// TIA Portal project "pro_2EV_N" (V16)
// Programa original de la laminadora

(* hardware
DEVICE "S7-1200 station_1"  S7-1200 Station
   slot 0: "Telaio di montaggio_0"  S7-1200 Rack  Rack  V1.0
   slot 1: "PLC"  CPU 1214C DC/DC/DC  6ES7 214-1AG40-0XB0  V4.4
   slot 2: "DQ 8x24VDC _1"  SM 1222 DQ8 x 24VDC  6ES7 222-1BF32-0XB0  V2.0
   slot 3: "AI 4xTC_1"  SM 1231 AI4 x TC  6ES7 231-5QD32-0XB0  V2.0
   slot 3: "DQ 4x24VDC_1"  DQ4 signal board (200 kHz)  6ES7 222-1BD30-0XB0  V1.0
*)

// ===== PLC "PLC"  CPU 1214C DC/DC/DC =====

VAR_GLOBAL   // PLC tag table "Tabla de variables estándar"
   "Emergenza" AT %I0.0 : Bool;
   "P_Reset" AT %I0.1 : Bool;
   "P_Stop_Sirena" AT %I0.2 : Bool;
   "Fc_Coperchio_Chiuso" AT %I0.5 : Bool;
   "Pressostato Aria" AT %I0.6 : Bool;
   "Fedd Back Pompa Vuoto" AT %I0.4 : Bool;
   "Analog Vuoto Sotto" AT %IW64 : Int;
   "Analog Vuoto Sopra" AT %IW66 : Int;
   "Feed Back Ins Resistenze" AT %I0.7 : Bool;
   "Temp 1 Basso" AT %IW128 : Int;
   "Temp 2 Basso" AT %IW130 : Int;
   "Temp 1 Alto" AT %IW132 : Int;
   "iw134" AT %IW134 : Word;
   "i0.3" AT %I0.3 : Bool;
   "Fc Pin Alti" AT %I1.0 : Bool;
   "Fc Pin Bassi" AT %I1.1 : Bool;
   "i1.2" AT %I1.2 : Bool;
   "i1.3" AT %I1.3 : Bool;
   "i1.4" AT %I1.4 : Bool;
   "qq" AT %Q2.6 : Bool;
   "Sirena" AT %Q0.0 : Bool;
   "Lamp_Allarme" AT %Q0.1 : Bool;
   "Lamp_Ciclo" AT %Q0.2 : Bool;
   "Lamp_Blu" AT %Q0.3 : Bool;
   "Comando Pompa vuoto" AT %Q0.4 : Bool;
   "EV Vuoto Sotto" AT %Q0.5 : Bool;
   "EV Aria Sotto" AT %Q0.6 : Bool;
   "Ev Big Vuoto Sopra" AT %Q0.7 : Bool;
   "Ev Big Aria Sopra" AT %Q1.0 : Bool;
   "Ev Small Aria Sopra" AT %Q1.1 : Bool;
   "Ev Small Vuoto Sopra" AT %Q2.0 : Bool;
   "Inserzione Resistenze" AT %Q2.1 : Bool;
   "Com Resistenze Basse" AT %Q2.2 : Bool;
   "Com Resistenze Alte" AT %Q2.3 : Bool;
   "EV H2O Raffredda" AT %Q2.4 : Bool;
   "EV Salita Pin" AT %Q2.5 : Bool;
   "Lamp_Reset" AT %Q2.7 : Bool;
   "System_Byte" AT %MB1 : Byte;
   "FirstScan" AT %M1.0 : Bool;
   "DiagStatusUpdate" AT %M1.1 : Bool;
   "AlwaysTRUE" AT %M1.2 : Bool;
   "AlwaysFALSE" AT %M1.3 : Bool;
   "Clock_Byte" AT %MB0 : Byte;
   "Clock_10Hz" AT %M0.0 : Bool;
   "Clock_5Hz" AT %M0.1 : Bool;
   "Clock_2.5Hz" AT %M0.2 : Bool;
   "Clock_2Hz" AT %M0.3 : Bool;
   "Clock_1.25Hz" AT %M0.4 : Bool;
   "Clock_1Hz" AT %M0.5 : Bool;
   "Clock_0.625Hz" AT %M0.6 : Bool;
   "Clock_0.5Hz" AT %M0.7 : Bool;
   "Start Temp Sotto" AT %M110.0 : Bool;
   "Start Temp Sopra" AT %M110.1 : Bool;
   "Mk Emergenza" AT %M90.0 : Bool;
   "Automatico" AT %M100.0 : Bool;
   "Automatico Start" AT %M100.1 : Bool;
   "Automatico Stop" AT %M100.2 : Bool;
   "Allarme" AT %M900.0 : Bool;
   "Ini Auto" AT %M100.3 : Bool;
   "Manuale" AT %M100.4 : Bool;
   "Com Resistenze Sotto" AT %M120.0 : Bool;
   "Com Resistenze Sopra" AT %M120.2 : Bool;
   "Start Vuoto Sotto" AT %M110.2 : Bool;
   "Start Vuoto Sopra" AT %M110.3 : Bool;
   "A1 Allarme Pompa Vuoto" AT %M1000.0 : Bool;
   "HMI Salta basso" AT %M35.0 : Bool;
   "M_OkNextStep" AT %M35.1 : Bool;
   "HMI Start Ciclo" AT %M50.0 : Bool;
   "Reset_T_Passo" AT %M300.0 : Bool;
   "HMI Stop Ciclo" AT %M50.1 : Bool;
   "Auto_ON" AT %M100.5 : Bool;
   "HMI Reset Ciclo" AT %M50.2 : Bool;
   "HMI Ciclo Terminato" AT %M50.3 : Bool;
   "Temp_Sotto in Range" AT %M111.0 : Bool;
   "Temp_Sopra in Range" AT %M111.1 : Bool;
   "Vuoto_Sotto in Range" AT %M111.2 : Bool;
   "Vuoto_Sopra in Range" AT %M111.3 : Bool;
   "S1 Fc Coperchio NON Chiuso" AT %M1010.0 : Bool;
   "MK_Registra_Temp" AT %M230.0 : Bool;
   "MK_Registra_Vuoto" AT %M230.1 : Bool;
   "Tempo_Passo OK" AT %M112.0 : Bool;
   "HMI Start Set Point Man Up" AT %M35.2 : Bool;
   "HMI Start Set Point Man Dw" AT %M35.3 : Bool;
   "HMI Set Point Man Gen" AT %M35.4 : Bool;
   "HMI Man Start Vuoto UP" AT %M35.5 : Bool;
   "HMI Man Start Vuoto DW" AT %M35.6 : Bool;
   "HMI Forzo Resistenze UP" AT %M35.7 : Bool;
   "HMI Forzo Resistenze DW" AT %M36.0 : Bool;
   "HMI Start Pompa Vuoto" AT %M36.1 : Bool;
   "HMI Com EV Vuoto Sotto" AT %M36.2 : Bool;
   "HMI Com EV Aria Sotto" AT %M36.3 : Bool;
   "HMI Com Ev Big Vuoto Sopra" AT %M36.4 : Bool;
   "HMI Com Ev Big Aria Sopra" AT %M36.5 : Bool;
   "HMI Com Ev Small Vuoto Sopra" AT %M36.6 : Bool;
   "HMI Com Resistenze Basse" AT %M37.0 : Bool;
   "HMI Com Resistenze Alte" AT %M37.1 : Bool;
   "HMI Com Ev Small Aria Sopra" AT %M36.7 : Bool;
   "HMI Stop Set Point Man Up" AT %M37.2 : Bool;
   "HMI Stop Set Point Man Dw" AT %M37.3 : Bool;
   "HMI Man Stop Vuoto UP" AT %M37.4 : Bool;
   "HMI Man Stop Vuoto DW" AT %M37.5 : Bool;
   "MK Man Resistenze UP" AT %M120.3 : Bool;
   "MK Man Resistenze DW" AT %M120.4 : Bool;
   "A2 All Max Temp Coperchio" AT %M1000.1 : Bool;
   "A3 All Max Temp Piastra" AT %M1000.2 : Bool;
   "A4 All Max Delta T" AT %M1000.3 : Bool;
   "Tag_1" AT %M10.0 : Bool;
   "Tag_2" AT %M11.0 : Bool;
   "MK Start Man V UP" AT %M112.1 : Bool;
   "MK Start Man V DW" AT %M112.2 : Bool;
   "MK Start Auto V UP" AT %M112.3 : Bool;
   "MK Start Auto V DW" AT %M112.4 : Bool;
   "MK Start Man Temp UP" AT %M112.5 : Bool;
   "MK Start Man Temp DW" AT %M112.6 : Bool;
   "MK Start Auto Temp UP" AT %M112.7 : Bool;
   "MK Start AutoTemp DW" AT %M113.0 : Bool;
   "A5 TimeOut Movimento PIN" AT %M1000.4 : Bool;
   "HMI Man Com PIN" AT %M37.6 : Bool;
   "MKA Salita PIN" AT %M113.1 : Bool;
   "S2 Chiudere il Coperchio" AT %M1010.1 : Bool;
   "MK Salta Passo" AT %M113.2 : Bool;
   "Tag_4" AT %MD1000 : DWord;
   "A6 EMERGENZA" AT %M1000.5 : Bool;
   "A7 All Max Delta T TC Piastra" AT %M1000.6 : Bool;
   "A8 Mancanza Aria" AT %M1000.7 : Bool;
   "A9 FeedBack KM18.1" AT %M1001.0 : Bool;
   "A10" AT %M1001.1 : Bool;
   "A11" AT %M1001.2 : Bool;
   "A12" AT %M1001.3 : Bool;
   "A13" AT %M1001.4 : Bool;
   "A14" AT %M1001.5 : Bool;
   "A15" AT %M1001.6 : Bool;
   "A16" AT %M1001.7 : Bool;
   "A17" AT %M1002.0 : Bool;
   "A18" AT %M1002.1 : Bool;
   "A19" AT %M1002.2 : Bool;
   "A20" AT %M1002.3 : Bool;
   "A21" AT %M1002.4 : Bool;
   "A22" AT %M1002.5 : Bool;
   "A23" AT %M1002.6 : Bool;
   "A24" AT %M1002.7 : Bool;
   "HMI Rese Allarmi" AT %M50.4 : Bool;
   "Tag_5" AT %MD35 : DWord;
   "Tag_6" AT %MD50 : DWord;
   "Tag_7" AT %MD100 : DWord;
   "Tag_8" AT %MD110 : DWord;
   "Tag_9" AT %MD120 : DWord;
   "Tag_10" AT %MD230 : DWord;
   "Tag_11" AT %MD1010 : DWord;
   "Reset Totale" AT %M910.0 : Bool;
   "HMI Man Com H2O" AT %M38.0 : Bool;
   "Mk EV Vuoto Sotto" AT %M130.0 : Bool;
   "Mk EV Aria Sotto" AT %M130.1 : Bool;
   "MK Ev Vuoto Big Sopra" AT %M130.2 : Bool;
   "MK Ev Small Vuoto Sopra" AT %M130.3 : Bool;
   "MK Ev Big Aria Sopra" AT %M130.4 : Bool;
   "MK Ev Small Aria Sopra" AT %M130.5 : Bool;
   "MK EV H20 Raffredda" AT %M130.6 : Bool;
   "MDPIN" AT %MD600 : DWord;
   "HMI Mem Altitudine" AT %M38.1 : Bool;
   "ARCHIVIO_ON" AT %M240.0 : Bool;
   "PIN_RICETTA" AT %MD60 : DWord;
   "PIN_RICETTA_P" AT %M60.0 : Bool;
   "PIN_RICETTA_P_1" AT %M60.1 : Bool;
   "PIN_RICETTA_P_2" AT %M60.2 : Bool;
   "PIN_RICETTA_P_3" AT %M60.3 : Bool;
   "PIN_RICETTA_P_4" AT %M60.4 : Bool;
   "PIN_RICETTA_P_5" AT %M60.5 : Bool;
   "PIN_RICETTA_P_6" AT %M60.6 : Bool;
   "PIN_RICETTA_P_7" AT %M60.7 : Bool;
   "PIN_RICETTA_P_8" AT %M61.0 : Bool;
   "PIN_RICETTA_P_9" AT %M61.1 : Bool;
   "PIN_RICETTA_P_10" AT %M61.2 : Bool;
   "PIN_RICETTA_P_11" AT %M61.3 : Bool;
   "PIN_RICETTA_P_12" AT %M61.4 : Bool;
   "PIN_RICETTA_P_13" AT %M61.5 : Bool;
   "PIN_RICETTA_P_14" AT %M61.6 : Bool;
   "PIN_RICETTA_P_15" AT %M61.7 : Bool;
   "PIN_RICETTA_P_16" AT %M62.0 : Bool;
   "PIN_RICETTA_P_17" AT %M62.1 : Bool;
   "PIN_RICETTA_P_18" AT %M62.2 : Bool;
   "PIN_RICETTA_P_19" AT %M62.3 : Bool;
   "PIN_RICETTA_P_20" AT %M62.4 : Bool;
   "ALLARMI(1)" AT %MW1000 : Word;
   "ARCHIVIO_OFF" AT %M240.1 : Bool;
   "DATAARCHIVIO_ON" AT %MD1004 : Time_Of_Day;
   "DATAARCHIVIO_OFF" AT %MD1014 : Time_Of_Day;
   "Tag_12" AT %M270.0 : Bool;
   "Tag_13" AT %MW1120 : Int;
   "HMI ImpDataOra" AT %M39.0 : Bool;
   "Tag_14" AT %M400.0 : Bool;
   "Tag_17" AT %M432.0 : Bool;
   "Tag_18" AT %M401.6 : Bool;
   "Tag_3" AT %M290.0 : Bool;
   "Tag_15" AT %M290.1 : Bool;
   "Tag_16" AT %MW1840 : Word;
   "Tag_19" AT %MD1840 : Real;
   "Tag_20" AT %M1578.0 : Bool;
   "Tag_21" AT %M1456.0 : Bool;
   "Tag_22" AT %M1523.5 : Bool;
   "Tag_23" AT %M1634.4 : Bool;
   "Tag_24" AT %M1425.3 : Bool;
   "Tag_25" AT %M1511.3 : Bool;
   "Tag_26" AT %M1423.0 : Bool;
   "Tag_27" AT %M1423.1 : Bool;
   "Tag_28" AT %M1523.3 : Bool;
   "HMI Export Vuoto" AT %M150.0 : Bool;
   "Tag_30" AT %MD1600 : Real;
   "Tag_31" AT %MB1250 : Byte;
   "Tag_32" AT %M1252.0 : Bool;
   "Tag_33" AT %M1245.0 : Bool;
   "Tag_34" AT %M763.5 : Bool;
   "ModeActivate PID Piastra" AT %M170.0 : Bool;
   "ModeActivate PID Coperchio" AT %M170.1 : Bool;
   "Errore PID Piastra" AT %M170.2 : Bool;
   "Errore PID Cover" AT %M170.3 : Bool;
   "Tag_35" AT %M700.0 : Bool;
   "Tag_36" AT %M700.2 : Bool;
   "Tag_37" AT %M701.0 : Bool;
   "Tag_38" AT %M705.0 : Bool;
   "Tag_39" AT %M705.1 : Bool;
   "Tag_40" AT %M723.0 : Bool;
   "Tag_41" AT %M723.1 : Bool;
   "Tag_42" AT %M732.0 : Bool;
   "Tag_43" AT %M732.1 : Bool;
   "USB Registra Vuoto" AT %M150.1 : Bool;
   "HMI Export Temp" AT %M151.0 : Bool;
   "USB Registra Temp" AT %M151.1 : Bool;
   "Tag_29" AT %M789.0 : Bool;
   "HMI Segnale Man Cover" AT %M54.0 : Bool;
   "EV Entrada Refrigerante" AT %Q4.0 : Bool;
   "EV purga" AT %Q4.1 : Bool;
   "Process Refri" AT %M70.0 : Bool;
   "Process Refri Fin" AT %M70.1 : Bool;
   "Proces_Refri_Fin" AT %M70.2 : Bool;
   "Refri_Necesaria" AT %M70.3 : Bool;
   "Ref_ON" AT %M70.4 : Bool;
   "REF_RICETTA" AT %MD80 : DWord;
   "REF_RICETTA_" AT %M80.0 : Bool;
   "REF_RICETTA_1" AT %M84.0 : Bool;
   "REF_RICETTA_2" AT %M84.1 : Bool;
   "REF_RICETTA_3" AT %M84.2 : Bool;
   "REF_RICETTA_4" AT %M84.3 : Bool;
   "REF_RICETTA_5" AT %M84.4 : Bool;
   "REF_RICETTA_6" AT %M84.5 : Bool;
   "REF_RICETTA_7" AT %M84.6 : Bool;
   "REF_RICETTA_8" AT %M84.7 : Bool;
   "REF_RICETTA_9" AT %M85.0 : Bool;
   "REF_RICETTA_10" AT %M85.1 : Bool;
   "REF_RICETTA_11" AT %M85.2 : Bool;
   "REF_RICETTA_12" AT %M85.3 : Bool;
   "REF_RICETTA_13" AT %M85.4 : Bool;
   "REF_RICETTA_14" AT %M85.5 : Bool;
   "REF_RICETTA_15" AT %M85.6 : Bool;
   "REF_RICETTA_16" AT %M85.7 : Bool;
   "REF_RICETTA_17" AT %M86.0 : Bool;
   "REF_RICETTA_18" AT %M86.1 : Bool;
   "REF_RICETTA_19" AT %M86.2 : Bool;
   "REF_RICETTA_20" AT %M86.3 : Bool;
END_VAR

TYPE "Dati_Ricetta"
VERSION : 0.1
   STRUCT
      Nome_Ricetta : String;
      "Passo 1" : Struct
         Tempo : Time;
         Vuoto_Sopra : Real;
         Vuoto_Sotto : Real;
         Temperatura_Sopra : Real;
         Temperatura_Sotto : Real;
         Free1 : Real;
         Free2 : Time;
      END_STRUCT;
      "Passo 2" : Struct
         Tempo : Time;
         Vuoto_Sopra : Real;
         Vuoto_Sotto : Real;
         Temperatura_Sopra : Real;
         Temperatura_Sotto : Real;
         Free1 : Real;
         Free2 : Time;
      END_STRUCT;
      "Passo 3" : Struct
         Tempo : Time;
         Vuoto_Sopra : Real;
         Vuoto_Sotto : Real;
         Temperatura_Sopra : Real;
         Temperatura_Sotto : Real;
         Free1 : Real;
         Free2 : Time;
      END_STRUCT;
      "Passo 4" : Struct
         Tempo : Time;
         Vuoto_Sopra : Real;
         Vuoto_Sotto : Real;
         Temperatura_Sopra : Real;
         Temperatura_Sotto : Real;
         Free1 : Real;
         Free2 : Time;
      END_STRUCT;
      "Passo 5" : Struct
         Tempo : Time;
         Vuoto_Sopra : Real;
         Vuoto_Sotto : Real;
         Temperatura_Sopra : Real;
         Temperatura_Sotto : Real;
         Free1 : Real;
         Free2 : Time;
      END_STRUCT;
      "Passo 6" : Struct
         Tempo : Time;
         Vuoto_Sopra : Real;
         Vuoto_Sotto : Real;
         Temperatura_Sopra : Real;
         Temperatura_Sotto : Real;
         Free1 : Real;
         Free2 : Time;
      END_STRUCT;
      "Passo 7" : Struct
         Tempo : Time;
         Vuoto_Sopra : Real;
         Vuoto_Sotto : Real;
         Temperatura_Sopra : Real;
         Temperatura_Sotto : Real;
         Free1 : Real;
         Free2 : Time;
      END_STRUCT;
      "Passo 8" : Struct
         Tempo : Time;
         Vuoto_Sopra : Real;
         Vuoto_Sotto : Real;
         Temperatura_Sopra : Real;
         Temperatura_Sotto : Real;
         Free1 : Real;
         Free2 : Time;
      END_STRUCT;
      "Passo 9" : Struct
         Tempo : Time;
         Vuoto_Sopra : Real;
         Vuoto_Sotto : Real;
         Temperatura_Sopra : Real;
         Temperatura_Sotto : Real;
         Free1 : Real;
         Free2 : Time;
      END_STRUCT;
      "Passo 10" : Struct
         Tempo : Time;
         Vuoto_Sopra : Real;
         Vuoto_Sotto : Real;
         Temperatura_Sopra : Real;
         Temperatura_Sotto : Real;
         Free1 : Real;
         Free2 : Time;
      END_STRUCT;
      "Passo 11" : Struct
         Tempo : Time;
         Vuoto_Sopra : Real;
         Vuoto_Sotto : Real;
         Temperatura_Sopra : Real;
         Temperatura_Sotto : Real;
         Free1 : Real;
         Free2 : Time;
      END_STRUCT;
      "Passo 12" : Struct
         Tempo : Time;
         Vuoto_Sopra : Real;
         Vuoto_Sotto : Real;
         Temperatura_Sopra : Real;
         Temperatura_Sotto : Real;
         Free1 : Real;
         Free2 : Time;
      END_STRUCT;
      "Passo 13" : Struct
         Tempo : Time;
         Vuoto_Sopra : Real;
         Vuoto_Sotto : Real;
         Temperatura_Sopra : Real;
         Temperatura_Sotto : Real;
         Free1 : Real;
         Free2 : Time;
      END_STRUCT;
      "Passo 14" : Struct
         Tempo : Time;
         Vuoto_Sopra : Real;
         Vuoto_Sotto : Real;
         Temperatura_Sopra : Real;
         Temperatura_Sotto : Real;
         Free1 : Real;
         Free2 : Time;
      END_STRUCT;
      "Passo 15" : Struct
         Tempo : Time;
         Vuoto_Sopra : Real;
         Vuoto_Sotto : Real;
         Temperatura_Sopra : Real;
         Temperatura_Sotto : Real;
         Free1 : Real;
         Free2 : Time;
      END_STRUCT;
      "Passo 16" : Struct
         Tempo : Time;
         Vuoto_Sopra : Real;
         Vuoto_Sotto : Real;
         Temperatura_Sopra : Real;
         Temperatura_Sotto : Real;
         Free1 : Real;
         Free2 : Time;
      END_STRUCT;
      "Passo 17" : Struct
         Tempo : Time;
         Vuoto_Sopra : Real;
         Vuoto_Sotto : Real;
         Temperatura_Sopra : Real;
         Temperatura_Sotto : Real;
         Free1 : Real;
         Free2 : Time;
      END_STRUCT;
      "Passo 18" : Struct
         Tempo : Time;
         Vuoto_Sopra : Real;
         Vuoto_Sotto : Real;
         Temperatura_Sopra : Real;
         Temperatura_Sotto : Real;
         Free1 : Real;
         Free2 : Time;
      END_STRUCT;
      "Passo 19" : Struct
         Tempo : Time;
         Vuoto_Sopra : Real;
         Vuoto_Sotto : Real;
         Temperatura_Sopra : Real;
         Temperatura_Sotto : Real;
         Free1 : Real;
         Free2 : Time;
      END_STRUCT;
      "Passo 20" : Struct
         Tempo : Time;
         Vuoto_Sopra : Real;
         Vuoto_Sotto : Real;
         Temperatura_Sopra : Real;
         Temperatura_Sotto : Real;
         Free1 : Real;
         Free2 : Time;
      END_STRUCT;
   END_STRUCT;
END_TYPE

DATA_BLOCK "Ricette"   // DB1
{ S7_Optimized_Access := 'FALSE' }
VERSION : 0.1
   VAR
      Ricetta : String := 'PRUEBA_CALENTAR$00$00$00$00$00';
      Numero : Int := 0;
      PIN_HMI : DWord := 16#0000_0000;
      PIN_Passo : Array[0..31] of Bool;
      "Passo 1" : Struct
         Tempo1 : Time := T#0MS;
         tempo2 : Time := T#0MS;
         "Temperatura UP" : Real := 0.0;
         "Temperatura DW" : Real := 0.0;
         "vuoto sopra" : Real := 0.0;
         "vuoto sotto" : Real := 0.0;
         libero2 : Real := 0.0;
         PIN : Bool := FALSE;
         REF_bit : Bool;
      END_STRUCT;
      "Passo 2" : Struct
         Tempo1 : Time := T#5MS;
         tempo2 : Time := T#0MS;
         "Temperatura UP" : Real := 50.0;
         "Temperatura DW" : Real := 120.0;
         "vuoto sopra" : Real := 0.0;
         "vuoto sotto" : Real := 0.0;
         libero2 : Real := 0.0;
         PIN : Bool := FALSE;
         REF_bit : Bool;
      END_STRUCT;
      "Passo 3" : Struct
         Tempo1 : Time := T#60MS;
         tempo2 : Time := T#0MS;
         "Temperatura UP" : Real := 50.0;
         "Temperatura DW" : Real := 120.0;
         "vuoto sopra" : Real := 1000.0;
         "vuoto sotto" : Real := 1000.0;
         libero2 : Real := 0.0;
         PIN : Bool := FALSE;
         REF_bit : Bool;
      END_STRUCT;
      "Passo 4" : Struct
         Tempo1 : Time := T#10MS;
         tempo2 : Time := T#0MS;
         "Temperatura UP" : Real := 50.0;
         "Temperatura DW" : Real := 120.0;
         "vuoto sopra" : Real := 0.0;
         "vuoto sotto" : Real := 1000.0;
         libero2 : Real := 0.0;
         PIN : Bool := FALSE;
         REF_bit : Bool;
      END_STRUCT;
      "Passo 5" : Struct
         Tempo1 : Time := T#10MS;
         tempo2 : Time := T#0MS;
         "Temperatura UP" : Real := 30.0;
         "Temperatura DW" : Real := 50.0;
         "vuoto sopra" : Real := 0.0;
         "vuoto sotto" : Real := 1000.0;
         libero2 : Real := 0.0;
         PIN : Bool := FALSE;
         REF_bit : Bool;
      END_STRUCT;
      "Passo 6" : Struct
         Tempo1 : Time := T#0MS;
         tempo2 : Time := T#0MS;
         "Temperatura UP" : Real := 0.0;
         "Temperatura DW" : Real := 0.0;
         "vuoto sopra" : Real := 0.0;
         "vuoto sotto" : Real := 0.0;
         libero2 : Real := 0.0;
         PIN : Bool := FALSE;
         REF_bit : Bool;
      END_STRUCT;
      "Passo 7" : Struct
         Tempo1 : Time := T#0MS;
         tempo2 : Time := T#0MS;
         "Temperatura UP" : Real := 0.0;
         "Temperatura DW" : Real := 0.0;
         "vuoto sopra" : Real := 0.0;
         "vuoto sotto" : Real := 0.0;
         libero2 : Real := 0.0;
         PIN : Bool := FALSE;
         REF_bit : Bool;
      END_STRUCT;
      "Passo 8" : Struct
         Tempo1 : Time := T#0MS;
         tempo2 : Time := T#0MS;
         "Temperatura UP" : Real := 0.0;
         "Temperatura DW" : Real := 0.0;
         "vuoto sopra" : Real := 0.0;
         "vuoto sotto" : Real := 0.0;
         libero2 : Real := 0.0;
         PIN : Bool := FALSE;
         REF_bit : Bool;
      END_STRUCT;
      "Passo 9" : Struct
         Tempo1 : Time := T#0MS;
         tempo2 : Time := T#0MS;
         "Temperatura UP" : Real := 0.0;
         "Temperatura DW" : Real := 0.0;
         "vuoto sopra" : Real := 0.0;
         "vuoto sotto" : Real := 0.0;
         libero2 : Real := 0.0;
         PIN : Bool := FALSE;
         REF_bit : Bool;
      END_STRUCT;
      "Passo 10" : Struct
         Tempo1 : Time := T#0MS;
         tempo2 : Time := T#0MS;
         "Temperatura UP" : Real := 0.0;
         "Temperatura DW" : Real := 0.0;
         "vuoto sopra" : Real := 0.0;
         "vuoto sotto" : Real := 0.0;
         libero2 : Real := 0.0;
         PIN : Bool := FALSE;
         REF_bit : Bool;
      END_STRUCT;
      "Passo 11" : Struct
         Tempo1 : Time := T#0MS;
         tempo2 : Time := T#0MS;
         "Temperatura UP" : Real := 0.0;
         "Temperatura DW" : Real := 0.0;
         "vuoto sopra" : Real := 0.0;
         "vuoto sotto" : Real := 0.0;
         libero2 : Real := 0.0;
         PIN : Bool := FALSE;
         REF_bit : Bool;
      END_STRUCT;
      "Passo 12" : Struct
         Tempo1 : Time := T#0MS;
         tempo2 : Time := T#0MS;
         "Temperatura UP" : Real := 0.0;
         "Temperatura DW" : Real := 0.0;
         "vuoto sopra" : Real := 0.0;
         "vuoto sotto" : Real := 0.0;
         libero2 : Real := 0.0;
         PIN : Bool := FALSE;
         REF_bit : Bool;
      END_STRUCT;
      "Passo 13" : Struct
         Tempo1 : Time := T#0MS;
         tempo2 : Time := T#0MS;
         "Temperatura UP" : Real := 0.0;
         "Temperatura DW" : Real := 0.0;
         "vuoto sopra" : Real := 0.0;
         "vuoto sotto" : Real := 0.0;
         libero2 : Real := 0.0;
         PIN : Bool := FALSE;
         REF_bit : Bool;
      END_STRUCT;
      "Passo 14" : Struct
         Tempo1 : Time := T#0MS;
         tempo2 : Time := T#0MS;
         "Temperatura UP" : Real := 0.0;
         "Temperatura DW" : Real := 0.0;
         "vuoto sopra" : Real := 0.0;
         "vuoto sotto" : Real := 0.0;
         libero2 : Real := 0.0;
         PIN : Bool := FALSE;
         REF_bit : Bool;
      END_STRUCT;
      "Passo 15" : Struct
         Tempo1 : Time := T#0MS;
         tempo2 : Time := T#0MS;
         "Temperatura UP" : Real := 0.0;
         "Temperatura DW" : Real := 0.0;
         "vuoto sopra" : Real := 0.0;
         "vuoto sotto" : Real := 0.0;
         libero2 : Real := 0.0;
         PIN : Bool := FALSE;
         REF_bit : Bool;
      END_STRUCT;
      "Passo 16" : Struct
         Tempo1 : Time := T#0MS;
         tempo2 : Time := T#0MS;
         "Temperatura UP" : Real := 0.0;
         "Temperatura DW" : Real := 0.0;
         "vuoto sopra" : Real := 0.0;
         "vuoto sotto" : Real := 0.0;
         libero2 : Real := 0.0;
         PIN : Bool := FALSE;
         REF_bit : Bool;
      END_STRUCT;
      "Passo 17" : Struct
         Tempo1 : Time := T#0MS;
         tempo2 : Time := T#0MS;
         "Temperatura UP" : Real := 0.0;
         "Temperatura DW" : Real := 0.0;
         "vuoto sopra" : Real := 0.0;
         "vuoto sotto" : Real := 0.0;
         libero2 : Real := 0.0;
         PIN : Bool := FALSE;
         REF_bit : Bool;
      END_STRUCT;
      "Passo 18" : Struct
         Tempo1 : Time := T#0MS;
         tempo2 : Time := T#0MS;
         "Temperatura UP" : Real := 0.0;
         "Temperatura DW" : Real := 0.0;
         "vuoto sopra" : Real := 0.0;
         "vuoto sotto" : Real := 0.0;
         libero2 : Real := 0.0;
         PIN : Bool := FALSE;
         REF_bit : Bool;
      END_STRUCT;
      "Passo 19" : Struct
         Tempo1 : Time := T#0MS;
         tempo2 : Time := T#0MS;
         "Temperatura UP" : Real := 0.0;
         "Temperatura DW" : Real := 0.0;
         "vuoto sopra" : Real := 0.0;
         "vuoto sotto" : Real := 0.0;
         libero2 : Real := 0.0;
         PIN : Bool := FALSE;
         REF_bit : Bool;
      END_STRUCT;
      "Passo 20" : Struct
         Tempo1 : Time := T#0MS;
         tempo2 : Time := T#0MS;
         "Temperatura UP" : Real := 0.0;
         "Temperatura DW" : Real := 0.0;
         "vuoto sopra" : Real := 0.0;
         "vuoto sotto" : Real := 0.0;
         libero2 : Real := 0.0;
         PIN : Bool := FALSE;
         REF_bit : Bool;
      END_STRUCT;
      REF_bit_Passo : Array[0..31] of Bool;
   END_VAR
BEGIN
   PIN_Passo[0] := FALSE;
   PIN_Passo[1] := FALSE;
   PIN_Passo[2] := FALSE;
   PIN_Passo[3] := FALSE;
   PIN_Passo[4] := FALSE;
   PIN_Passo[5] := FALSE;
   PIN_Passo[6] := FALSE;
   PIN_Passo[7] := FALSE;
   PIN_Passo[8] := FALSE;
   PIN_Passo[9] := FALSE;
   PIN_Passo[10] := FALSE;
   PIN_Passo[11] := FALSE;
   PIN_Passo[12] := FALSE;
   PIN_Passo[13] := FALSE;
   PIN_Passo[14] := FALSE;
   PIN_Passo[15] := FALSE;
   PIN_Passo[16] := FALSE;
   PIN_Passo[17] := FALSE;
   PIN_Passo[18] := FALSE;
   PIN_Passo[19] := FALSE;
   PIN_Passo[20] := FALSE;
   PIN_Passo[21] := FALSE;
   PIN_Passo[22] := FALSE;
   PIN_Passo[23] := FALSE;
   PIN_Passo[24] := FALSE;
   PIN_Passo[25] := FALSE;
   PIN_Passo[26] := FALSE;
   PIN_Passo[27] := FALSE;
   PIN_Passo[28] := FALSE;
   PIN_Passo[29] := FALSE;
   PIN_Passo[30] := FALSE;
   PIN_Passo[31] := FALSE;
END_DATA_BLOCK

DATA_BLOCK "Temperature"   // DB2
{ S7_Optimized_Access := 'FALSE' }
VERSION : 0.1
   VAR
      Temperatura_Auto : Real := 0.0;
      "Termocoppia Piastra 1" : Real := 1100.0;
      "Divisore TC1 Piastra" : Real := 10.0;
      "Correzione TC1 Piastra" : Real := 0.0;
      "Appo TC1" : Real := 110.0;
      "Max Temperatura Piastra" : Real := 200.0;
      "Termocoppia Piastra 2" : Real := 1102.0;
      "Divisore TC2 Piastra" : Real := 10.0;
      "Correzione TC2 Piastra" : Real := 0.0;
      "Appo TC2" : Real := 110.2;
      "Max_Delta T  Cop/Piastra" : Real := 150.0;
      "Max Delta T Termocoppie DW" : Real := 20.0;
      "Delta TT Istantaneo" : Real := -0.1999969;
      "Delta Appoggio" : Real := -20.0;
      "Termocoppia coperchio" : Real := 301.0;
      "Divisore TC Coperchio" : Real := 10.0;
      "Correzione TC Coperchio" : Real := 0.0;
      "Appo TC Cop" : Real := 30.1;
      "Max Temperatura Coperchio" : Real := 72.0;
      "Temperatura Piastra" : Real := 110.1;
      "Temperatura coperchio" : Real := 30.1;
      "Set_point Piastra" : Real := 110.0;
      "Set Point Coperchio" : Real := 48.0;
      "Set Point Generale" : Real := 0.0;
      "Set Point Man Sopra" : Real := 89.0;
      "Set Point Man Sotto" : Real := 110.0;
      "Set Point Man Generale" : Real := 0.0;
      HMI_Toll_Temp_Passo_UP : Real := 6.0;
      HMI_Toll_Temp_Passo_DW : Real := 3.5;
      "SogliaPasso_T_UP+" : Real := 54.0;
      "SogliaPasso_T_UP-" : Real := 42.0;
      "SogliaPasso_T_DW+" : Real := 2.0;
      "SogliaPasso_T_DW-" : Real := -2.0;
      "Tolleranza -1 Piastra" : Real := 3.0;
      "Tolleranza -2 Piastra" : Real := 5.0;
      "Tolleranza -3 Piastra" : Real := 10.0;
      "Tolleranza -4 Piastra" : Real := 20.0;
      "Tolleranza +1 Piastra" : Real := 0.1;
      "DeltaTemp x H2O Piastra" : Real := 1.8;
      "Soglia -1 Piastra" : Real := -3.0;
      "Soglia -2 Piastra" : Real := -5.0;
      "Soglia -3 Piastra" : Real := -10.0;
      "Soglia -4 Piastra" : Real := -20.0;
      "Soglia +1 Piastra" : Real := 0.1;
      "Soglia C° X H2O Piastra" : Real := 1.8;
      free : Real := 0.0;
      "Tolleranza -1 Coperchio" : Real := 1.0;
      "Tolleranza -2 Coperchio" : Real := 2.5;
      "Tolleranza -3 Coperchio" : Real := 5.0;
      "Tolleranza -4 Coperchio" : Real := 10.0;
      "Tolleranza +1 Coperchio" : Real := 0.5;
      "DeltaTemp x H2O Coperchio" : Real := 7.0;
      "Soglia -1 Coperchio" : Real := 47.0;
      "Soglia -2 Coperchio" : Real := 45.5;
      "Soglia -3 Coperchio" : Real := 43.0;
      "Soglia -4 Coperchio" : Real := 38.0;
      "Soglia +1 Coperchio" : Real := 48.5;
      "Soglia C° X H2O Coperchio" : Real := 0.0;
      free2 : Real := 0.0;
      "T_ON 1 Piastra" : Time := T#1S;
      "T_OFF 1 Piastra" : Time := T#1S_500MS;
      "T_ON 2 Piastra" : Time := T#1S;
      "T_OFF 2 Piastra" : Time := T#1S;
      "T_ON 3 Piastra" : Time := T#5S;
      "T_OFF 3 Piastra" : Time := T#1S;
      "T_ON 4 Piastra" : Time := T#10S;
      "T_OFF 4 Piastra" : Time := T#1S;
      "T_ON 5 Piastra" : Time := T#250MS;
      "T_OFF 5 Piastra" : Time := T#3S;
      "T_ON 1 Coperchio" : Time := T#3S;
      "T_OFF 1 Coperchio" : Time := T#700MS;
      "T_ON 2 Coperchio" : Time := T#5S;
      "T_OFF 2 Coperchio" : Time := T#500MS;
      "T_ON 3 Coperchio" : Time := T#10S;
      "T_OFF 3 Coperchio" : Time := T#1S;
      "T_ON 4 Coperchio" : Time := T#20S;
      "T_OFF 4 Coperchio" : Time := T#1S;
      "T_ON 5 Coperchio" : Time := T#750MS;
      "T_OFF 5 Coperchio" : Time := T#1S;
      "Min Valore temp UP" : Int;
      "Max Valore temp UP" : Int := 72;
      "Min Valore temp DW" : Int;
      "Max Valore temp DW" : Int := 200;
   END_VAR
BEGIN
END_DATA_BLOCK

DATA_BLOCK "Vuoto"   // DB3
{ S7_Optimized_Access := 'FALSE' }
VERSION : 0.1
   VAR
      "TFM Motore Pompa Vuoto" : Time := T#3M;
      "Valore Vuoto Sotto" : Real := 793.5913;
      "K x4mA_VuotoSotto" : Real := 5450.0;
      "Divisore Vuoto Sotto" : Real := 22.02;
      "K Correggi Vuoto Sotto" : Real := -994.0;
      "SetPoint Vuoto Sotto" : Real := 800.0;
      "SetPoint Man Vuoto Sotto" : Real := 800.0;
      "Tolleranza a 1000 Sotto" : Real := 50.0;
      "Soglia Max Sotto" : Real := 950.0;
      "Tolleranza +1 Sotto_Vuoto" : Real := 10.0;
      "Tolleranza -1 Sotto_Aria" : Real := 10.0;
      "Soglia +1 Sotto Vuoto" : Real := 790.0;
      "Soglia -1 Sotto Aria" : Real := 810.0;
      "Tolleranza Sotto Automatico" : Real := 30.0;
      "Soglia Sotto + Auto" : Real := 830.0;
      "Soglia Sotto - Auto" : Real := 770.0;
      "Valore Vuoto Sopra" : Real := 172.5046;
      "Divisore Vuoto Sopra" : Real := 22.034;
      "K x4mA_VuotoSopra" : Real := 5440.0;
      "K Correggi Vuoto Sopra" : Real := -999.0;
      "SetPoint Vuoto Sopra" : Real := 0.0;
      "SetPoint Man Vuoto Sopra" : Real := 0.0;
      "Tolleranza a 1000 Sopra" : Real := 50.0;
      "Soglia Max Sopra" : Real := 950.0;
      "Tolleranza +1Fine Sopra" : Real := 0.0;
      "Tolleranza +2Grossa Sopra" : Real := 25.0;
      "Tolleranza -1Fine Sopra" : Real := 10.0;
      "Tolleranza -2 Grossa Sopra" : Real := 100.0;
      "Tolleranza Passo Coperchio" : Real := 1.0;
      "Tolleranza Passo Piastra" : Real := 1.0;
      "Tolleranza Zero" : Real := 10.0;
      "Soglia +1 Fine Sopra" : Real := 0.0;
      "Soglia -1 Fine Sopra" : Real := -10.0;
      "Soglia +2 Grossa Sopra" : Real := 25.0;
      "Soglia -2 Grossa Sopra" : Real := -100.0;
      "Tolleranza Sopra Automatico" : Real := 30.0;
      "Soglia Sopra + Auto" : Real := 30.0;
      "Soglia Sopra - Auto" : Real := -30.0;
      testint : Int := 0;
      K_Altitudine_V_UP : Real := 0.0;
      K_Altitudine_V_DW : Real := 0.0;
   END_VAR
BEGIN
END_DATA_BLOCK

DATA_BLOCK "Dati Ciclo"   // DB4
{ S7_Optimized_Access := 'FALSE' }
VERSION : 0.1
   VAR
      "Stato Macchina" : Int;
      Ab_Auto_Passo : Int;
      CicloAutPasso : Int;
      A_PassoRicetta : Int;
      "Passo in Corso" : Struct
         Tempo1 : Time;
         tempo2 : Time;
         "Temperatura UP" : Real;
         "Temperatura DW" : Real;
         "vuoto sopra" : Real;
         "vuoto sotto" : Real;
         libero2 : Real;
         PIN : Bool;
         REF_bit : Bool;
      END_STRUCT;
      Tempo1_sec : Time;
      Tempo2_sec : Time;
      HMI_DurataPasso : Int;
      App_T_Passo : Real;
      Tempo_Passo : Time;
      T_Resto_Passo : Time;
      Temperatura_Passo : Real;
      Vuoto_Sopra_Passo : Real;
      Vuoto_Sotto_Passo : Real;
      pin1 : Real;
      pin2 : DInt;
      pin3 : DWord;
      TemperaturaSottoDINT : DInt;
      Tempo_X_MiniSet : Time;
      t1xminiset : Time;
      Miniset_DINT : DInt;
      Miniset_DINT_1 : DInt;
      Miniset_DINT_2 : DInt;
      MiniSet_P : Real;
      MiniSet_P_1 : Real;
      MiniSet_P_2 : Real;
      SP_PassoPrec : Real;
      SP_PassoAttu : Real;
      Delta_T_Passo : Real;
   END_VAR
BEGIN
END_DATA_BLOCK

DATA_BLOCK "Parametri Macchina"   // DB5
{ S7_Optimized_Access := 'FALSE' }
VERSION : 0.1
   VAR
      Modello : Array[0..20] of Word;
      "Temp Provvisoria" : Real;
   END_VAR
BEGIN
END_DATA_BLOCK

DATA_BLOCK "Trend"   // DB6
{ S7_Optimized_Access := 'FALSE' }
VERSION : 0.1
   VAR
      Trend_Temperature : Array[0..3] of Real;
      Tred_Pressioni : Array[0..3] of Real;
      "Time Trend Temp" : Time := T#10s;
      "Time Trend Pression" : Time := T#10s;
      Trend_Temperature_HS : Array[0..3] of Real;
      Tred_Pressioni_HS : Array[0..3] of Real;
   END_VAR
BEGIN
END_DATA_BLOCK

DATA_BLOCK "Blocco_dati_1"   // DB7
{ S7_Optimized_Access := 'FALSE' }
VERSION : 0.1
   VAR
      "HMI Num Pagina" : Int;
      "HMI NumPasso" : Int;
      f : Int;
      RTM_imposta_Conta : DInt;
      RTM_ReturnValue : Int;
      RTM_Status : Bool;
      RTM_CurrentValue : DInt;
      RTM_ComandMode : Byte := 16#1;
      RPIN : DWord;
   END_VAR
BEGIN
END_DATA_BLOCK

DATA_BLOCK "Data_ora"   // DB8
{ S7_Optimized_Access := 'FALSE' }
VERSION : 0.1
   VAR
      dataora : DTL := DTL#2022-06-01-13:15:53.231817;
      "return" : Int := 0;
      anno : Int := 2022;
      mese : Int := 6;
      giorno : Int := 1;
      giornosettimanale : Int := 4;
      ora : Int := 13;
      minuti : Int := 15;
      secondi : Int := 53;
      w8 : Int := 0;
      w9 : Int := 0;
      inputdataora : DTL := DTL#2022-06-01-12:03:00;
      returninputDTL : Int := 0;
      dataArchivioON : DTL := DTL#2022-06-01-11:26:19.989299;
      "add time" : Time := T#10s;
      "local time" : Time_Of_Day;
   END_VAR
BEGIN
END_DATA_BLOCK

DATA_BLOCK "Ricetta In Uso"   // DB10
{ S7_Optimized_Access := 'FALSE' }
VERSION : 0.1
   VAR
      Ricetta : Array[0..20] of Word;
      Numero : Int;
      PIN_HMI : DWord;
      PIN_Passo : Array[0..31] of Bool;
      "Passo 1" : Struct
         Tempo1 : Time;
         tempo2 : Time;
         "Temperatura UP" : Real;
         "Temperatura DW" : Real;
         "vuoto sopra" : Real;
         "vuoto sotto" : Real;
         libero2 : Real;
         PIN : Bool;
         REF_bit : Bool;
      END_STRUCT;
      "Passo 2" : Struct
         Tempo1 : Time;
         tempo2 : Time;
         "Temperatura UP" : Real;
         "Temperatura DW" : Real;
         "vuoto sopra" : Real;
         "vuoto sotto" : Real;
         libero2 : Real;
         PIN : Bool;
         REF_bit : Bool;
      END_STRUCT;
      "Passo 3" : Struct
         Tempo1 : Time;
         tempo2 : Time;
         "Temperatura UP" : Real;
         "Temperatura DW" : Real;
         "vuoto sopra" : Real;
         "vuoto sotto" : Real;
         libero2 : Real;
         PIN : Bool;
         REF_bit : Bool;
      END_STRUCT;
      "Passo 4" : Struct
         Tempo1 : Time;
         tempo2 : Time;
         "Temperatura UP" : Real;
         "Temperatura DW" : Real;
         "vuoto sopra" : Real;
         "vuoto sotto" : Real;
         libero2 : Real;
         PIN : Bool;
         REF_bit : Bool;
      END_STRUCT;
      "Passo 5" : Struct
         Tempo1 : Time;
         tempo2 : Time;
         "Temperatura UP" : Real;
         "Temperatura DW" : Real;
         "vuoto sopra" : Real;
         "vuoto sotto" : Real;
         libero2 : Real;
         PIN : Bool;
         REF_bit : Bool;
      END_STRUCT;
      "Passo 6" : Struct
         Tempo1 : Time;
         tempo2 : Time;
         "Temperatura UP" : Real;
         "Temperatura DW" : Real;
         "vuoto sopra" : Real;
         "vuoto sotto" : Real;
         libero2 : Real;
         PIN : Bool;
         REF_bit : Bool;
      END_STRUCT;
      "Passo 7" : Struct
         Tempo1 : Time;
         tempo2 : Time;
         "Temperatura UP" : Real;
         "Temperatura DW" : Real;
         "vuoto sopra" : Real;
         "vuoto sotto" : Real;
         libero2 : Real;
         PIN : Bool;
         REF_bit : Bool;
      END_STRUCT;
      "Passo 8" : Struct
         Tempo1 : Time;
         tempo2 : Time;
         "Temperatura UP" : Real;
         "Temperatura DW" : Real;
         "vuoto sopra" : Real;
         "vuoto sotto" : Real;
         libero2 : Real;
         PIN : Bool;
         REF_bit : Bool;
      END_STRUCT;
      "Passo 9" : Struct
         Tempo1 : Time;
         tempo2 : Time;
         "Temperatura UP" : Real;
         "Temperatura DW" : Real;
         "vuoto sopra" : Real;
         "vuoto sotto" : Real;
         libero2 : Real;
         PIN : Bool;
         REF_bit : Bool;
      END_STRUCT;
      "Passo 10" : Struct
         Tempo1 : Time;
         tempo2 : Time;
         "Temperatura UP" : Real;
         "Temperatura DW" : Real;
         "vuoto sopra" : Real;
         "vuoto sotto" : Real;
         libero2 : Real;
         PIN : Bool;
         REF_bit : Bool;
      END_STRUCT;
      "Passo 11" : Struct
         Tempo1 : Time;
         tempo2 : Time;
         "Temperatura UP" : Real;
         "Temperatura DW" : Real;
         "vuoto sopra" : Real;
         "vuoto sotto" : Real;
         libero2 : Real;
         PIN : Bool;
         REF_bit : Bool;
      END_STRUCT;
      "Passo 12" : Struct
         Tempo1 : Time;
         tempo2 : Time;
         "Temperatura UP" : Real;
         "Temperatura DW" : Real;
         "vuoto sopra" : Real;
         "vuoto sotto" : Real;
         libero2 : Real;
         PIN : Bool;
         REF_bit : Bool;
      END_STRUCT;
      "Passo 13" : Struct
         Tempo1 : Time;
         tempo2 : Time;
         "Temperatura UP" : Real;
         "Temperatura DW" : Real;
         "vuoto sopra" : Real;
         "vuoto sotto" : Real;
         libero2 : Real;
         PIN : Bool;
         REF_bit : Bool;
      END_STRUCT;
      "Passo 14" : Struct
         Tempo1 : Time;
         tempo2 : Time;
         "Temperatura UP" : Real;
         "Temperatura DW" : Real;
         "vuoto sopra" : Real;
         "vuoto sotto" : Real;
         libero2 : Real;
         PIN : Bool;
         REF_bit : Bool;
      END_STRUCT;
      "Passo 15" : Struct
         Tempo1 : Time;
         tempo2 : Time;
         "Temperatura UP" : Real;
         "Temperatura DW" : Real;
         "vuoto sopra" : Real;
         "vuoto sotto" : Real;
         libero2 : Real;
         PIN : Bool;
         REF_bit : Bool;
      END_STRUCT;
      "Passo 16" : Struct
         Tempo1 : Time;
         tempo2 : Time;
         "Temperatura UP" : Real;
         "Temperatura DW" : Real;
         "vuoto sopra" : Real;
         "vuoto sotto" : Real;
         libero2 : Real;
         PIN : Bool;
         REF_bit : Bool;
      END_STRUCT;
      "Passo 17" : Struct
         Tempo1 : Time;
         tempo2 : Time;
         "Temperatura UP" : Real;
         "Temperatura DW" : Real;
         "vuoto sopra" : Real;
         "vuoto sotto" : Real;
         libero2 : Real;
         PIN : Bool;
         REF_bit : Bool;
      END_STRUCT;
      "Passo 18" : Struct
         Tempo1 : Time;
         tempo2 : Time;
         "Temperatura UP" : Real;
         "Temperatura DW" : Real;
         "vuoto sopra" : Real;
         "vuoto sotto" : Real;
         libero2 : Real;
         PIN : Bool;
         REF_bit : Bool;
      END_STRUCT;
      "Passo 19" : Struct
         Tempo1 : Time;
         tempo2 : Time;
         "Temperatura UP" : Real;
         "Temperatura DW" : Real;
         "vuoto sopra" : Real;
         "vuoto sotto" : Real;
         libero2 : Real;
         PIN : Bool;
         REF_bit : Bool;
      END_STRUCT;
      "Passo 20" : Struct
         Tempo1 : Time;
         tempo2 : Time;
         "Temperatura UP" : Real;
         "Temperatura DW" : Real;
         "vuoto sopra" : Real;
         "vuoto sotto" : Real;
         libero2 : Real;
         PIN : Bool;
         REF_bit : Bool;
      END_STRUCT;
      Test_bit : Bool;
      REF_bit_Passo : Array[0..31] of Bool;
   END_VAR
BEGIN
END_DATA_BLOCK

DATA_BLOCK "DDD"   // DB11
{ S7_Optimized_Access := 'FALSE' }
VERSION : 0.1
   VAR
      anno : Int := 2022;
      mese : Int := 6;
      giorno : Int := 1;
      giornosettimanale : Int := 4;
      ora : Int := 13;
      minuti : Int := 15;
      secondi : Int := 53;
      w8 : Int := 0;
      w9 : Int := 0;
   END_VAR
BEGIN
END_DATA_BLOCK

DATA_BLOCK "Dati PID"   // DB12
{ S7_Optimized_Access := 'FALSE' }
VERSION : 0.1
   VAR
      "Modo PID Piastra" : Int := 3;
      "Modo PID Coperchio" : Int := 3;
      "Errore PID Piastra" : Int;
      "Errore PID Cover" : Int;
      "State PID Piastra" : Int;
      "State PID Cover" : Int;
      "Gain PID Piastra" : Real := 50.0;
      "Ti PID Piastra" : Real := 100.0;
      "Td PID Piastra" : Real := 5.0;
      "Gain PID Cover" : Real := 200.0;
      "Ti PID Cover" : Real := 1.0;
      "Td PID Cover" : Real;
   END_VAR
BEGIN
END_DATA_BLOCK

DATA_BLOCK "TITOLORICETTA"   // DB13
{ S7_Optimized_Access := 'TRUE' }
VERSION : 0.1
   VAR
      TITOLO : String;
   END_VAR
BEGIN
END_DATA_BLOCK

// folder: System blocks/Program resources

DATA_BLOCK "IEC_Timer_0_DB_6"   // DB14
{ S7_Optimized_Access := 'TRUE' }
AUTHOR : Simatic
FAMILY : IEC
NAME : IEC_TMR
VERSION : 1.0
// stored: InstanceOfName IEC_TIMER
"IEC_TIMER"
BEGIN
END_DATA_BLOCK

DATA_BLOCK "IEC_Timer_0_DB_7"   // DB15
{ S7_Optimized_Access := 'TRUE' }
AUTHOR : Simatic
FAMILY : IEC
NAME : IEC_TMR
VERSION : 1.0
// stored: InstanceOfName IEC_TIMER
"IEC_TIMER"
BEGIN
END_DATA_BLOCK

DATA_BLOCK "IEC_Timer_0_DB_10"   // DB18
{ S7_Optimized_Access := 'TRUE' }
AUTHOR : Simatic
FAMILY : IEC
NAME : IEC_TMR
VERSION : 1.0
// stored: InstanceOfName IEC_TIMER
"IEC_TIMER"
BEGIN
END_DATA_BLOCK

DATA_BLOCK "IEC_Timer_0_DB_3"   // DB122
{ S7_Optimized_Access := 'TRUE' }
AUTHOR : Simatic
FAMILY : IEC
NAME : IEC_TMR
VERSION : 1.0
// stored: InstanceOfName IEC_TIMER
"IEC_TIMER"
BEGIN
END_DATA_BLOCK

DATA_BLOCK "IEC_Timer_0_DB_12"   // DB123
{ S7_Optimized_Access := 'TRUE' }
AUTHOR : Simatic
FAMILY : IEC
NAME : IEC_TMR
VERSION : 1.0
// stored: InstanceOfName IEC_TIMER
"IEC_TIMER"
BEGIN
END_DATA_BLOCK

DATA_BLOCK "IEC_Timer_0_DB_14"   // DB124
{ S7_Optimized_Access := 'TRUE' }
AUTHOR : Simatic
FAMILY : IEC
NAME : IEC_TMR
VERSION : 1.0
// stored: InstanceOfName IEC_TIMER
"IEC_TIMER"
BEGIN
END_DATA_BLOCK

DATA_BLOCK "IEC_Timer_0_DB_15"   // DB125
{ S7_Optimized_Access := 'TRUE' }
AUTHOR : Simatic
FAMILY : IEC
NAME : IEC_TMR
VERSION : 1.0
// stored: InstanceOfName IEC_TIMER
"IEC_TIMER"
BEGIN
END_DATA_BLOCK

DATA_BLOCK "IEC_Timer_0_DB_16"   // DB126
{ S7_Optimized_Access := 'TRUE' }
AUTHOR : Simatic
FAMILY : IEC
NAME : IEC_TMR
VERSION : 1.0
// stored: InstanceOfName IEC_TIMER
"IEC_TIMER"
BEGIN
END_DATA_BLOCK

DATA_BLOCK "IEC_Timer_0_DB_13"   // DB130
{ S7_Optimized_Access := 'TRUE' }
AUTHOR : Simatic
FAMILY : IEC
NAME : IEC_TMR
VERSION : 1.0
// stored: InstanceOfName IEC_TIMER
"IEC_TIMER"
BEGIN
END_DATA_BLOCK

DATA_BLOCK "IEC_Timer_0_DB_4"   // DB131
{ S7_Optimized_Access := 'TRUE' }
AUTHOR : Simatic
FAMILY : IEC
NAME : IEC_TMR
VERSION : 1.0
// stored: InstanceOfName IEC_TIMER
"IEC_TIMER"
BEGIN
END_DATA_BLOCK

DATA_BLOCK "IEC_Timer_0_DB_41"   // DB132
{ S7_Optimized_Access := 'TRUE' }
AUTHOR : Simatic
FAMILY : IEC
NAME : IEC_TMR
VERSION : 1.0
// stored: InstanceOfName IEC_TIMER
"IEC_TIMER"
BEGIN
END_DATA_BLOCK

DATA_BLOCK "IEC_Timer_0_DB_26"   // DB133
{ S7_Optimized_Access := 'TRUE' }
AUTHOR : Simatic
FAMILY : IEC
NAME : IEC_TMR
VERSION : 1.0
// stored: InstanceOfName IEC_TIMER
"IEC_TIMER"
BEGIN
END_DATA_BLOCK

DATA_BLOCK "IEC_Timer_0_DB_18"   // DB134
{ S7_Optimized_Access := 'TRUE' }
AUTHOR : Simatic
FAMILY : IEC
NAME : IEC_TMR
VERSION : 1.0
// stored: InstanceOfName IEC_TIMER
"IEC_TIMER"
BEGIN
END_DATA_BLOCK

DATA_BLOCK "IEC_Timer_0_DB_17"   // DB135
{ S7_Optimized_Access := 'TRUE' }
AUTHOR : Simatic
FAMILY : IEC
NAME : IEC_TMR
VERSION : 1.0
// stored: InstanceOfName IEC_TIMER
"IEC_TIMER"
BEGIN
END_DATA_BLOCK

DATA_BLOCK "IEC_Timer_0_DB_27"   // DB136
{ S7_Optimized_Access := 'TRUE' }
AUTHOR : Simatic
FAMILY : IEC
NAME : IEC_TMR
VERSION : 1.0
// stored: InstanceOfName IEC_TIMER
"IEC_TIMER"
BEGIN
END_DATA_BLOCK

DATA_BLOCK "IEC_Timer_0_DB_2"   // DB140
{ S7_Optimized_Access := 'TRUE' }
AUTHOR : Simatic
FAMILY : IEC
NAME : IEC_TMR
VERSION : 1.0
// stored: InstanceOfName IEC_TIMER
"IEC_TIMER"
BEGIN
END_DATA_BLOCK

DATA_BLOCK "IEC_Timer_0_DB_28"   // DB141
{ S7_Optimized_Access := 'TRUE' }
AUTHOR : Simatic
FAMILY : IEC
NAME : IEC_TMR
VERSION : 1.0
// stored: InstanceOfName IEC_TIMER
"IEC_TIMER"
BEGIN
END_DATA_BLOCK

DATA_BLOCK "IEC_Timer_0_DB_29"   // DB142
{ S7_Optimized_Access := 'TRUE' }
AUTHOR : Simatic
FAMILY : IEC
NAME : IEC_TMR
VERSION : 1.0
// stored: InstanceOfName IEC_TIMER
"IEC_TIMER"
BEGIN
END_DATA_BLOCK

DATA_BLOCK "IEC_Timer_0_DB"   // DB143
{ S7_Optimized_Access := 'TRUE' }
AUTHOR : Simatic
FAMILY : IEC
NAME : IEC_TMR
VERSION : 1.0
// stored: InstanceOfName IEC_TIMER
"IEC_TIMER"
BEGIN
END_DATA_BLOCK

DATA_BLOCK "IEC_Timer_0_DB_1"   // DB144
{ S7_Optimized_Access := 'TRUE' }
AUTHOR : Simatic
FAMILY : IEC
NAME : IEC_TMR
VERSION : 1.0
// stored: InstanceOfName IEC_TIMER
"IEC_TIMER"
BEGIN
END_DATA_BLOCK

DATA_BLOCK "IEC_Timer_0_DB_31"   // DB145
{ S7_Optimized_Access := 'TRUE' }
AUTHOR : Simatic
FAMILY : IEC
NAME : IEC_TMR
VERSION : 1.0
// stored: InstanceOfName IEC_TIMER
"IEC_TIMER"
BEGIN
END_DATA_BLOCK

DATA_BLOCK "IEC_Timer_0_DB_33"   // DB148
{ S7_Optimized_Access := 'TRUE' }
AUTHOR : Simatic
FAMILY : IEC
NAME : IEC_TMR
VERSION : 1.0
// stored: InstanceOfName IEC_TIMER
"IEC_TIMER"
BEGIN
END_DATA_BLOCK

DATA_BLOCK "IEC_Timer_0_DB_34"   // DB150
{ S7_Optimized_Access := 'TRUE' }
AUTHOR : Simatic
FAMILY : IEC
NAME : IEC_TMR
VERSION : 1.0
// stored: InstanceOfName IEC_TIMER
"IEC_TIMER"
BEGIN
END_DATA_BLOCK

DATA_BLOCK "IEC_Timer_0_DB_35"   // DB151
{ S7_Optimized_Access := 'TRUE' }
AUTHOR : Simatic
FAMILY : IEC
NAME : IEC_TMR
VERSION : 1.0
// stored: InstanceOfName IEC_TIMER
"IEC_TIMER"
BEGIN
END_DATA_BLOCK

DATA_BLOCK "IEC_Timer_0_DB_40"   // DB152
{ S7_Optimized_Access := 'TRUE' }
AUTHOR : Simatic
FAMILY : IEC
NAME : IEC_TMR
VERSION : 1.0
// stored: InstanceOfName IEC_TIMER
"IEC_TIMER"
BEGIN
END_DATA_BLOCK

DATA_BLOCK "IEC_Timer_0_DB_37"   // DB153
{ S7_Optimized_Access := 'TRUE' }
AUTHOR : Simatic
FAMILY : IEC
NAME : IEC_TMR
VERSION : 1.0
// stored: InstanceOfName IEC_TIMER
"IEC_TIMER"
BEGIN
END_DATA_BLOCK

DATA_BLOCK "IEC_Timer_0_DB_39"   // DB154
{ S7_Optimized_Access := 'TRUE' }
AUTHOR : Simatic
FAMILY : IEC
NAME : IEC_TMR
VERSION : 1.0
// stored: InstanceOfName IEC_TIMER
"IEC_TIMER"
BEGIN
END_DATA_BLOCK

DATA_BLOCK "IEC_Timer_0_DB_36"   // DB160
{ S7_Optimized_Access := 'TRUE' }
AUTHOR : Simatic
FAMILY : IEC
NAME : IEC_TMR
VERSION : 1.0
// stored: InstanceOfName IEC_TIMER
"IEC_TIMER"
BEGIN
END_DATA_BLOCK

DATA_BLOCK "IEC_Timer_0_DB_38"   // DB161
{ S7_Optimized_Access := 'TRUE' }
AUTHOR : Simatic
FAMILY : IEC
NAME : IEC_TMR
VERSION : 1.0
// stored: InstanceOfName IEC_TIMER
"IEC_TIMER"
BEGIN
END_DATA_BLOCK

DATA_BLOCK "IEC_Timer_0_DB_32"   // DB180
{ S7_Optimized_Access := 'TRUE' }
AUTHOR : Simatic
FAMILY : IEC
NAME : IEC_TMR
VERSION : 1.0
// stored: InstanceOfName IEC_TIMER
"IEC_TIMER"
BEGIN
END_DATA_BLOCK

DATA_BLOCK "IEC_Timer_0_DB_42"   // DB187
{ S7_Optimized_Access := 'TRUE' }
AUTHOR : Simatic
FAMILY : IEC
NAME : IEC_TMR
VERSION : 1.0
// stored: InstanceOfName IEC_TIMER
"IEC_TIMER"
BEGIN
END_DATA_BLOCK

// folder: (top level)

FUNCTION "PIN" : Void   // FC1, LAD
{ S7_Optimized_Access := 'TRUE' }
VERSION : 0.1
BEGIN

REGION Network 1: Q2.5 EV SALITA PIN
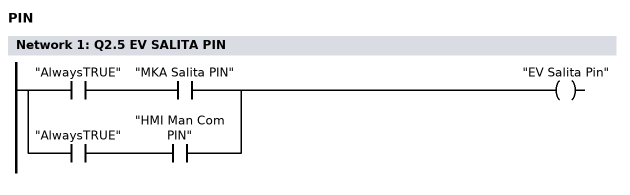
   RUNG wire#powerrail
      Contact( "AlwaysTRUE" )
      Contact( "MKA Salita PIN" )
      wire#w1
      Coil( "EV Salita Pin" )
   END_RUNG
   RUNG wire#powerrail
      Contact( "AlwaysTRUE" )
      Contact( "HMI Man Com PIN" )
   END_RUNG wire#w1
   // the same network as SCL:
   "EV Salita Pin" := ("AlwaysTRUE" AND "MKA Salita PIN") OR ("AlwaysTRUE" AND "HMI Man Com PIN");
END_REGION
END_FUNCTION

FUNCTION "Ciclo_Aut" : Void   // FC2, LAD
{ S7_Optimized_Access := 'TRUE' }
VERSION : 0.1
   VAR_TEMP   // added for the SCL form of the ladder/FBD networks
      _w1 : Bool;
      _w2 : Bool;
   END_VAR
BEGIN

REGION Network 1
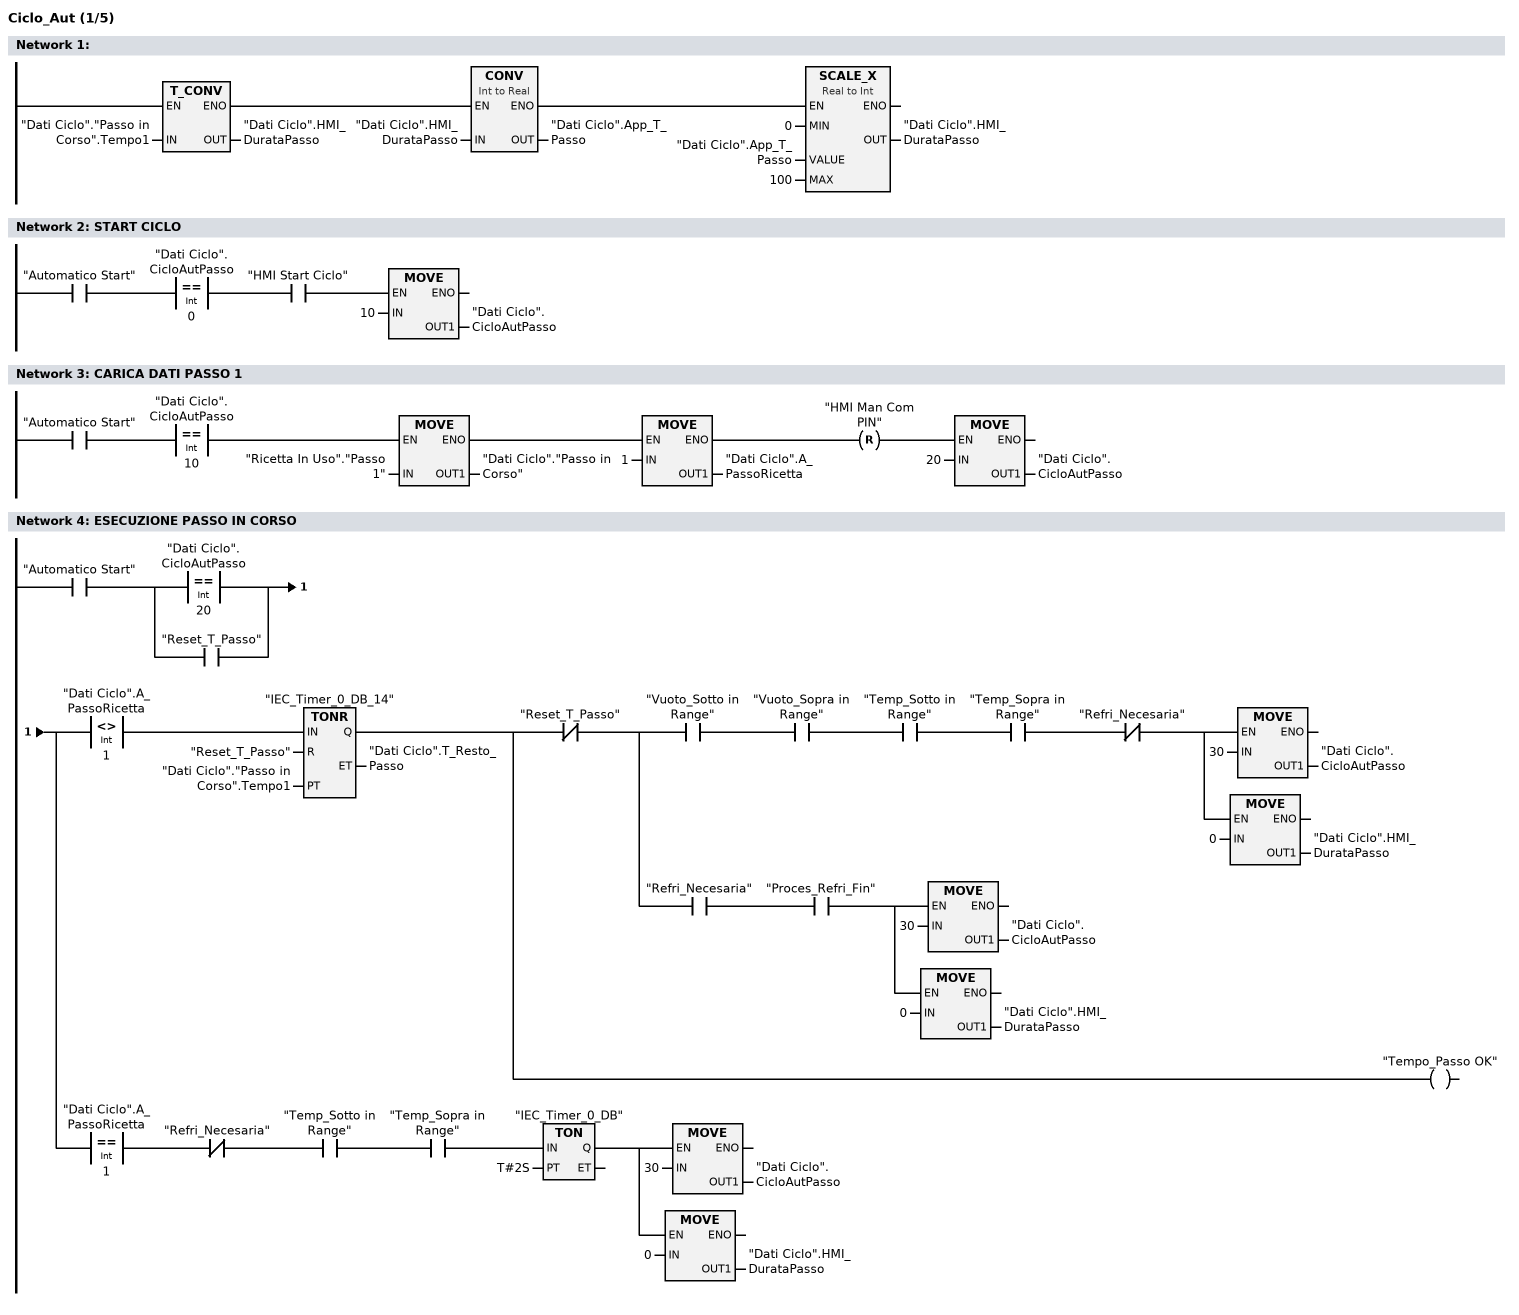
   // ENO of a box is taken as its EN; it also drops when the box reports an error
   "Dati Ciclo".HMI_DurataPasso := T_CONV(IN := "Dati Ciclo"."Passo in Corso".Tempo1);
   "Dati Ciclo".App_T_Passo := INT_TO_REAL("Dati Ciclo".HMI_DurataPasso);
   "Dati Ciclo".HMI_DurataPasso := SCALE_X(MIN := 0, VALUE := "Dati Ciclo".App_T_Passo, MAX := 100);
END_REGION

REGION Network 2: START CICLO
   RUNG wire#powerrail
      Contact( "Automatico Start" )
      { S7_Templates := "SrcType := Int" } EQ_Contact(in1 := "Dati Ciclo".CicloAutPasso, in2 := 0)
      Contact( "HMI Start Ciclo" )
      Move(in := 10, out1 => "Dati Ciclo".CicloAutPasso)
   END_RUNG
   // the same network as SCL:
   IF "Automatico Start" AND ("Dati Ciclo".CicloAutPasso = 0) AND "HMI Start Ciclo" THEN
       "Dati Ciclo".CicloAutPasso := 10;
   END_IF;
END_REGION

REGION Network 3: CARICA DATI PASSO 1
   RUNG wire#powerrail
      Contact( "Automatico Start" )
      { S7_Templates := "SrcType := Int" } EQ_Contact(in1 := "Dati Ciclo".CicloAutPasso, in2 := 10)
      Move(in := "Ricetta In Uso"."Passo 1", out1 => "Dati Ciclo"."Passo in Corso")
      Move(in := 1, out1 => "Dati Ciclo".A_PassoRicetta)
      R_Coil( "HMI Man Com PIN" )
      Move(in := 20, out1 => "Dati Ciclo".CicloAutPasso)
   END_RUNG
   // the same network as SCL:
   IF "Automatico Start" AND ("Dati Ciclo".CicloAutPasso = 10) THEN
       "Dati Ciclo"."Passo in Corso" := "Ricetta In Uso"."Passo 1";
       "Dati Ciclo".A_PassoRicetta := 1;
       "HMI Man Com PIN" := FALSE;
       "Dati Ciclo".CicloAutPasso := 20;
   END_IF;
END_REGION

REGION Network 4: ESECUZIONE PASSO IN CORSO
   #_w1 := "Automatico Start" AND (("Dati Ciclo".CicloAutPasso = 20) OR "Reset_T_Passo");
   "IEC_Timer_0_DB_14".TONR(IN := #_w1 AND ("Dati Ciclo".A_PassoRicetta <> 1),
                           R := "Reset_T_Passo",
                           PT := "Dati Ciclo"."Passo in Corso".Tempo1,
                           ET => "Dati Ciclo".T_Resto_Passo);
   #_w2 := "IEC_Timer_0_DB_14".Q AND NOT "Reset_T_Passo";
   IF #_w2 AND "Vuoto_Sotto in Range" AND "Vuoto_Sopra in Range" AND "Temp_Sotto in Range" AND "Temp_Sopra in Range" AND NOT "Refri_Necesaria" THEN
       "Dati Ciclo".CicloAutPasso := 30;
       "Dati Ciclo".HMI_DurataPasso := 0;
   END_IF;
   IF #_w2 AND "Refri_Necesaria" AND "Proces_Refri_Fin" THEN
       "Dati Ciclo".CicloAutPasso := 30;
       "Dati Ciclo".HMI_DurataPasso := 0;
   END_IF;
   "Tempo_Passo OK" := "IEC_Timer_0_DB_14".Q;
   "IEC_Timer_0_DB".TON(IN := #_w1 AND ("Dati Ciclo".A_PassoRicetta = 1) AND NOT "Refri_Necesaria" AND "Temp_Sotto in Range" AND "Temp_Sopra in Range",
                        PT := T#2S);
   IF "IEC_Timer_0_DB".Q THEN
       "Dati Ciclo".CicloAutPasso := 30;
       "Dati Ciclo".HMI_DurataPasso := 0;
   END_IF;
END_REGION

REGION Network 5: PIN IN AUTOMATICO + SALTA PASSO
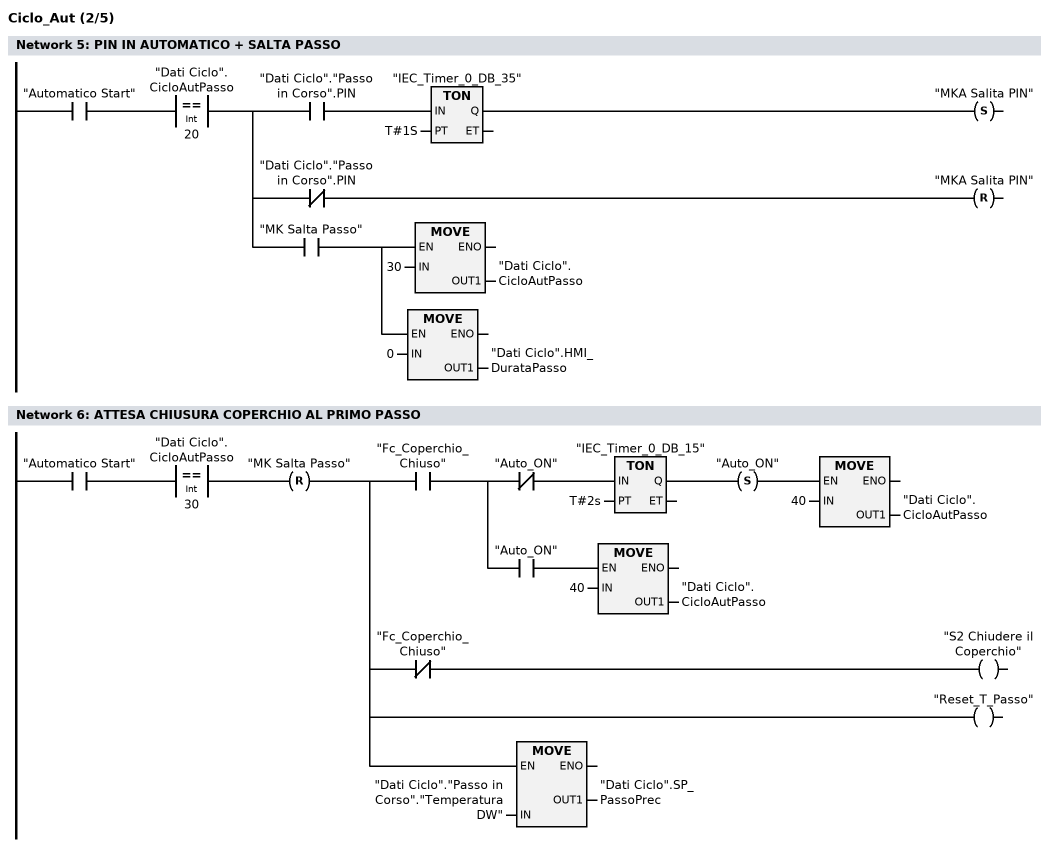
   #_w1 := "Automatico Start" AND ("Dati Ciclo".CicloAutPasso = 20);
   "IEC_Timer_0_DB_35".TON(IN := #_w1 AND "Dati Ciclo"."Passo in Corso".PIN, PT := T#1S);
   IF "IEC_Timer_0_DB_35".Q THEN "MKA Salita PIN" := TRUE; END_IF;
   IF #_w1 AND NOT "Dati Ciclo"."Passo in Corso".PIN THEN "MKA Salita PIN" := FALSE; END_IF;
   IF #_w1 AND "MK Salta Passo" THEN
       "Dati Ciclo".CicloAutPasso := 30;
       "Dati Ciclo".HMI_DurataPasso := 0;
   END_IF;
END_REGION

REGION Network 6: ATTESA CHIUSURA COPERCHIO AL PRIMO PASSO
   #_w1 := "Automatico Start" AND ("Dati Ciclo".CicloAutPasso = 30);
   IF #_w1 THEN "MK Salta Passo" := FALSE; END_IF;
   #_w2 := #_w1 AND "Fc_Coperchio_Chiuso";
   "IEC_Timer_0_DB_15".TON(IN := #_w2 AND NOT "Auto_ON", PT := T#2s);
   IF "IEC_Timer_0_DB_15".Q THEN
       "Auto_ON" := TRUE;
       "Dati Ciclo".CicloAutPasso := 40;
   END_IF;
   IF #_w2 AND "Auto_ON" THEN "Dati Ciclo".CicloAutPasso := 40; END_IF;
   "S2 Chiudere il Coperchio" := #_w1 AND NOT "Fc_Coperchio_Chiuso";
   "Reset_T_Passo" := #_w1;
   IF #_w1 THEN "Dati Ciclo".SP_PassoPrec := "Dati Ciclo"."Passo in Corso"."Temperatura DW"; END_IF;
END_REGION

REGION Network 7: CARICA DATI PASSO SUCCESSIVO
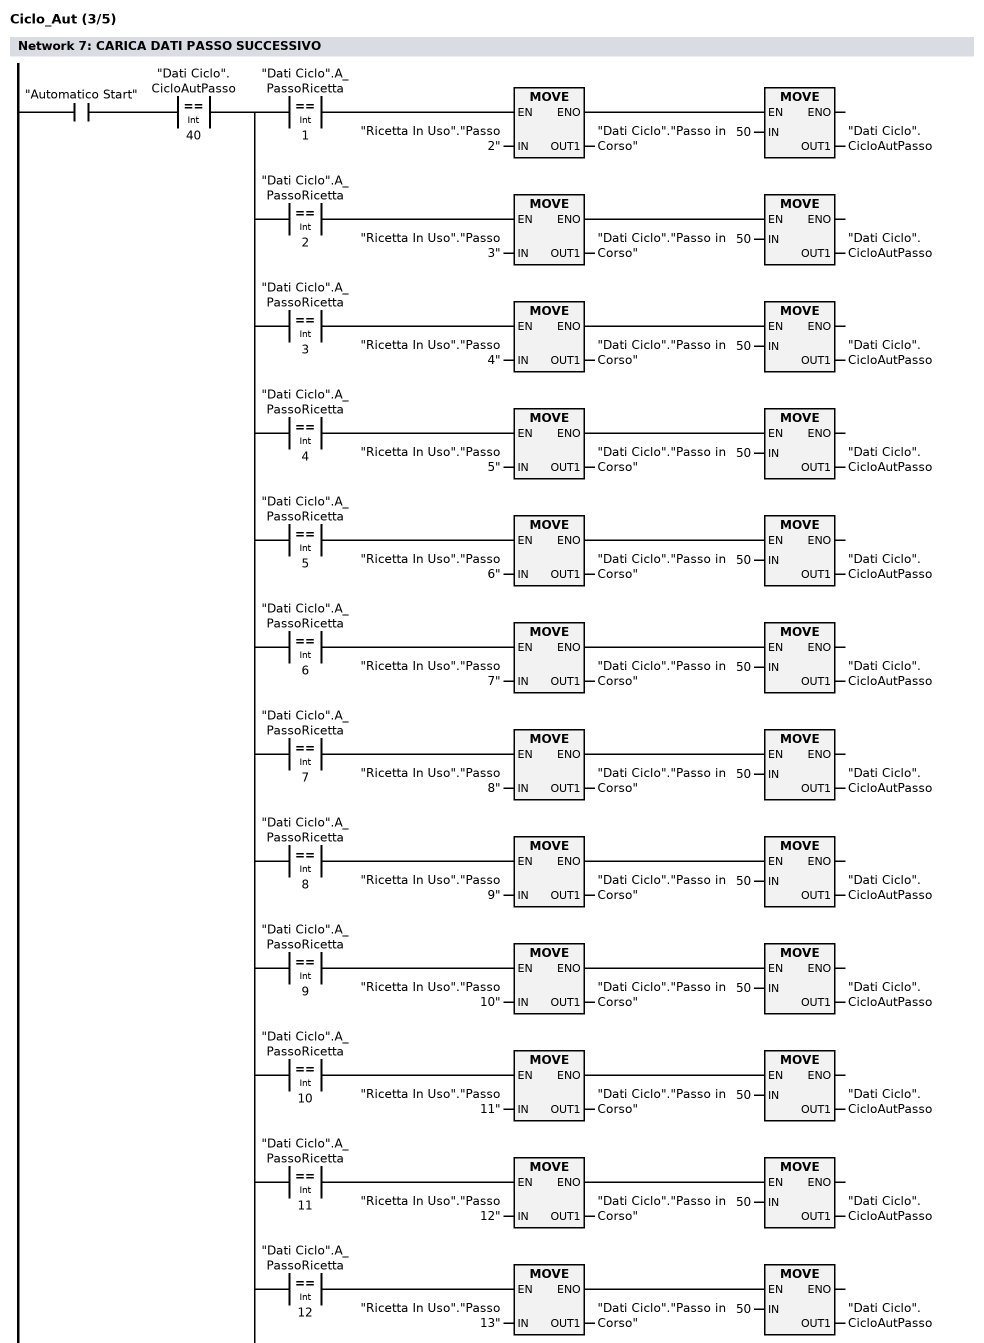
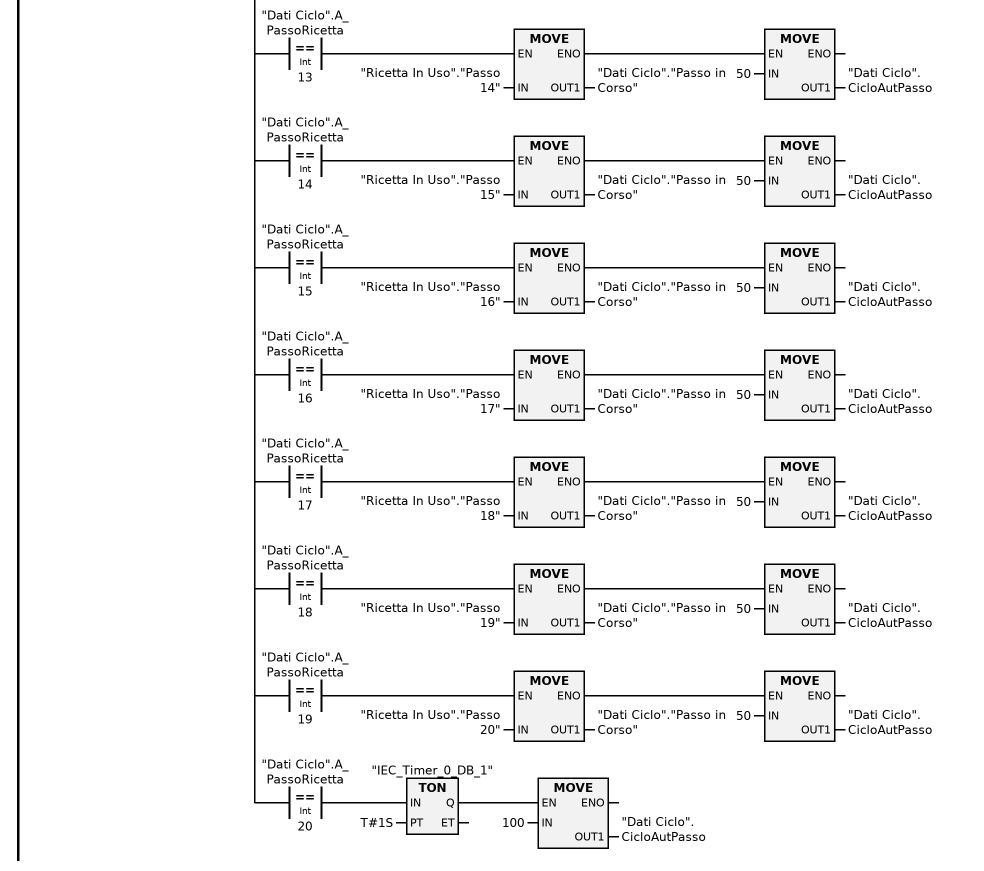
   #_w1 := "Automatico Start" AND ("Dati Ciclo".CicloAutPasso = 40);
   IF #_w1 AND ("Dati Ciclo".A_PassoRicetta = 1) THEN
       "Dati Ciclo"."Passo in Corso" := "Ricetta In Uso"."Passo 2";
       "Dati Ciclo".CicloAutPasso := 50;
   END_IF;
   IF #_w1 AND ("Dati Ciclo".A_PassoRicetta = 2) THEN
       "Dati Ciclo"."Passo in Corso" := "Ricetta In Uso"."Passo 3";
       "Dati Ciclo".CicloAutPasso := 50;
   END_IF;
   IF #_w1 AND ("Dati Ciclo".A_PassoRicetta = 3) THEN
       "Dati Ciclo"."Passo in Corso" := "Ricetta In Uso"."Passo 4";
       "Dati Ciclo".CicloAutPasso := 50;
   END_IF;
   IF #_w1 AND ("Dati Ciclo".A_PassoRicetta = 4) THEN
       "Dati Ciclo"."Passo in Corso" := "Ricetta In Uso"."Passo 5";
       "Dati Ciclo".CicloAutPasso := 50;
   END_IF;
   IF #_w1 AND ("Dati Ciclo".A_PassoRicetta = 5) THEN
       "Dati Ciclo"."Passo in Corso" := "Ricetta In Uso"."Passo 6";
       "Dati Ciclo".CicloAutPasso := 50;
   END_IF;
   IF #_w1 AND ("Dati Ciclo".A_PassoRicetta = 6) THEN
       "Dati Ciclo"."Passo in Corso" := "Ricetta In Uso"."Passo 7";
       "Dati Ciclo".CicloAutPasso := 50;
   END_IF;
   IF #_w1 AND ("Dati Ciclo".A_PassoRicetta = 7) THEN
       "Dati Ciclo"."Passo in Corso" := "Ricetta In Uso"."Passo 8";
       "Dati Ciclo".CicloAutPasso := 50;
   END_IF;
   IF #_w1 AND ("Dati Ciclo".A_PassoRicetta = 8) THEN
       "Dati Ciclo"."Passo in Corso" := "Ricetta In Uso"."Passo 9";
       "Dati Ciclo".CicloAutPasso := 50;
   END_IF;
   IF #_w1 AND ("Dati Ciclo".A_PassoRicetta = 9) THEN
       "Dati Ciclo"."Passo in Corso" := "Ricetta In Uso"."Passo 10";
       "Dati Ciclo".CicloAutPasso := 50;
   END_IF;
   IF #_w1 AND ("Dati Ciclo".A_PassoRicetta = 10) THEN
       "Dati Ciclo"."Passo in Corso" := "Ricetta In Uso"."Passo 11";
       "Dati Ciclo".CicloAutPasso := 50;
   END_IF;
   IF #_w1 AND ("Dati Ciclo".A_PassoRicetta = 11) THEN
       "Dati Ciclo"."Passo in Corso" := "Ricetta In Uso"."Passo 12";
       "Dati Ciclo".CicloAutPasso := 50;
   END_IF;
   IF #_w1 AND ("Dati Ciclo".A_PassoRicetta = 12) THEN
       "Dati Ciclo"."Passo in Corso" := "Ricetta In Uso"."Passo 13";
       "Dati Ciclo".CicloAutPasso := 50;
   END_IF;
   IF #_w1 AND ("Dati Ciclo".A_PassoRicetta = 13) THEN
       "Dati Ciclo"."Passo in Corso" := "Ricetta In Uso"."Passo 14";
       "Dati Ciclo".CicloAutPasso := 50;
   END_IF;
   IF #_w1 AND ("Dati Ciclo".A_PassoRicetta = 14) THEN
       "Dati Ciclo"."Passo in Corso" := "Ricetta In Uso"."Passo 15";
       "Dati Ciclo".CicloAutPasso := 50;
   END_IF;
   IF #_w1 AND ("Dati Ciclo".A_PassoRicetta = 15) THEN
       "Dati Ciclo"."Passo in Corso" := "Ricetta In Uso"."Passo 16";
       "Dati Ciclo".CicloAutPasso := 50;
   END_IF;
   IF #_w1 AND ("Dati Ciclo".A_PassoRicetta = 16) THEN
       "Dati Ciclo"."Passo in Corso" := "Ricetta In Uso"."Passo 17";
       "Dati Ciclo".CicloAutPasso := 50;
   END_IF;
   IF #_w1 AND ("Dati Ciclo".A_PassoRicetta = 17) THEN
       "Dati Ciclo"."Passo in Corso" := "Ricetta In Uso"."Passo 18";
       "Dati Ciclo".CicloAutPasso := 50;
   END_IF;
   IF #_w1 AND ("Dati Ciclo".A_PassoRicetta = 18) THEN
       "Dati Ciclo"."Passo in Corso" := "Ricetta In Uso"."Passo 19";
       "Dati Ciclo".CicloAutPasso := 50;
   END_IF;
   IF #_w1 AND ("Dati Ciclo".A_PassoRicetta = 19) THEN
       "Dati Ciclo"."Passo in Corso" := "Ricetta In Uso"."Passo 20";
       "Dati Ciclo".CicloAutPasso := 50;
   END_IF;
   "IEC_Timer_0_DB_1".TON(IN := #_w1 AND ("Dati Ciclo".A_PassoRicetta = 20), PT := T#1S);
   IF "IEC_Timer_0_DB_1".Q THEN "Dati Ciclo".CicloAutPasso := 100; END_IF;
END_REGION

REGION Network 8: SOMMA POSSO RICETTA
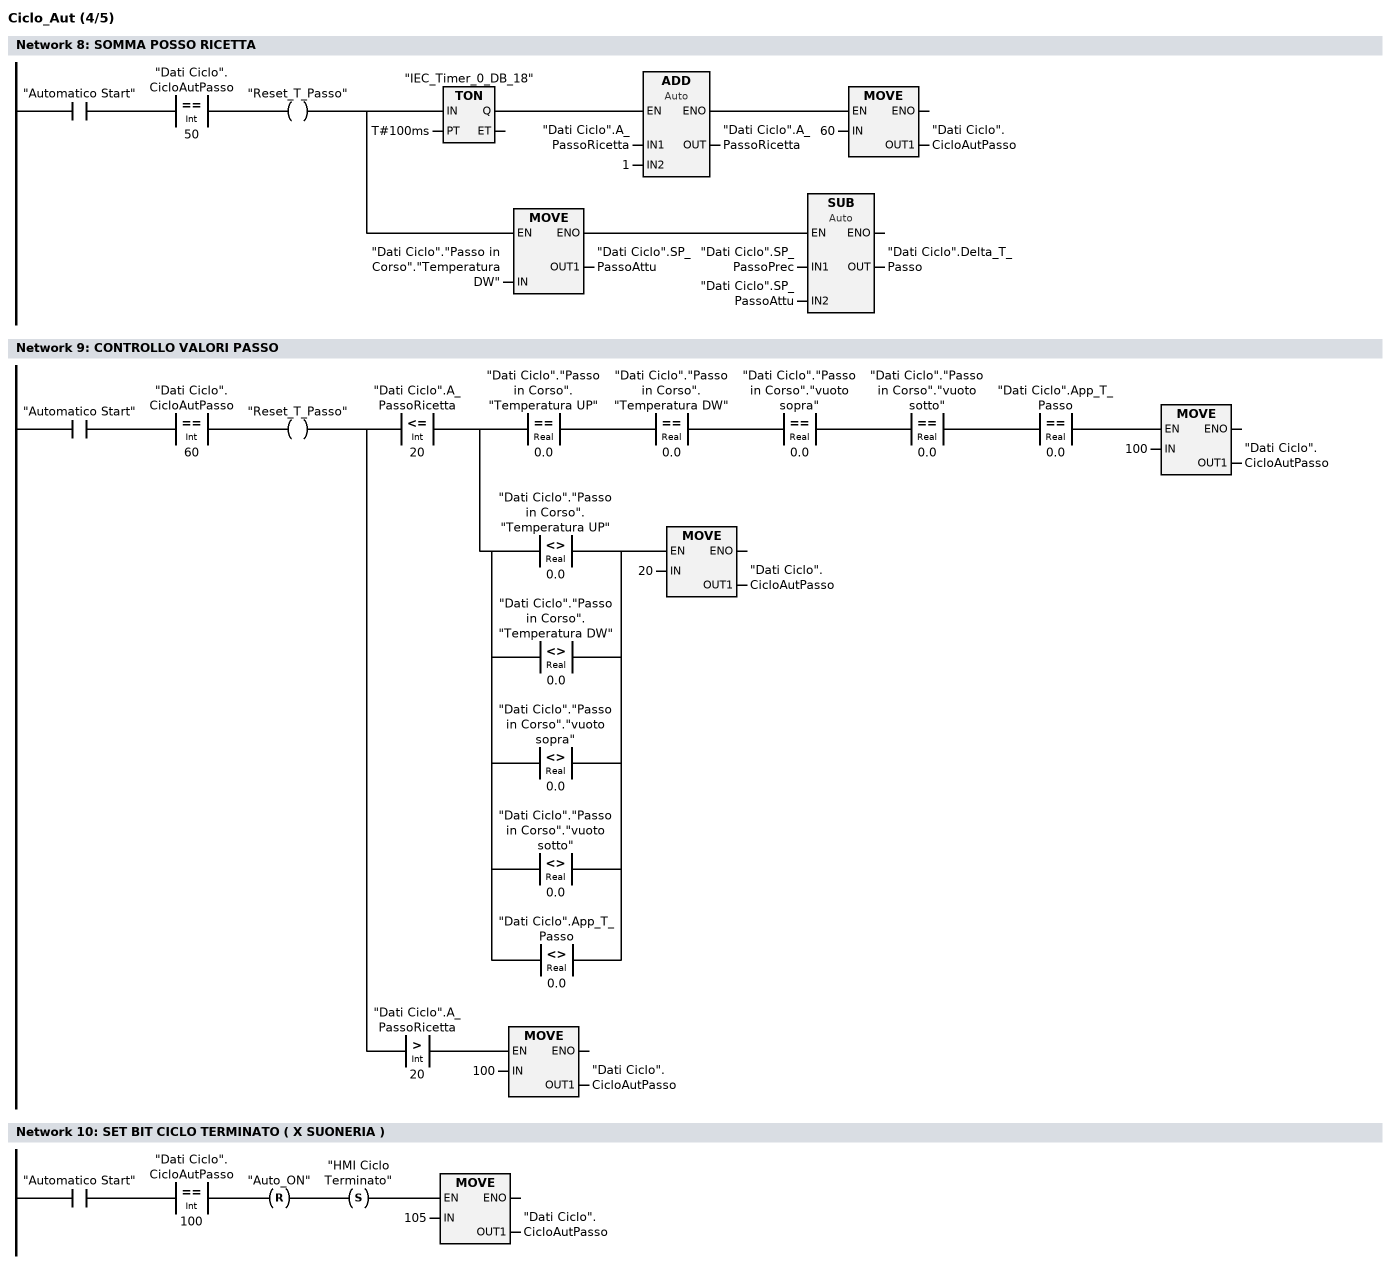
   "Reset_T_Passo" := "Automatico Start" AND ("Dati Ciclo".CicloAutPasso = 50);
   "IEC_Timer_0_DB_18".TON(IN := "Reset_T_Passo", PT := T#100ms);
   IF "IEC_Timer_0_DB_18".Q THEN
       "Dati Ciclo".A_PassoRicetta := "Dati Ciclo".A_PassoRicetta + 1;
       "Dati Ciclo".CicloAutPasso := 60;
   END_IF;
   IF "Reset_T_Passo" THEN
       "Dati Ciclo".SP_PassoAttu := "Dati Ciclo"."Passo in Corso"."Temperatura DW";
       "Dati Ciclo".Delta_T_Passo := "Dati Ciclo".SP_PassoPrec - "Dati Ciclo".SP_PassoAttu;
   END_IF;
END_REGION

REGION Network 9: CONTROLLO VALORI PASSO
   RUNG wire#powerrail
      Contact( "Automatico Start" )
      { S7_Templates := "SrcType := Int" } EQ_Contact(in1 := "Dati Ciclo".CicloAutPasso, in2 := 60)
      Coil( "Reset_T_Passo" )
      wire#w1
      { S7_Templates := "SrcType := Int" } LE_Contact(in1 := "Dati Ciclo".A_PassoRicetta, in2 := 20)
      wire#w2
      { S7_Templates := "SrcType := Real" } EQ_Contact(in1 := "Dati Ciclo"."Passo in Corso"."Temperatura UP", in2 := 0.0)
      { S7_Templates := "SrcType := Real" } EQ_Contact(in1 := "Dati Ciclo"."Passo in Corso"."Temperatura DW", in2 := 0.0)
      { S7_Templates := "SrcType := Real" } EQ_Contact(in1 := "Dati Ciclo"."Passo in Corso"."vuoto sopra", in2 := 0.0)
      { S7_Templates := "SrcType := Real" } EQ_Contact(in1 := "Dati Ciclo"."Passo in Corso"."vuoto sotto", in2 := 0.0)
      { S7_Templates := "SrcType := Real" } EQ_Contact(in1 := "Dati Ciclo".App_T_Passo, in2 := 0.0)
      Move(in := 100, out1 => "Dati Ciclo".CicloAutPasso)
   END_RUNG
   RUNG wire#w2
      { S7_Templates := "SrcType := Real" } NE_Contact(in1 := "Dati Ciclo"."Passo in Corso"."Temperatura UP", in2 := 0.0)
      wire#w3
      Move(in := 20, out1 => "Dati Ciclo".CicloAutPasso)
   END_RUNG
   RUNG wire#w2
      { S7_Templates := "SrcType := Real" } NE_Contact(in1 := "Dati Ciclo"."Passo in Corso"."Temperatura DW", in2 := 0.0)
   END_RUNG wire#w3
   RUNG wire#w2
      { S7_Templates := "SrcType := Real" } NE_Contact(in1 := "Dati Ciclo"."Passo in Corso"."vuoto sopra", in2 := 0.0)
   END_RUNG wire#w3
   RUNG wire#w2
      { S7_Templates := "SrcType := Real" } NE_Contact(in1 := "Dati Ciclo"."Passo in Corso"."vuoto sotto", in2 := 0.0)
   END_RUNG wire#w3
   RUNG wire#w2
      { S7_Templates := "SrcType := Real" } NE_Contact(in1 := "Dati Ciclo".App_T_Passo, in2 := 0.0)
   END_RUNG wire#w3
   RUNG wire#w1
      { S7_Templates := "SrcType := Int" } GT_Contact(in1 := "Dati Ciclo".A_PassoRicetta, in2 := 20)
      Move(in := 100, out1 => "Dati Ciclo".CicloAutPasso)
   END_RUNG
   // the same network as SCL:
   "Reset_T_Passo" := "Automatico Start" AND ("Dati Ciclo".CicloAutPasso = 60);
   #_w1 := "Reset_T_Passo" AND ("Dati Ciclo".A_PassoRicetta <= 20);
   IF #_w1 AND ("Dati Ciclo"."Passo in Corso"."Temperatura UP" = 0.0) AND ("Dati Ciclo"."Passo in Corso"."Temperatura DW" = 0.0) AND ("Dati Ciclo"."Passo in Corso"."vuoto sopra" = 0.0) AND ("Dati Ciclo"."Passo in Corso"."vuoto sotto" = 0.0) AND ("Dati Ciclo".App_T_Passo = 0.0) THEN
       "Dati Ciclo".CicloAutPasso := 100;
   END_IF;
   IF #_w1 AND (("Dati Ciclo"."Passo in Corso"."Temperatura UP" <> 0.0) OR ("Dati Ciclo"."Passo in Corso"."Temperatura DW" <> 0.0) OR ("Dati Ciclo"."Passo in Corso"."vuoto sopra" <> 0.0) OR ("Dati Ciclo"."Passo in Corso"."vuoto sotto" <> 0.0) OR ("Dati Ciclo".App_T_Passo <> 0.0)) THEN
       "Dati Ciclo".CicloAutPasso := 20;
   END_IF;
   IF "Reset_T_Passo" AND ("Dati Ciclo".A_PassoRicetta > 20) THEN "Dati Ciclo".CicloAutPasso := 100; END_IF;
END_REGION

REGION Network 10: SET BIT CICLO TERMINATO ( X SUONERIA )
   RUNG wire#powerrail
      Contact( "Automatico Start" )
      { S7_Templates := "SrcType := Int" } EQ_Contact(in1 := "Dati Ciclo".CicloAutPasso, in2 := 100)
      R_Coil( "Auto_ON" )
      S_Coil( "HMI Ciclo Terminato" )
      Move(in := 105, out1 => "Dati Ciclo".CicloAutPasso)
   END_RUNG
   // the same network as SCL:
   IF "Automatico Start" AND ("Dati Ciclo".CicloAutPasso = 100) THEN
       "Auto_ON" := FALSE;
       "HMI Ciclo Terminato" := TRUE;
       "Dati Ciclo".CicloAutPasso := 105;
   END_IF;
END_REGION

REGION Network 11
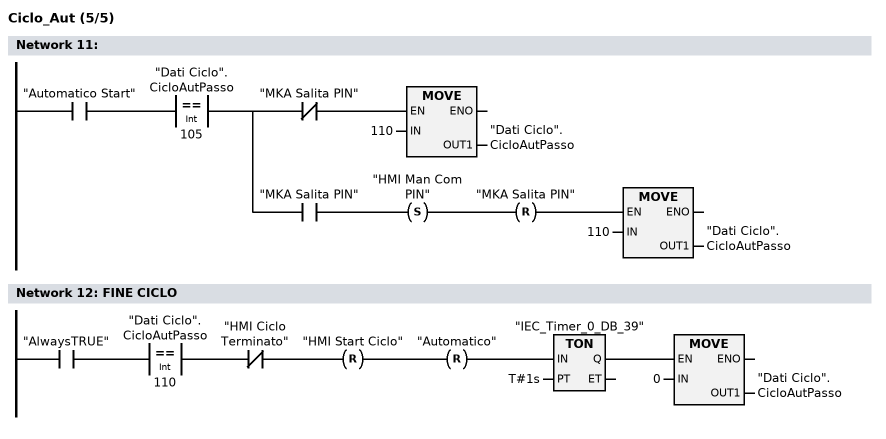
   RUNG wire#powerrail
      Contact( "Automatico Start" )
      { S7_Templates := "SrcType := Int" } EQ_Contact(in1 := "Dati Ciclo".CicloAutPasso, in2 := 105)
      wire#w1
      I_Contact( "MKA Salita PIN" )
      Move(in := 110, out1 => "Dati Ciclo".CicloAutPasso)
   END_RUNG
   RUNG wire#w1
      Contact( "MKA Salita PIN" )
      S_Coil( "HMI Man Com PIN" )
      R_Coil( "MKA Salita PIN" )
      Move(in := 110, out1 => "Dati Ciclo".CicloAutPasso)
   END_RUNG
   // the same network as SCL:
   #_w1 := "Automatico Start" AND ("Dati Ciclo".CicloAutPasso = 105);
   IF #_w1 AND NOT "MKA Salita PIN" THEN "Dati Ciclo".CicloAutPasso := 110; END_IF;
   IF #_w1 AND "MKA Salita PIN" THEN "HMI Man Com PIN" := TRUE; END_IF;
   #_w2 := #_w1 AND "MKA Salita PIN";
   IF #_w2 THEN
       "MKA Salita PIN" := FALSE;
       "Dati Ciclo".CicloAutPasso := 110;
   END_IF;
END_REGION

REGION Network 12: FINE CICLO
   #_w1 := "AlwaysTRUE" AND ("Dati Ciclo".CicloAutPasso = 110) AND NOT "HMI Ciclo Terminato";
   IF #_w1 THEN
       "HMI Start Ciclo" := FALSE;
       "Automatico" := FALSE;
   END_IF;
   "IEC_Timer_0_DB_39".TON(IN := #_w1, PT := T#1s);
   IF "IEC_Timer_0_DB_39".Q THEN "Dati Ciclo".CicloAutPasso := 0; END_IF;
END_REGION
END_FUNCTION

FUNCTION "Generale" : Void   // FC3, LAD
{ S7_Optimized_Access := 'TRUE' }
VERSION : 0.1
   VAR_TEMP   // added for the SCL form of the ladder/FBD networks
      _w1 : Bool;
   END_VAR
BEGIN

REGION Network 1: CONDICIONE DI MANUALE
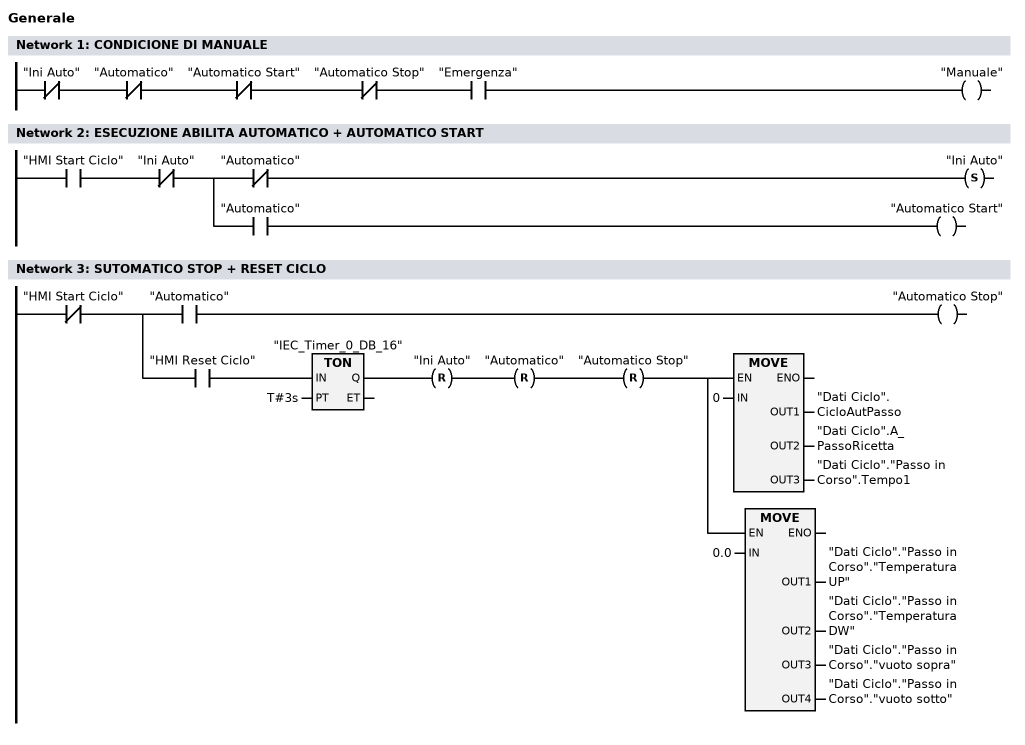
   RUNG wire#powerrail
      I_Contact( "Ini Auto" )
      I_Contact( "Automatico" )
      I_Contact( "Automatico Start" )
      I_Contact( "Automatico Stop" )
      Contact( "Emergenza" )
      Coil( "Manuale" )
   END_RUNG
   // the same network as SCL:
   "Manuale" := NOT "Ini Auto" AND NOT "Automatico" AND NOT "Automatico Start" AND NOT "Automatico Stop" AND "Emergenza";
END_REGION

REGION Network 2: ESECUZIONE ABILITA AUTOMATICO + AUTOMATICO START
   RUNG wire#powerrail
      Contact( "HMI Start Ciclo" )
      I_Contact( "Ini Auto" )
      wire#w1
      I_Contact( "Automatico" )
      S_Coil( "Ini Auto" )
   END_RUNG
   RUNG wire#w1
      Contact( "Automatico" )
      Coil( "Automatico Start" )
   END_RUNG
   // the same network as SCL:
   #_w1 := "HMI Start Ciclo" AND NOT "Ini Auto";
   IF #_w1 AND NOT "Automatico" THEN "Ini Auto" := TRUE; END_IF;
   "Automatico Start" := #_w1 AND "Automatico";
END_REGION

REGION Network 3: SUTOMATICO STOP + RESET CICLO
   "Automatico Stop" := NOT "HMI Start Ciclo" AND "Automatico";
   "IEC_Timer_0_DB_16".TON(IN := NOT "HMI Start Ciclo" AND "HMI Reset Ciclo", PT := T#3s);
   IF "IEC_Timer_0_DB_16".Q THEN
       "Ini Auto" := FALSE;
       "Automatico" := FALSE;
       "Automatico Stop" := FALSE;
       "Dati Ciclo".CicloAutPasso := 0;
       "Dati Ciclo".A_PassoRicetta := 0;
       "Dati Ciclo"."Passo in Corso".Tempo1 := 0;
       "Dati Ciclo"."Passo in Corso"."Temperatura UP" := 0.0;
       "Dati Ciclo"."Passo in Corso"."Temperatura DW" := 0.0;
       "Dati Ciclo"."Passo in Corso"."vuoto sopra" := 0.0;
       "Dati Ciclo"."Passo in Corso"."vuoto sotto" := 0.0;
   END_IF;
END_REGION
END_FUNCTION

FUNCTION "Ab Auto" : Void   // FC4, LAD
{ S7_Optimized_Access := 'TRUE' }
VERSION : 0.1
BEGIN

REGION Network 1: START ABILITA AUTO CON RESET MANUALI
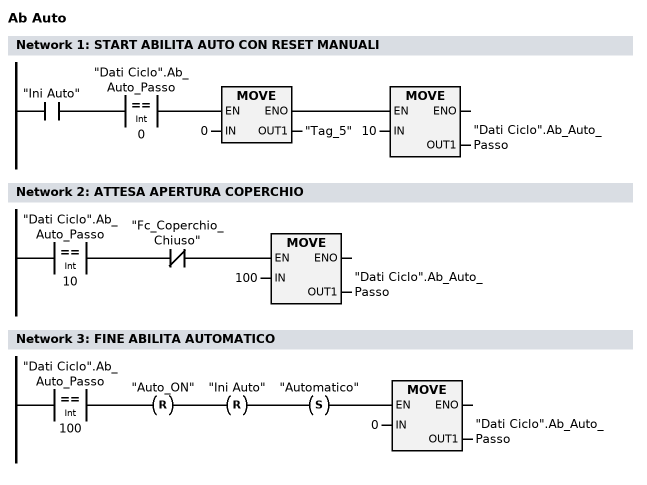
   RUNG wire#powerrail
      Contact( "Ini Auto" )
      { S7_Templates := "SrcType := Int" } EQ_Contact(in1 := "Dati Ciclo".Ab_Auto_Passo, in2 := 0)
      Move(in := 0, out1 => "Tag_5")
      Move(in := 10, out1 => "Dati Ciclo".Ab_Auto_Passo)
   END_RUNG
   // the same network as SCL:
   IF "Ini Auto" AND ("Dati Ciclo".Ab_Auto_Passo = 0) THEN
       "Tag_5" := 0;
       "Dati Ciclo".Ab_Auto_Passo := 10;
   END_IF;
END_REGION

REGION Network 2: ATTESA APERTURA COPERCHIO
   RUNG wire#powerrail
      { S7_Templates := "SrcType := Int" } EQ_Contact(in1 := "Dati Ciclo".Ab_Auto_Passo, in2 := 10)
      I_Contact( "Fc_Coperchio_Chiuso" )
      Move(in := 100, out1 => "Dati Ciclo".Ab_Auto_Passo)
   END_RUNG
   // the same network as SCL:
   IF ("Dati Ciclo".Ab_Auto_Passo = 10) AND NOT "Fc_Coperchio_Chiuso" THEN
       "Dati Ciclo".Ab_Auto_Passo := 100;
   END_IF;
END_REGION

REGION Network 3: FINE ABILITA AUTOMATICO
   RUNG wire#powerrail
      { S7_Templates := "SrcType := Int" } EQ_Contact(in1 := "Dati Ciclo".Ab_Auto_Passo, in2 := 100)
      R_Coil( "Auto_ON" )
      R_Coil( "Ini Auto" )
      S_Coil( "Automatico" )
      Move(in := 0, out1 => "Dati Ciclo".Ab_Auto_Passo)
   END_RUNG
   // the same network as SCL:
   IF "Dati Ciclo".Ab_Auto_Passo = 100 THEN
       "Auto_ON" := FALSE;
       "Ini Auto" := FALSE;
       "Automatico" := TRUE;
       "Dati Ciclo".Ab_Auto_Passo := 0;
   END_IF;
END_REGION
END_FUNCTION

FUNCTION "Ausiliari" : Void   // FC5, LAD
{ S7_Optimized_Access := 'TRUE' }
VERSION : 0.1
   VAR_TEMP   // added for the SCL form of the ladder/FBD networks
      _w1 : Bool;
      _w2 : Bool;
      _w3 : Bool;
      _w4 : Bool;
      _w5 : Bool;
      _w6 : Bool;
      _w7 : Bool;
      _w8 : Bool;
      _w9 : Bool;
      _w10 : Bool;
      _w11 : Bool;
      _w12 : Bool;
      _w13 : Bool;
      _w14 : Bool;
      _w15 : Bool;
      _w16 : Bool;
      _w17 : Bool;
      _w18 : Bool;
      _w19 : Bool;
      _w20 : Bool;
      _w21 : Bool;
   END_VAR
BEGIN

REGION Network 1: VARIABILE STATO MACCHINA
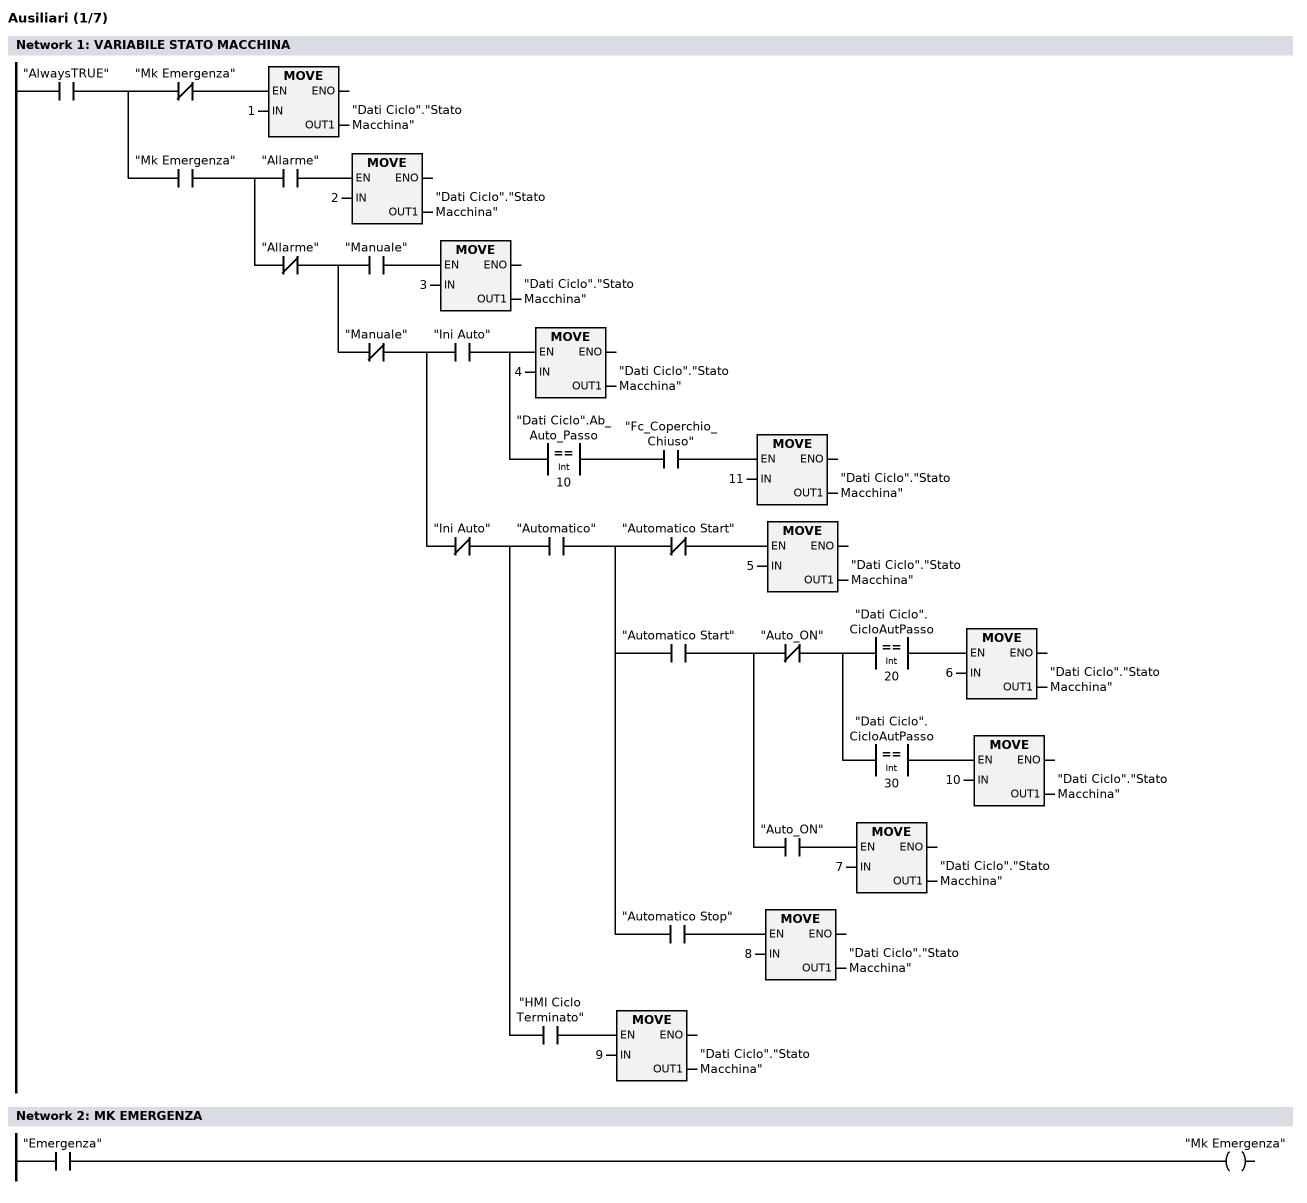
   RUNG wire#powerrail
      Contact( "AlwaysTRUE" )
      wire#w1
      I_Contact( "Mk Emergenza" )
      Move(in := 1, out1 => "Dati Ciclo"."Stato Macchina")
   END_RUNG
   RUNG wire#w1
      Contact( "Mk Emergenza" )
      wire#w2
      Contact( "Allarme" )
      Move(in := 2, out1 => "Dati Ciclo"."Stato Macchina")
   END_RUNG
   RUNG wire#w2
      I_Contact( "Allarme" )
      wire#w3
      Contact( "Manuale" )
      Move(in := 3, out1 => "Dati Ciclo"."Stato Macchina")
   END_RUNG
   RUNG wire#w3
      I_Contact( "Manuale" )
      wire#w4
      Contact( "Ini Auto" )
      wire#w5
      Move(in := 4, out1 => "Dati Ciclo"."Stato Macchina")
   END_RUNG
   RUNG wire#w5
      { S7_Templates := "SrcType := Int" } EQ_Contact(in1 := "Dati Ciclo".Ab_Auto_Passo, in2 := 10)
      Contact( "Fc_Coperchio_Chiuso" )
      Move(in := 11, out1 => "Dati Ciclo"."Stato Macchina")
   END_RUNG
   RUNG wire#w4
      I_Contact( "Ini Auto" )
      wire#w6
      Contact( "Automatico" )
      wire#w7
      I_Contact( "Automatico Start" )
      Move(in := 5, out1 => "Dati Ciclo"."Stato Macchina")
   END_RUNG
   RUNG wire#w7
      Contact( "Automatico Start" )
      wire#w8
      I_Contact( "Auto_ON" )
      wire#w9
      { S7_Templates := "SrcType := Int" } EQ_Contact(in1 := "Dati Ciclo".CicloAutPasso, in2 := 20)
      Move(in := 6, out1 => "Dati Ciclo"."Stato Macchina")
   END_RUNG
   RUNG wire#w9
      { S7_Templates := "SrcType := Int" } EQ_Contact(in1 := "Dati Ciclo".CicloAutPasso, in2 := 30)
      Move(in := 10, out1 => "Dati Ciclo"."Stato Macchina")
   END_RUNG
   RUNG wire#w8
      Contact( "Auto_ON" )
      Move(in := 7, out1 => "Dati Ciclo"."Stato Macchina")
   END_RUNG
   RUNG wire#w7
      Contact( "Automatico Stop" )
      Move(in := 8, out1 => "Dati Ciclo"."Stato Macchina")
   END_RUNG
   RUNG wire#w6
      Contact( "HMI Ciclo Terminato" )
      Move(in := 9, out1 => "Dati Ciclo"."Stato Macchina")
   END_RUNG
   // the same network as SCL:
   IF "AlwaysTRUE" AND NOT "Mk Emergenza" THEN "Dati Ciclo"."Stato Macchina" := 1; END_IF;
   #_w1 := "AlwaysTRUE" AND "Mk Emergenza";
   IF #_w1 AND "Allarme" THEN "Dati Ciclo"."Stato Macchina" := 2; END_IF;
   #_w2 := #_w1 AND NOT "Allarme";
   IF #_w2 AND "Manuale" THEN "Dati Ciclo"."Stato Macchina" := 3; END_IF;
   #_w3 := #_w2 AND NOT "Manuale";
   #_w4 := #_w3 AND "Ini Auto";
   IF #_w4 THEN "Dati Ciclo"."Stato Macchina" := 4; END_IF;
   IF #_w4 AND ("Dati Ciclo".Ab_Auto_Passo = 10) AND "Fc_Coperchio_Chiuso" THEN
       "Dati Ciclo"."Stato Macchina" := 11;
   END_IF;
   #_w5 := #_w3 AND NOT "Ini Auto";
   #_w6 := #_w5 AND "Automatico";
   IF #_w6 AND NOT "Automatico Start" THEN "Dati Ciclo"."Stato Macchina" := 5; END_IF;
   #_w7 := #_w6 AND "Automatico Start";
   #_w8 := #_w7 AND NOT "Auto_ON";
   IF #_w8 AND ("Dati Ciclo".CicloAutPasso = 20) THEN "Dati Ciclo"."Stato Macchina" := 6; END_IF;
   IF #_w8 AND ("Dati Ciclo".CicloAutPasso = 30) THEN "Dati Ciclo"."Stato Macchina" := 10; END_IF;
   IF #_w7 AND "Auto_ON" THEN "Dati Ciclo"."Stato Macchina" := 7; END_IF;
   IF #_w6 AND "Automatico Stop" THEN "Dati Ciclo"."Stato Macchina" := 8; END_IF;
   IF #_w5 AND "HMI Ciclo Terminato" THEN "Dati Ciclo"."Stato Macchina" := 9; END_IF;
END_REGION

REGION Network 2: MK EMERGENZA
   RUNG wire#powerrail
      Contact( "Emergenza" )
      Coil( "Mk Emergenza" )
   END_RUNG
   // the same network as SCL:
   "Mk Emergenza" := "Emergenza";
END_REGION

REGION Network 3: REGISTRAZIONI TEMPERATURE
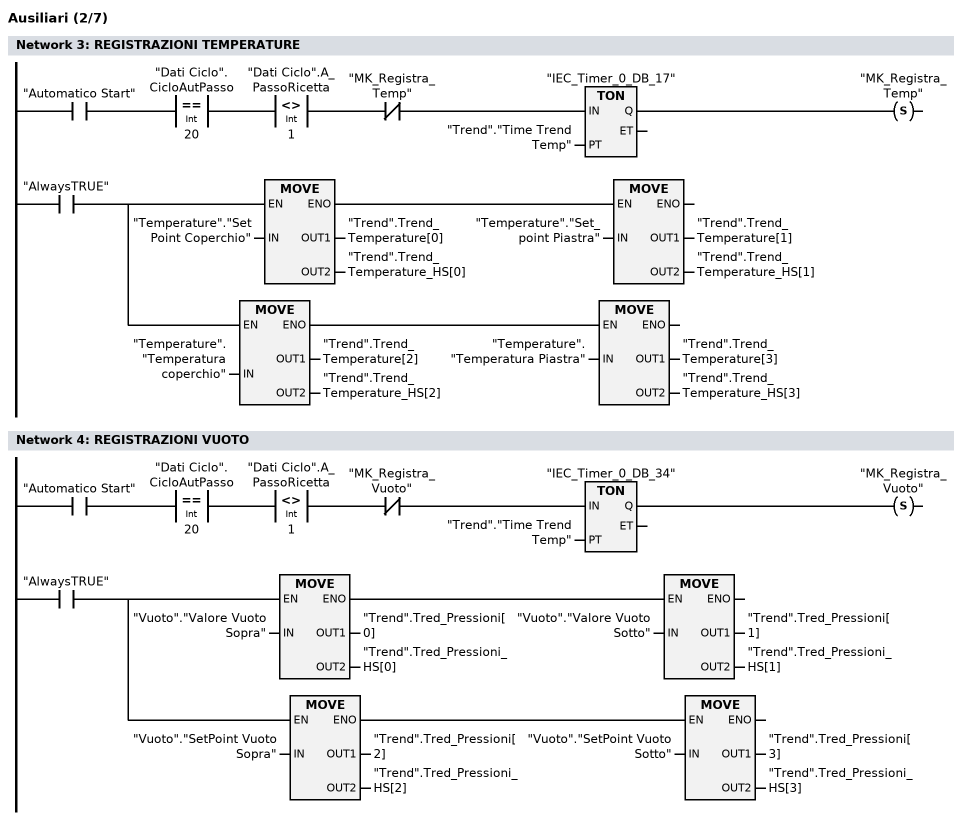
   "IEC_Timer_0_DB_17".TON(IN := "Automatico Start" AND ("Dati Ciclo".CicloAutPasso = 20) AND ("Dati Ciclo".A_PassoRicetta <> 1) AND NOT "MK_Registra_Temp",
                           PT := "Trend"."Time Trend Temp");
   IF "IEC_Timer_0_DB_17".Q THEN "MK_Registra_Temp" := TRUE; END_IF;
   IF "AlwaysTRUE" THEN
       "Trend".Trend_Temperature[0] := "Temperature"."Set Point Coperchio";
       "Trend".Trend_Temperature_HS[0] := "Temperature"."Set Point Coperchio";
       "Trend".Trend_Temperature[1] := "Temperature"."Set_point Piastra";
       "Trend".Trend_Temperature_HS[1] := "Temperature"."Set_point Piastra";
       "Trend".Trend_Temperature[2] := "Temperature"."Temperatura coperchio";
       "Trend".Trend_Temperature_HS[2] := "Temperature"."Temperatura coperchio";
       "Trend".Trend_Temperature[3] := "Temperature"."Temperatura Piastra";
       "Trend".Trend_Temperature_HS[3] := "Temperature"."Temperatura Piastra";
   END_IF;
END_REGION

REGION Network 4: REGISTRAZIONI VUOTO
   "IEC_Timer_0_DB_34".TON(IN := "Automatico Start" AND ("Dati Ciclo".CicloAutPasso = 20) AND ("Dati Ciclo".A_PassoRicetta <> 1) AND NOT "MK_Registra_Vuoto",
                           PT := "Trend"."Time Trend Temp");
   IF "IEC_Timer_0_DB_34".Q THEN "MK_Registra_Vuoto" := TRUE; END_IF;
   IF "AlwaysTRUE" THEN
       "Trend".Tred_Pressioni[0] := "Vuoto"."Valore Vuoto Sopra";
       "Trend".Tred_Pressioni_HS[0] := "Vuoto"."Valore Vuoto Sopra";
       "Trend".Tred_Pressioni[1] := "Vuoto"."Valore Vuoto Sotto";
       "Trend".Tred_Pressioni_HS[1] := "Vuoto"."Valore Vuoto Sotto";
       "Trend".Tred_Pressioni[2] := "Vuoto"."SetPoint Vuoto Sopra";
       "Trend".Tred_Pressioni_HS[2] := "Vuoto"."SetPoint Vuoto Sopra";
       "Trend".Tred_Pressioni[3] := "Vuoto"."SetPoint Vuoto Sotto";
       "Trend".Tred_Pressioni_HS[3] := "Vuoto"."SetPoint Vuoto Sotto";
   END_IF;
END_REGION

REGION Network 5: COPIA RICETTA
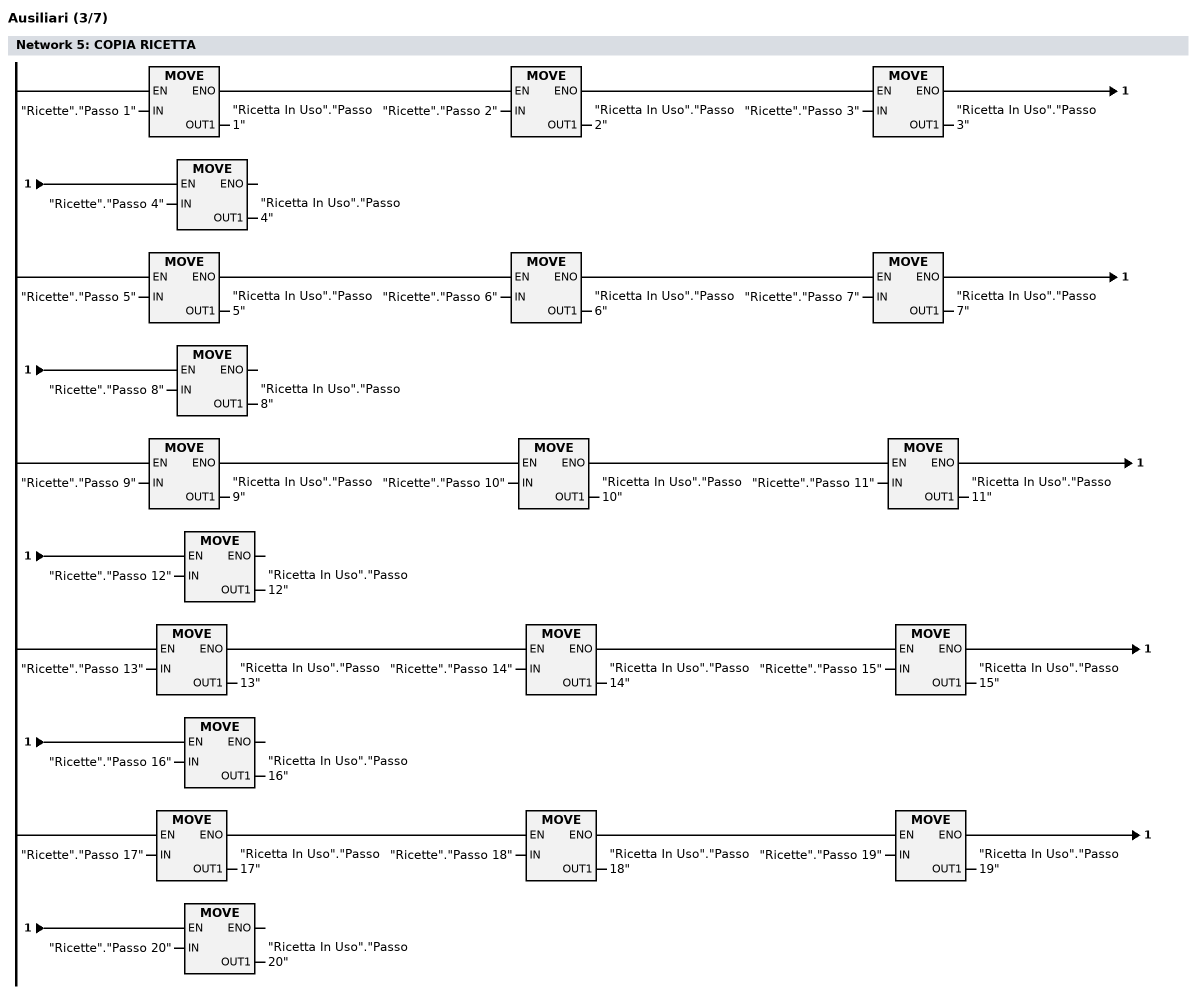
   RUNG wire#powerrail
      Move(in := "Ricette"."Passo 1", out1 => "Ricetta In Uso"."Passo 1")
      Move(in := "Ricette"."Passo 2", out1 => "Ricetta In Uso"."Passo 2")
      Move(in := "Ricette"."Passo 3", out1 => "Ricetta In Uso"."Passo 3")
      Move(in := "Ricette"."Passo 4", out1 => "Ricetta In Uso"."Passo 4")
   END_RUNG
   RUNG wire#powerrail
      Move(in := "Ricette"."Passo 5", out1 => "Ricetta In Uso"."Passo 5")
      Move(in := "Ricette"."Passo 6", out1 => "Ricetta In Uso"."Passo 6")
      Move(in := "Ricette"."Passo 7", out1 => "Ricetta In Uso"."Passo 7")
      Move(in := "Ricette"."Passo 8", out1 => "Ricetta In Uso"."Passo 8")
   END_RUNG
   RUNG wire#powerrail
      Move(in := "Ricette"."Passo 9", out1 => "Ricetta In Uso"."Passo 9")
      Move(in := "Ricette"."Passo 10", out1 => "Ricetta In Uso"."Passo 10")
      Move(in := "Ricette"."Passo 11", out1 => "Ricetta In Uso"."Passo 11")
      Move(in := "Ricette"."Passo 12", out1 => "Ricetta In Uso"."Passo 12")
   END_RUNG
   RUNG wire#powerrail
      Move(in := "Ricette"."Passo 13", out1 => "Ricetta In Uso"."Passo 13")
      Move(in := "Ricette"."Passo 14", out1 => "Ricetta In Uso"."Passo 14")
      Move(in := "Ricette"."Passo 15", out1 => "Ricetta In Uso"."Passo 15")
      Move(in := "Ricette"."Passo 16", out1 => "Ricetta In Uso"."Passo 16")
   END_RUNG
   RUNG wire#powerrail
      Move(in := "Ricette"."Passo 17", out1 => "Ricetta In Uso"."Passo 17")
      Move(in := "Ricette"."Passo 18", out1 => "Ricetta In Uso"."Passo 18")
      Move(in := "Ricette"."Passo 19", out1 => "Ricetta In Uso"."Passo 19")
      Move(in := "Ricette"."Passo 20", out1 => "Ricetta In Uso"."Passo 20")
   END_RUNG
   // the same network as SCL:
   "Ricetta In Uso"."Passo 1" := "Ricette"."Passo 1";
   "Ricetta In Uso"."Passo 2" := "Ricette"."Passo 2";
   "Ricetta In Uso"."Passo 3" := "Ricette"."Passo 3";
   "Ricetta In Uso"."Passo 4" := "Ricette"."Passo 4";
   "Ricetta In Uso"."Passo 5" := "Ricette"."Passo 5";
   "Ricetta In Uso"."Passo 6" := "Ricette"."Passo 6";
   "Ricetta In Uso"."Passo 7" := "Ricette"."Passo 7";
   "Ricetta In Uso"."Passo 8" := "Ricette"."Passo 8";
   "Ricetta In Uso"."Passo 9" := "Ricette"."Passo 9";
   "Ricetta In Uso"."Passo 10" := "Ricette"."Passo 10";
   "Ricetta In Uso"."Passo 11" := "Ricette"."Passo 11";
   "Ricetta In Uso"."Passo 12" := "Ricette"."Passo 12";
   "Ricetta In Uso"."Passo 13" := "Ricette"."Passo 13";
   "Ricetta In Uso"."Passo 14" := "Ricette"."Passo 14";
   "Ricetta In Uso"."Passo 15" := "Ricette"."Passo 15";
   "Ricetta In Uso"."Passo 16" := "Ricette"."Passo 16";
   "Ricetta In Uso"."Passo 17" := "Ricette"."Passo 17";
   "Ricetta In Uso"."Passo 18" := "Ricette"."Passo 18";
   "Ricetta In Uso"."Passo 19" := "Ricette"."Passo 19";
   "Ricetta In Uso"."Passo 20" := "Ricette"."Passo 20";
END_REGION

REGION Network 6: COSTRUZIONE BIT PIN
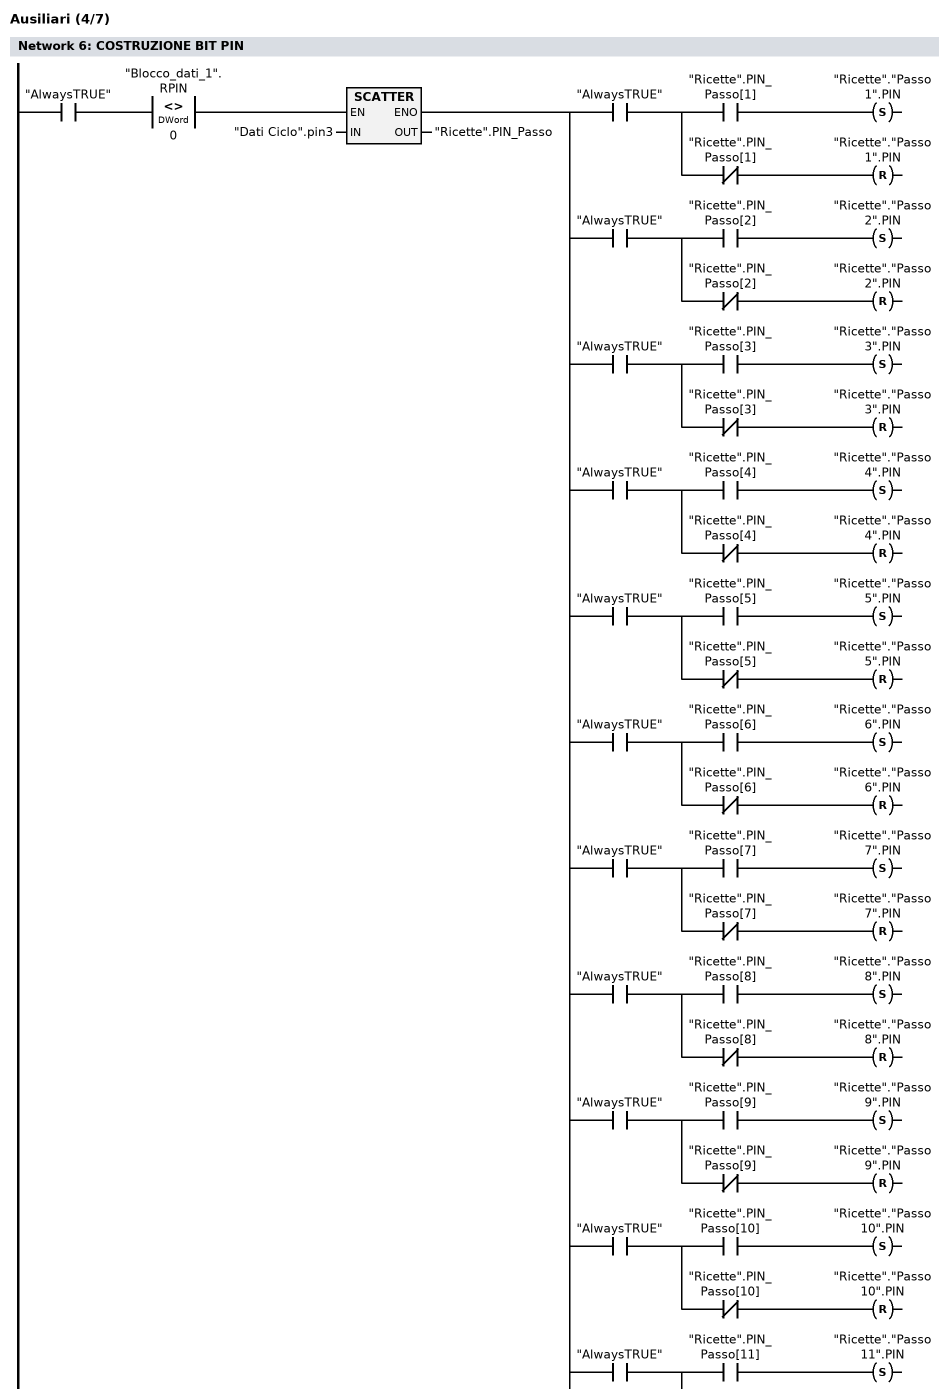
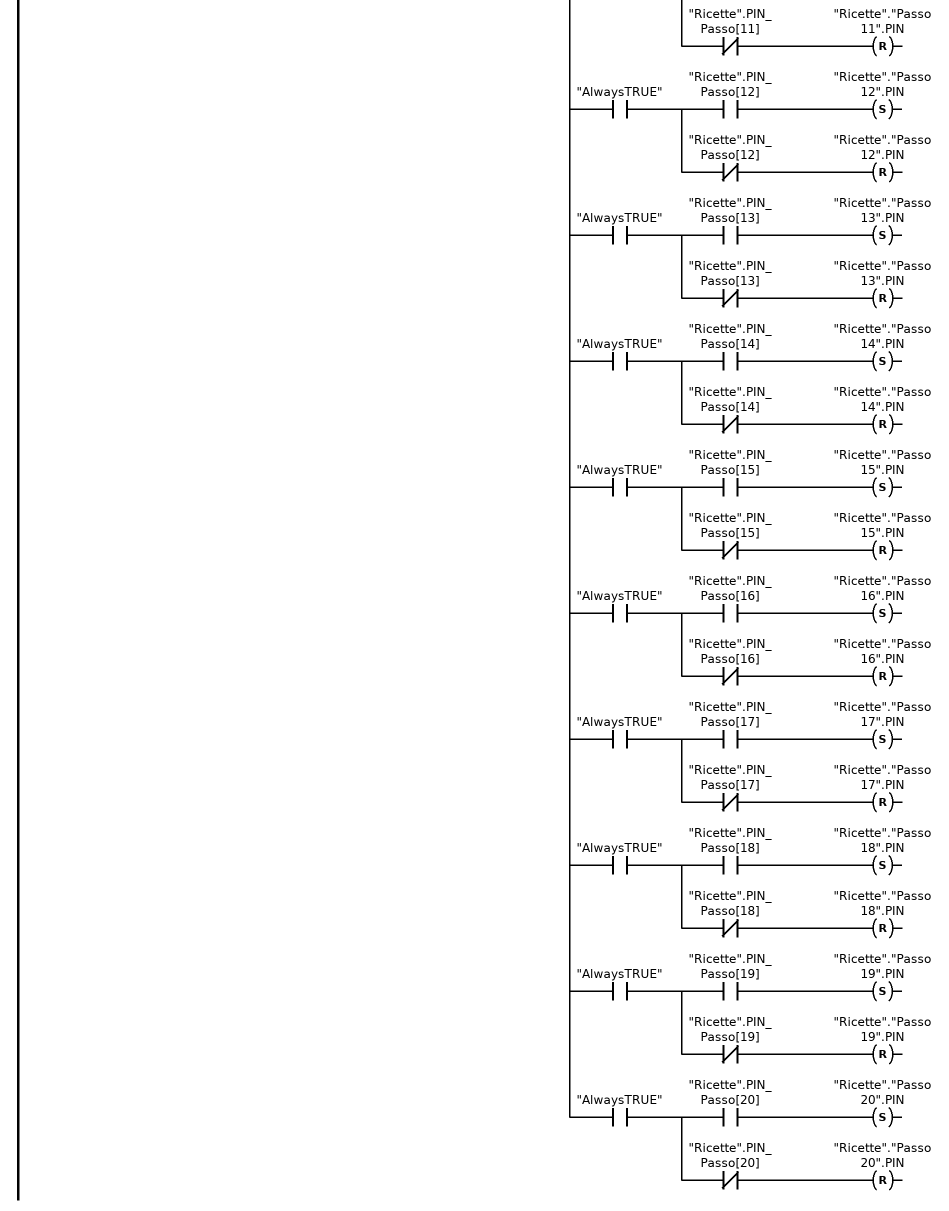
   #_w1 := "AlwaysTRUE" AND ("Blocco_dati_1".RPIN <> 0);
   IF #_w1 THEN SCATTER(IN := "Dati Ciclo".pin3, OUT => "Ricette".PIN_Passo); END_IF;
   #_w2 := #_w1 AND "AlwaysTRUE";
   IF #_w2 AND "Ricette".PIN_Passo[1] THEN "Ricette"."Passo 1".PIN := TRUE; END_IF;
   IF #_w2 AND NOT "Ricette".PIN_Passo[1] THEN "Ricette"."Passo 1".PIN := FALSE; END_IF;
   #_w3 := #_w1 AND "AlwaysTRUE";
   IF #_w3 AND "Ricette".PIN_Passo[2] THEN "Ricette"."Passo 2".PIN := TRUE; END_IF;
   IF #_w3 AND NOT "Ricette".PIN_Passo[2] THEN "Ricette"."Passo 2".PIN := FALSE; END_IF;
   #_w4 := #_w1 AND "AlwaysTRUE";
   IF #_w4 AND "Ricette".PIN_Passo[3] THEN "Ricette"."Passo 3".PIN := TRUE; END_IF;
   IF #_w4 AND NOT "Ricette".PIN_Passo[3] THEN "Ricette"."Passo 3".PIN := FALSE; END_IF;
   #_w5 := #_w1 AND "AlwaysTRUE";
   IF #_w5 AND "Ricette".PIN_Passo[4] THEN "Ricette"."Passo 4".PIN := TRUE; END_IF;
   IF #_w5 AND NOT "Ricette".PIN_Passo[4] THEN "Ricette"."Passo 4".PIN := FALSE; END_IF;
   #_w6 := #_w1 AND "AlwaysTRUE";
   IF #_w6 AND "Ricette".PIN_Passo[5] THEN "Ricette"."Passo 5".PIN := TRUE; END_IF;
   IF #_w6 AND NOT "Ricette".PIN_Passo[5] THEN "Ricette"."Passo 5".PIN := FALSE; END_IF;
   #_w7 := #_w1 AND "AlwaysTRUE";
   IF #_w7 AND "Ricette".PIN_Passo[6] THEN "Ricette"."Passo 6".PIN := TRUE; END_IF;
   IF #_w7 AND NOT "Ricette".PIN_Passo[6] THEN "Ricette"."Passo 6".PIN := FALSE; END_IF;
   #_w8 := #_w1 AND "AlwaysTRUE";
   IF #_w8 AND "Ricette".PIN_Passo[7] THEN "Ricette"."Passo 7".PIN := TRUE; END_IF;
   IF #_w8 AND NOT "Ricette".PIN_Passo[7] THEN "Ricette"."Passo 7".PIN := FALSE; END_IF;
   #_w9 := #_w1 AND "AlwaysTRUE";
   IF #_w9 AND "Ricette".PIN_Passo[8] THEN "Ricette"."Passo 8".PIN := TRUE; END_IF;
   IF #_w9 AND NOT "Ricette".PIN_Passo[8] THEN "Ricette"."Passo 8".PIN := FALSE; END_IF;
   #_w10 := #_w1 AND "AlwaysTRUE";
   IF #_w10 AND "Ricette".PIN_Passo[9] THEN "Ricette"."Passo 9".PIN := TRUE; END_IF;
   IF #_w10 AND NOT "Ricette".PIN_Passo[9] THEN "Ricette"."Passo 9".PIN := FALSE; END_IF;
   #_w11 := #_w1 AND "AlwaysTRUE";
   IF #_w11 AND "Ricette".PIN_Passo[10] THEN "Ricette"."Passo 10".PIN := TRUE; END_IF;
   IF #_w11 AND NOT "Ricette".PIN_Passo[10] THEN "Ricette"."Passo 10".PIN := FALSE; END_IF;
   #_w12 := #_w1 AND "AlwaysTRUE";
   IF #_w12 AND "Ricette".PIN_Passo[11] THEN "Ricette"."Passo 11".PIN := TRUE; END_IF;
   IF #_w12 AND NOT "Ricette".PIN_Passo[11] THEN "Ricette"."Passo 11".PIN := FALSE; END_IF;
   #_w13 := #_w1 AND "AlwaysTRUE";
   IF #_w13 AND "Ricette".PIN_Passo[12] THEN "Ricette"."Passo 12".PIN := TRUE; END_IF;
   IF #_w13 AND NOT "Ricette".PIN_Passo[12] THEN "Ricette"."Passo 12".PIN := FALSE; END_IF;
   #_w14 := #_w1 AND "AlwaysTRUE";
   IF #_w14 AND "Ricette".PIN_Passo[13] THEN "Ricette"."Passo 13".PIN := TRUE; END_IF;
   IF #_w14 AND NOT "Ricette".PIN_Passo[13] THEN "Ricette"."Passo 13".PIN := FALSE; END_IF;
   #_w15 := #_w1 AND "AlwaysTRUE";
   IF #_w15 AND "Ricette".PIN_Passo[14] THEN "Ricette"."Passo 14".PIN := TRUE; END_IF;
   IF #_w15 AND NOT "Ricette".PIN_Passo[14] THEN "Ricette"."Passo 14".PIN := FALSE; END_IF;
   #_w16 := #_w1 AND "AlwaysTRUE";
   IF #_w16 AND "Ricette".PIN_Passo[15] THEN "Ricette"."Passo 15".PIN := TRUE; END_IF;
   IF #_w16 AND NOT "Ricette".PIN_Passo[15] THEN "Ricette"."Passo 15".PIN := FALSE; END_IF;
   #_w17 := #_w1 AND "AlwaysTRUE";
   IF #_w17 AND "Ricette".PIN_Passo[16] THEN "Ricette"."Passo 16".PIN := TRUE; END_IF;
   IF #_w17 AND NOT "Ricette".PIN_Passo[16] THEN "Ricette"."Passo 16".PIN := FALSE; END_IF;
   #_w18 := #_w1 AND "AlwaysTRUE";
   IF #_w18 AND "Ricette".PIN_Passo[17] THEN "Ricette"."Passo 17".PIN := TRUE; END_IF;
   IF #_w18 AND NOT "Ricette".PIN_Passo[17] THEN "Ricette"."Passo 17".PIN := FALSE; END_IF;
   #_w19 := #_w1 AND "AlwaysTRUE";
   IF #_w19 AND "Ricette".PIN_Passo[18] THEN "Ricette"."Passo 18".PIN := TRUE; END_IF;
   IF #_w19 AND NOT "Ricette".PIN_Passo[18] THEN "Ricette"."Passo 18".PIN := FALSE; END_IF;
   #_w20 := #_w1 AND "AlwaysTRUE";
   IF #_w20 AND "Ricette".PIN_Passo[19] THEN "Ricette"."Passo 19".PIN := TRUE; END_IF;
   IF #_w20 AND NOT "Ricette".PIN_Passo[19] THEN "Ricette"."Passo 19".PIN := FALSE; END_IF;
   #_w21 := #_w1 AND "AlwaysTRUE";
   IF #_w21 AND "Ricette".PIN_Passo[20] THEN "Ricette"."Passo 20".PIN := TRUE; END_IF;
   IF #_w21 AND NOT "Ricette".PIN_Passo[20] THEN "Ricette"."Passo 20".PIN := FALSE; END_IF;
END_REGION

REGION Network 7
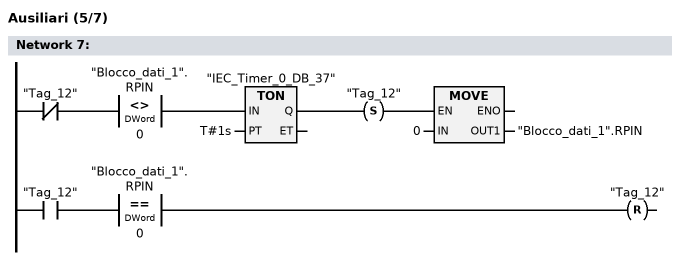
   "IEC_Timer_0_DB_37".TON(IN := NOT "Tag_12" AND ("Blocco_dati_1".RPIN <> 0), PT := T#1s);
   IF "IEC_Timer_0_DB_37".Q THEN
       "Tag_12" := TRUE;
       "Blocco_dati_1".RPIN := 0;
   END_IF;
   IF "Tag_12" AND ("Blocco_dati_1".RPIN = 0) THEN "Tag_12" := FALSE; END_IF;
END_REGION

REGION Network 8: MOLTIPLICA PER MILLE I VALORI TEMPO DELLA RICETTA
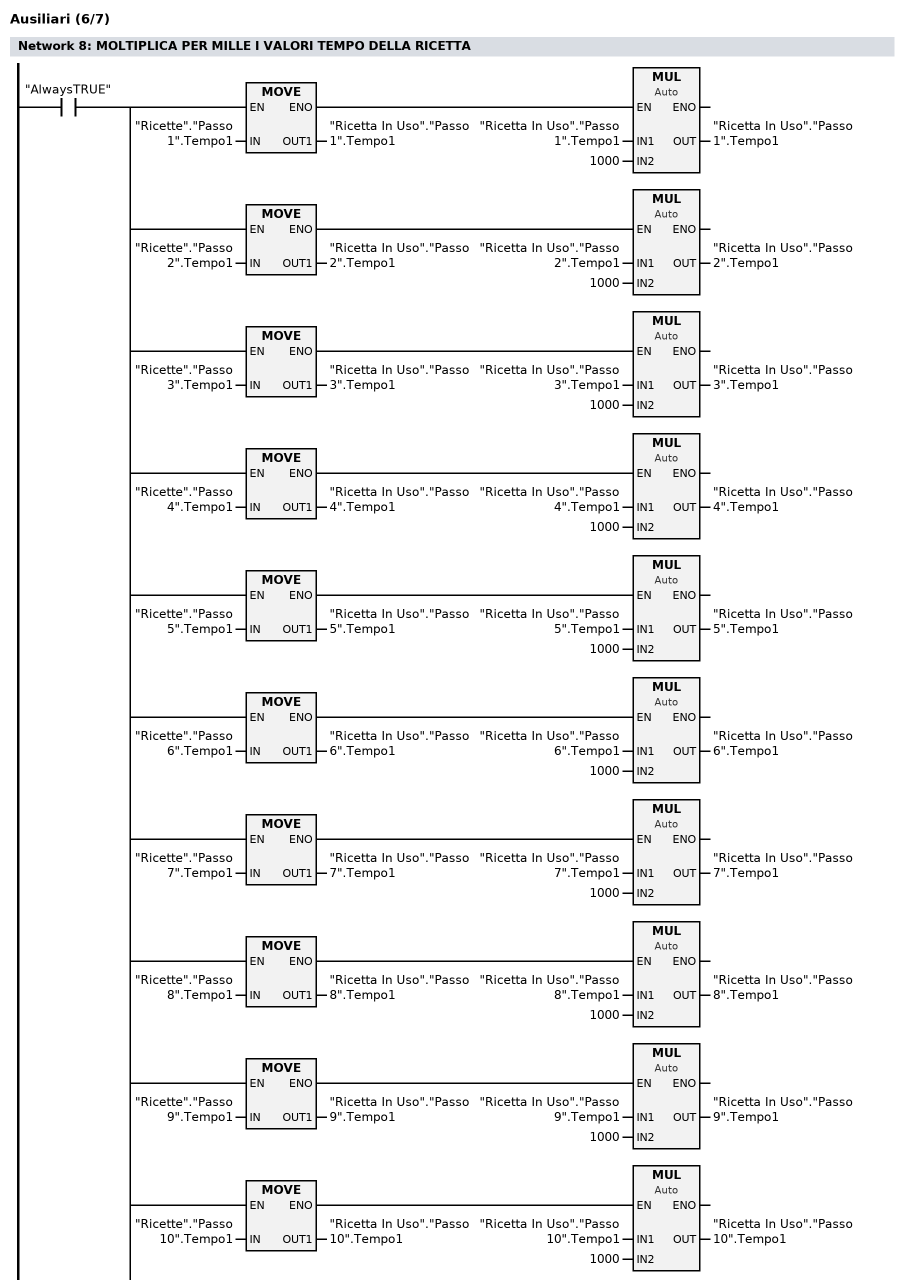
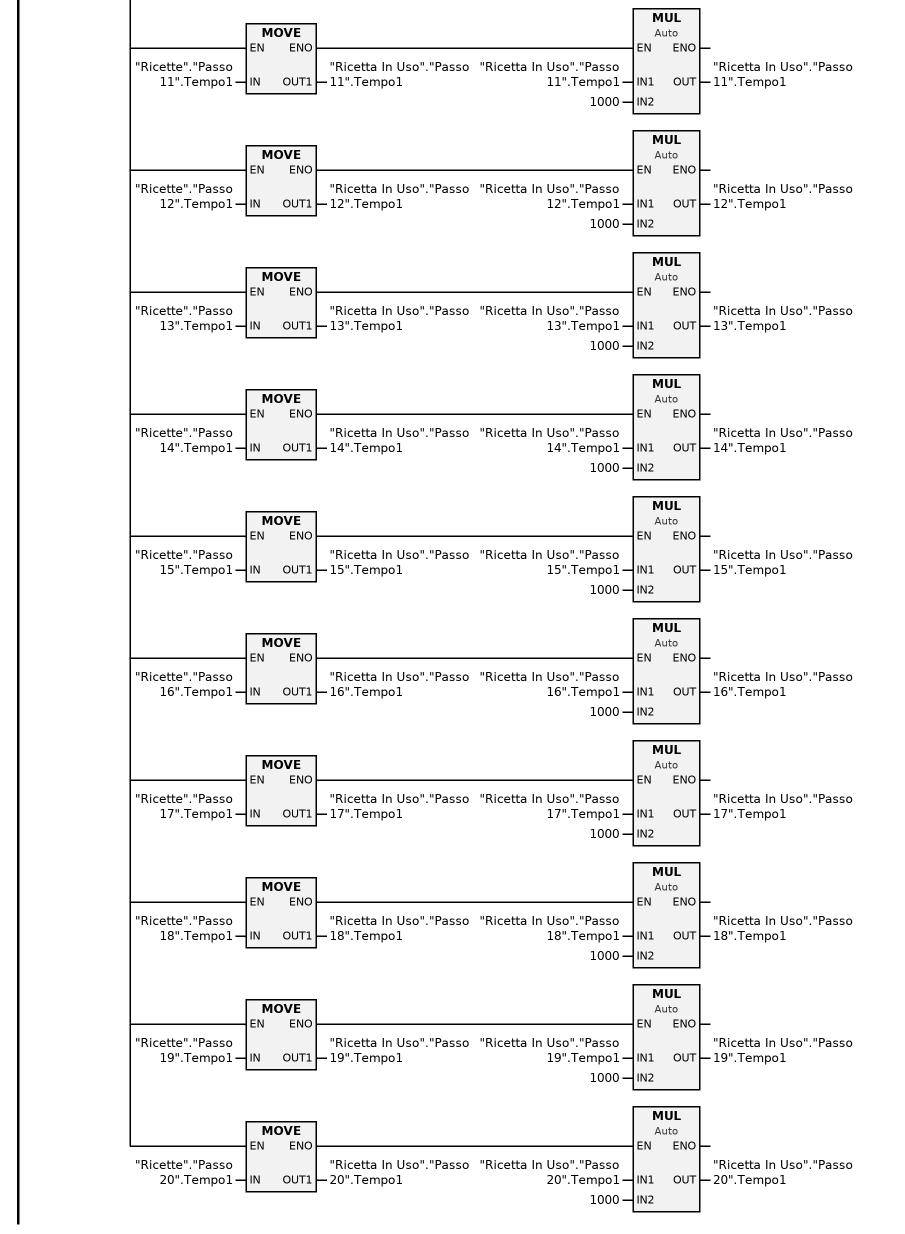
   RUNG wire#powerrail
      Contact( "AlwaysTRUE" )
      wire#w1
      Move(in := "Ricette"."Passo 1".Tempo1, out1 => "Ricetta In Uso"."Passo 1".Tempo1)
      Mul(in1 := "Ricetta In Uso"."Passo 1".Tempo1, in2 := 1000, out => "Ricetta In Uso"."Passo 1".Tempo1)
   END_RUNG
   RUNG wire#w1
      Move(in := "Ricette"."Passo 2".Tempo1, out1 => "Ricetta In Uso"."Passo 2".Tempo1)
      Mul(in1 := "Ricetta In Uso"."Passo 2".Tempo1, in2 := 1000, out => "Ricetta In Uso"."Passo 2".Tempo1)
   END_RUNG
   RUNG wire#w1
      Move(in := "Ricette"."Passo 3".Tempo1, out1 => "Ricetta In Uso"."Passo 3".Tempo1)
      Mul(in1 := "Ricetta In Uso"."Passo 3".Tempo1, in2 := 1000, out => "Ricetta In Uso"."Passo 3".Tempo1)
   END_RUNG
   RUNG wire#w1
      Move(in := "Ricette"."Passo 4".Tempo1, out1 => "Ricetta In Uso"."Passo 4".Tempo1)
      Mul(in1 := "Ricetta In Uso"."Passo 4".Tempo1, in2 := 1000, out => "Ricetta In Uso"."Passo 4".Tempo1)
   END_RUNG
   RUNG wire#w1
      Move(in := "Ricette"."Passo 5".Tempo1, out1 => "Ricetta In Uso"."Passo 5".Tempo1)
      Mul(in1 := "Ricetta In Uso"."Passo 5".Tempo1, in2 := 1000, out => "Ricetta In Uso"."Passo 5".Tempo1)
   END_RUNG
   RUNG wire#w1
      Move(in := "Ricette"."Passo 6".Tempo1, out1 => "Ricetta In Uso"."Passo 6".Tempo1)
      Mul(in1 := "Ricetta In Uso"."Passo 6".Tempo1, in2 := 1000, out => "Ricetta In Uso"."Passo 6".Tempo1)
   END_RUNG
   RUNG wire#w1
      Move(in := "Ricette"."Passo 7".Tempo1, out1 => "Ricetta In Uso"."Passo 7".Tempo1)
      Mul(in1 := "Ricetta In Uso"."Passo 7".Tempo1, in2 := 1000, out => "Ricetta In Uso"."Passo 7".Tempo1)
   END_RUNG
   RUNG wire#w1
      Move(in := "Ricette"."Passo 8".Tempo1, out1 => "Ricetta In Uso"."Passo 8".Tempo1)
      Mul(in1 := "Ricetta In Uso"."Passo 8".Tempo1, in2 := 1000, out => "Ricetta In Uso"."Passo 8".Tempo1)
   END_RUNG
   RUNG wire#w1
      Move(in := "Ricette"."Passo 9".Tempo1, out1 => "Ricetta In Uso"."Passo 9".Tempo1)
      Mul(in1 := "Ricetta In Uso"."Passo 9".Tempo1, in2 := 1000, out => "Ricetta In Uso"."Passo 9".Tempo1)
   END_RUNG
   RUNG wire#w1
      Move(in := "Ricette"."Passo 10".Tempo1, out1 => "Ricetta In Uso"."Passo 10".Tempo1)
      Mul(in1 := "Ricetta In Uso"."Passo 10".Tempo1, in2 := 1000, out => "Ricetta In Uso"."Passo 10".Tempo1)
   END_RUNG
   RUNG wire#w1
      Move(in := "Ricette"."Passo 11".Tempo1, out1 => "Ricetta In Uso"."Passo 11".Tempo1)
      Mul(in1 := "Ricetta In Uso"."Passo 11".Tempo1, in2 := 1000, out => "Ricetta In Uso"."Passo 11".Tempo1)
   END_RUNG
   RUNG wire#w1
      Move(in := "Ricette"."Passo 12".Tempo1, out1 => "Ricetta In Uso"."Passo 12".Tempo1)
      Mul(in1 := "Ricetta In Uso"."Passo 12".Tempo1, in2 := 1000, out => "Ricetta In Uso"."Passo 12".Tempo1)
   END_RUNG
   RUNG wire#w1
      Move(in := "Ricette"."Passo 13".Tempo1, out1 => "Ricetta In Uso"."Passo 13".Tempo1)
      Mul(in1 := "Ricetta In Uso"."Passo 13".Tempo1, in2 := 1000, out => "Ricetta In Uso"."Passo 13".Tempo1)
   END_RUNG
   RUNG wire#w1
      Move(in := "Ricette"."Passo 14".Tempo1, out1 => "Ricetta In Uso"."Passo 14".Tempo1)
      Mul(in1 := "Ricetta In Uso"."Passo 14".Tempo1, in2 := 1000, out => "Ricetta In Uso"."Passo 14".Tempo1)
   END_RUNG
   RUNG wire#w1
      Move(in := "Ricette"."Passo 15".Tempo1, out1 => "Ricetta In Uso"."Passo 15".Tempo1)
      Mul(in1 := "Ricetta In Uso"."Passo 15".Tempo1, in2 := 1000, out => "Ricetta In Uso"."Passo 15".Tempo1)
   END_RUNG
   RUNG wire#w1
      Move(in := "Ricette"."Passo 16".Tempo1, out1 => "Ricetta In Uso"."Passo 16".Tempo1)
      Mul(in1 := "Ricetta In Uso"."Passo 16".Tempo1, in2 := 1000, out => "Ricetta In Uso"."Passo 16".Tempo1)
   END_RUNG
   RUNG wire#w1
      Move(in := "Ricette"."Passo 17".Tempo1, out1 => "Ricetta In Uso"."Passo 17".Tempo1)
      Mul(in1 := "Ricetta In Uso"."Passo 17".Tempo1, in2 := 1000, out => "Ricetta In Uso"."Passo 17".Tempo1)
   END_RUNG
   RUNG wire#w1
      Move(in := "Ricette"."Passo 18".Tempo1, out1 => "Ricetta In Uso"."Passo 18".Tempo1)
      Mul(in1 := "Ricetta In Uso"."Passo 18".Tempo1, in2 := 1000, out => "Ricetta In Uso"."Passo 18".Tempo1)
   END_RUNG
   RUNG wire#w1
      Move(in := "Ricette"."Passo 19".Tempo1, out1 => "Ricetta In Uso"."Passo 19".Tempo1)
      Mul(in1 := "Ricetta In Uso"."Passo 19".Tempo1, in2 := 1000, out => "Ricetta In Uso"."Passo 19".Tempo1)
   END_RUNG
   RUNG wire#w1
      Move(in := "Ricette"."Passo 20".Tempo1, out1 => "Ricetta In Uso"."Passo 20".Tempo1)
      Mul(in1 := "Ricetta In Uso"."Passo 20".Tempo1, in2 := 1000, out => "Ricetta In Uso"."Passo 20".Tempo1)
   END_RUNG
   // the same network as SCL:
   IF "AlwaysTRUE" THEN
       "Ricetta In Uso"."Passo 1".Tempo1 := "Ricette"."Passo 1".Tempo1;
       "Ricetta In Uso"."Passo 1".Tempo1 := "Ricetta In Uso"."Passo 1".Tempo1 * 1000;
       "Ricetta In Uso"."Passo 2".Tempo1 := "Ricette"."Passo 2".Tempo1;
       "Ricetta In Uso"."Passo 2".Tempo1 := "Ricetta In Uso"."Passo 2".Tempo1 * 1000;
       "Ricetta In Uso"."Passo 3".Tempo1 := "Ricette"."Passo 3".Tempo1;
       "Ricetta In Uso"."Passo 3".Tempo1 := "Ricetta In Uso"."Passo 3".Tempo1 * 1000;
       "Ricetta In Uso"."Passo 4".Tempo1 := "Ricette"."Passo 4".Tempo1;
       "Ricetta In Uso"."Passo 4".Tempo1 := "Ricetta In Uso"."Passo 4".Tempo1 * 1000;
       "Ricetta In Uso"."Passo 5".Tempo1 := "Ricette"."Passo 5".Tempo1;
       "Ricetta In Uso"."Passo 5".Tempo1 := "Ricetta In Uso"."Passo 5".Tempo1 * 1000;
       "Ricetta In Uso"."Passo 6".Tempo1 := "Ricette"."Passo 6".Tempo1;
       "Ricetta In Uso"."Passo 6".Tempo1 := "Ricetta In Uso"."Passo 6".Tempo1 * 1000;
       "Ricetta In Uso"."Passo 7".Tempo1 := "Ricette"."Passo 7".Tempo1;
       "Ricetta In Uso"."Passo 7".Tempo1 := "Ricetta In Uso"."Passo 7".Tempo1 * 1000;
       "Ricetta In Uso"."Passo 8".Tempo1 := "Ricette"."Passo 8".Tempo1;
       "Ricetta In Uso"."Passo 8".Tempo1 := "Ricetta In Uso"."Passo 8".Tempo1 * 1000;
       "Ricetta In Uso"."Passo 9".Tempo1 := "Ricette"."Passo 9".Tempo1;
       "Ricetta In Uso"."Passo 9".Tempo1 := "Ricetta In Uso"."Passo 9".Tempo1 * 1000;
       "Ricetta In Uso"."Passo 10".Tempo1 := "Ricette"."Passo 10".Tempo1;
       "Ricetta In Uso"."Passo 10".Tempo1 := "Ricetta In Uso"."Passo 10".Tempo1 * 1000;
       "Ricetta In Uso"."Passo 11".Tempo1 := "Ricette"."Passo 11".Tempo1;
       "Ricetta In Uso"."Passo 11".Tempo1 := "Ricetta In Uso"."Passo 11".Tempo1 * 1000;
       "Ricetta In Uso"."Passo 12".Tempo1 := "Ricette"."Passo 12".Tempo1;
       "Ricetta In Uso"."Passo 12".Tempo1 := "Ricetta In Uso"."Passo 12".Tempo1 * 1000;
       "Ricetta In Uso"."Passo 13".Tempo1 := "Ricette"."Passo 13".Tempo1;
       "Ricetta In Uso"."Passo 13".Tempo1 := "Ricetta In Uso"."Passo 13".Tempo1 * 1000;
       "Ricetta In Uso"."Passo 14".Tempo1 := "Ricette"."Passo 14".Tempo1;
       "Ricetta In Uso"."Passo 14".Tempo1 := "Ricetta In Uso"."Passo 14".Tempo1 * 1000;
       "Ricetta In Uso"."Passo 15".Tempo1 := "Ricette"."Passo 15".Tempo1;
       "Ricetta In Uso"."Passo 15".Tempo1 := "Ricetta In Uso"."Passo 15".Tempo1 * 1000;
       "Ricetta In Uso"."Passo 16".Tempo1 := "Ricette"."Passo 16".Tempo1;
       "Ricetta In Uso"."Passo 16".Tempo1 := "Ricetta In Uso"."Passo 16".Tempo1 * 1000;
       "Ricetta In Uso"."Passo 17".Tempo1 := "Ricette"."Passo 17".Tempo1;
       "Ricetta In Uso"."Passo 17".Tempo1 := "Ricetta In Uso"."Passo 17".Tempo1 * 1000;
       "Ricetta In Uso"."Passo 18".Tempo1 := "Ricette"."Passo 18".Tempo1;
       "Ricetta In Uso"."Passo 18".Tempo1 := "Ricetta In Uso"."Passo 18".Tempo1 * 1000;
       "Ricetta In Uso"."Passo 19".Tempo1 := "Ricette"."Passo 19".Tempo1;
       "Ricetta In Uso"."Passo 19".Tempo1 := "Ricetta In Uso"."Passo 19".Tempo1 * 1000;
       "Ricetta In Uso"."Passo 20".Tempo1 := "Ricette"."Passo 20".Tempo1;
       "Ricetta In Uso"."Passo 20".Tempo1 := "Ricetta In Uso"."Passo 20".Tempo1 * 1000;
   END_IF;
END_REGION

REGION Network 9: VISUALIZZAZIONE NUMERO PASSO -1 PER HMI
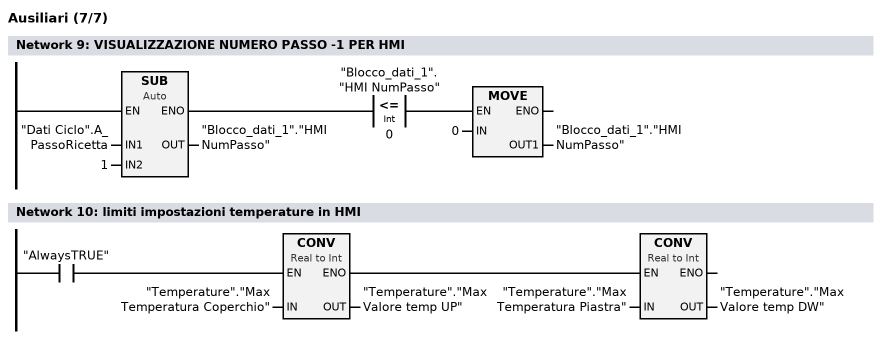
   RUNG wire#powerrail
      Sub(in1 := "Dati Ciclo".A_PassoRicetta, in2 := 1, out => "Blocco_dati_1"."HMI NumPasso")
      { S7_Templates := "SrcType := Int" } LE_Contact(in1 := "Blocco_dati_1"."HMI NumPasso", in2 := 0)
      Move(in := 0, out1 => "Blocco_dati_1"."HMI NumPasso")
   END_RUNG
   // the same network as SCL:
   "Blocco_dati_1"."HMI NumPasso" := "Dati Ciclo".A_PassoRicetta - 1;
   IF "Blocco_dati_1"."HMI NumPasso" <= 0 THEN "Blocco_dati_1"."HMI NumPasso" := 0; END_IF;
END_REGION

REGION Network 10: limiti impostazioni temperature in HMI
   RUNG wire#powerrail
      Contact( "AlwaysTRUE" )
      { S7_Templates := "[SrcType := Real, DestType := Int]" } Convert(in := "Temperature"."Max Temperatura Coperchio", out => "Temperature"."Max Valore temp UP")
      { S7_Templates := "[SrcType := Real, DestType := Int]" } Convert(in := "Temperature"."Max Temperatura Piastra", out => "Temperature"."Max Valore temp DW")
   END_RUNG
   // the same network as SCL:
   IF "AlwaysTRUE" THEN
       "Temperature"."Max Valore temp UP" := REAL_TO_INT("Temperature"."Max Temperatura Coperchio");
       "Temperature"."Max Valore temp DW" := REAL_TO_INT("Temperature"."Max Temperatura Piastra");
   END_IF;
END_REGION
END_FUNCTION

FUNCTION "Segnalazioni" : Void   // FC6, LAD
{ S7_Optimized_Access := 'TRUE' }
VERSION : 0.1
BEGIN

REGION Network 1: Q0.1 LAMPADA ALLARME
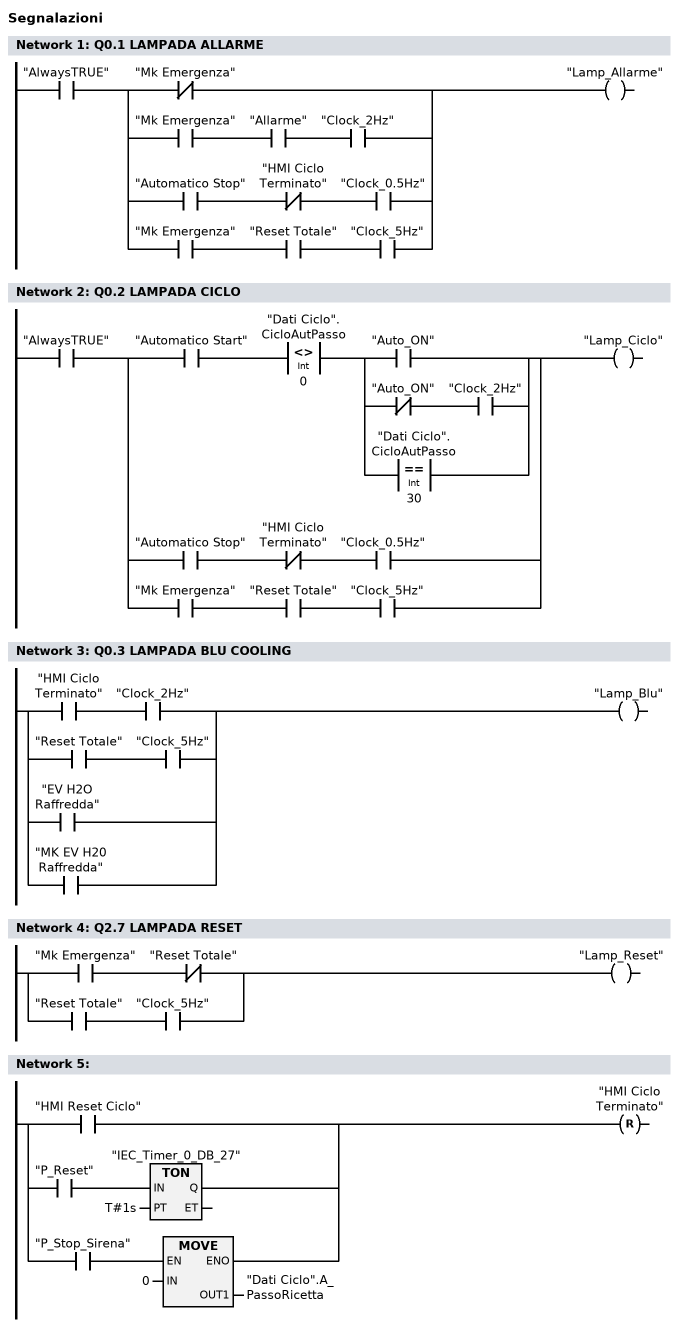
   RUNG wire#powerrail
      Contact( "AlwaysTRUE" )
      wire#w1
      I_Contact( "Mk Emergenza" )
      wire#w2
      Coil( "Lamp_Allarme" )
   END_RUNG
   RUNG wire#w1
      Contact( "Mk Emergenza" )
      Contact( "Allarme" )
      Contact( "Clock_2Hz" )
   END_RUNG wire#w2
   RUNG wire#w1
      Contact( "Automatico Stop" )
      I_Contact( "HMI Ciclo Terminato" )
      Contact( "Clock_0.5Hz" )
   END_RUNG wire#w2
   RUNG wire#w1
      Contact( "Mk Emergenza" )
      Contact( "Reset Totale" )
      Contact( "Clock_5Hz" )
   END_RUNG wire#w2
   // the same network as SCL:
   "Lamp_Allarme" := "AlwaysTRUE" AND (NOT "Mk Emergenza" OR ("Mk Emergenza" AND "Allarme" AND "Clock_2Hz") OR ("Automatico Stop" AND NOT "HMI Ciclo Terminato" AND "Clock_0.5Hz") OR ("Mk Emergenza" AND "Reset Totale" AND "Clock_5Hz"));
END_REGION

REGION Network 2: Q0.2 LAMPADA CICLO
   RUNG wire#powerrail
      Contact( "AlwaysTRUE" )
      wire#w1
      Contact( "Automatico Start" )
      { S7_Templates := "SrcType := Int" } NE_Contact(in1 := "Dati Ciclo".CicloAutPasso, in2 := 0)
      wire#w2
      Contact( "Auto_ON" )
      wire#w3
      Coil( "Lamp_Ciclo" )
   END_RUNG
   RUNG wire#w2
      I_Contact( "Auto_ON" )
      Contact( "Clock_2Hz" )
   END_RUNG wire#w3
   RUNG wire#w2
      { S7_Templates := "SrcType := Int" } EQ_Contact(in1 := "Dati Ciclo".CicloAutPasso, in2 := 30)
   END_RUNG wire#w3
   RUNG wire#w1
      Contact( "Automatico Stop" )
      I_Contact( "HMI Ciclo Terminato" )
      Contact( "Clock_0.5Hz" )
   END_RUNG wire#w3
   RUNG wire#w1
      Contact( "Mk Emergenza" )
      Contact( "Reset Totale" )
      Contact( "Clock_5Hz" )
   END_RUNG wire#w3
   // the same network as SCL:
   "Lamp_Ciclo" := "AlwaysTRUE" AND (("Automatico Start" AND ("Dati Ciclo".CicloAutPasso <> 0) AND ("Auto_ON" OR (NOT "Auto_ON" AND "Clock_2Hz") OR ("Dati Ciclo".CicloAutPasso = 30))) OR ("Automatico Stop" AND NOT "HMI Ciclo Terminato" AND "Clock_0.5Hz") OR ("Mk Emergenza" AND "Reset Totale" AND "Clock_5Hz"));
END_REGION

REGION Network 3: Q0.3 LAMPADA BLU COOLING
   RUNG wire#powerrail
      Contact( "HMI Ciclo Terminato" )
      Contact( "Clock_2Hz" )
      wire#w1
      Coil( "Lamp_Blu" )
   END_RUNG
   RUNG wire#powerrail
      Contact( "Reset Totale" )
      Contact( "Clock_5Hz" )
   END_RUNG wire#w1
   RUNG wire#powerrail
      Contact( "EV H2O Raffredda" )
   END_RUNG wire#w1
   RUNG wire#powerrail
      Contact( "MK EV H20 Raffredda" )
   END_RUNG wire#w1
   // the same network as SCL:
   "Lamp_Blu" := ("HMI Ciclo Terminato" AND "Clock_2Hz") OR ("Reset Totale" AND "Clock_5Hz") OR "EV H2O Raffredda" OR "MK EV H20 Raffredda";
END_REGION

REGION Network 4: Q2.7 LAMPADA RESET
   RUNG wire#powerrail
      Contact( "Mk Emergenza" )
      I_Contact( "Reset Totale" )
      wire#w1
      Coil( "Lamp_Reset" )
   END_RUNG
   RUNG wire#powerrail
      Contact( "Reset Totale" )
      Contact( "Clock_5Hz" )
   END_RUNG wire#w1
   // the same network as SCL:
   "Lamp_Reset" := ("Mk Emergenza" AND NOT "Reset Totale") OR ("Reset Totale" AND "Clock_5Hz");
END_REGION

REGION Network 5
   "IEC_Timer_0_DB_27".TON(IN := "P_Reset", PT := T#1s);
   IF "P_Stop_Sirena" THEN "Dati Ciclo".A_PassoRicetta := 0; END_IF;
   IF "HMI Reset Ciclo" OR "IEC_Timer_0_DB_27".Q OR "P_Stop_Sirena" THEN
       "HMI Ciclo Terminato" := FALSE;
   END_IF;
END_REGION
END_FUNCTION

FUNCTION "Blocco_1" : Void   // FC7, LAD
{ S7_Optimized_Access := 'TRUE' }
VERSION : 0.1
BEGIN

REGION Network 1
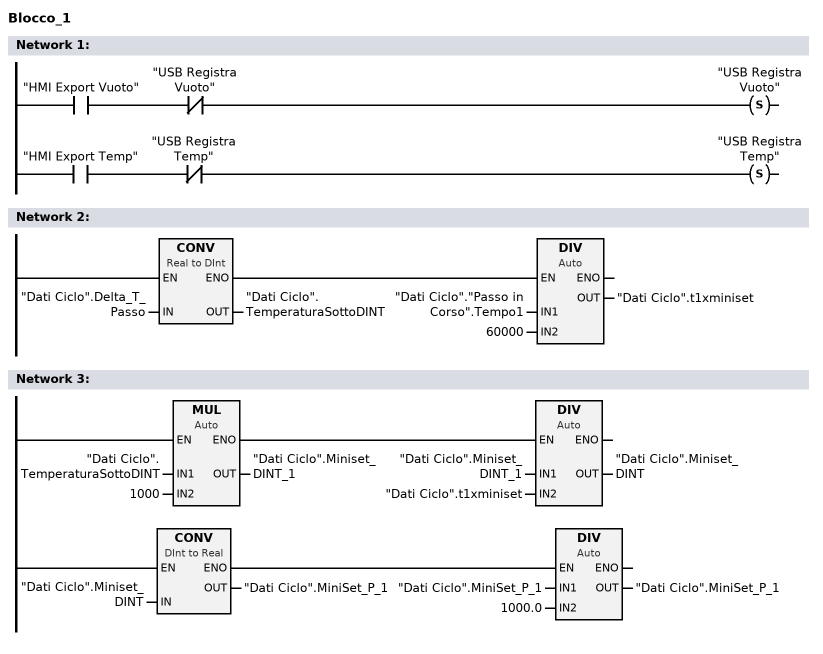
   RUNG wire#powerrail
      Contact( "HMI Export Vuoto" )
      I_Contact( "USB Registra Vuoto" )
      S_Coil( "USB Registra Vuoto" )
   END_RUNG
   RUNG wire#powerrail
      Contact( "HMI Export Temp" )
      I_Contact( "USB Registra Temp" )
      S_Coil( "USB Registra Temp" )
   END_RUNG
   // the same network as SCL:
   IF "HMI Export Vuoto" AND NOT "USB Registra Vuoto" THEN "USB Registra Vuoto" := TRUE; END_IF;
   IF "HMI Export Temp" AND NOT "USB Registra Temp" THEN "USB Registra Temp" := TRUE; END_IF;
END_REGION

REGION Network 2
   RUNG wire#powerrail
      { S7_Templates := "[SrcType := Real, DestType := DInt]" } Convert(in := "Dati Ciclo".Delta_T_Passo, out => "Dati Ciclo".TemperaturaSottoDINT)
      Div(in1 := "Dati Ciclo"."Passo in Corso".Tempo1, in2 := 60000, out => "Dati Ciclo".t1xminiset)
   END_RUNG
   // the same network as SCL:
   "Dati Ciclo".TemperaturaSottoDINT := REAL_TO_DINT("Dati Ciclo".Delta_T_Passo);
   "Dati Ciclo".t1xminiset := "Dati Ciclo"."Passo in Corso".Tempo1 / 60000;
END_REGION

REGION Network 3
   RUNG wire#powerrail
      Mul(in1 := "Dati Ciclo".TemperaturaSottoDINT, in2 := 1000, out => "Dati Ciclo".Miniset_DINT_1)
      Div(in1 := "Dati Ciclo".Miniset_DINT_1, in2 := "Dati Ciclo".t1xminiset, out => "Dati Ciclo".Miniset_DINT)
   END_RUNG
   RUNG wire#powerrail
      { S7_Templates := "[SrcType := DInt, DestType := Real]" } Convert(in := "Dati Ciclo".Miniset_DINT, out => "Dati Ciclo".MiniSet_P_1)
      Div(in1 := "Dati Ciclo".MiniSet_P_1, in2 := 1000.0, out => "Dati Ciclo".MiniSet_P_1)
   END_RUNG
   // the same network as SCL:
   "Dati Ciclo".Miniset_DINT_1 := "Dati Ciclo".TemperaturaSottoDINT * 1000;
   "Dati Ciclo".Miniset_DINT := "Dati Ciclo".Miniset_DINT_1 / "Dati Ciclo".t1xminiset;
   "Dati Ciclo".MiniSet_P_1 := DINT_TO_REAL("Dati Ciclo".Miniset_DINT);
   "Dati Ciclo".MiniSet_P_1 := "Dati Ciclo".MiniSet_P_1 / 1000.0;
END_REGION
END_FUNCTION

FUNCTION "Data Ora" : Void   // FC8, LAD
{ S7_Optimized_Access := 'TRUE' }
VERSION : 0.1
   VAR_TEMP   // added for the SCL form of the ladder/FBD networks
      _w1 : Bool;
      _w2 : Bool;
   END_VAR
BEGIN

REGION Network 1
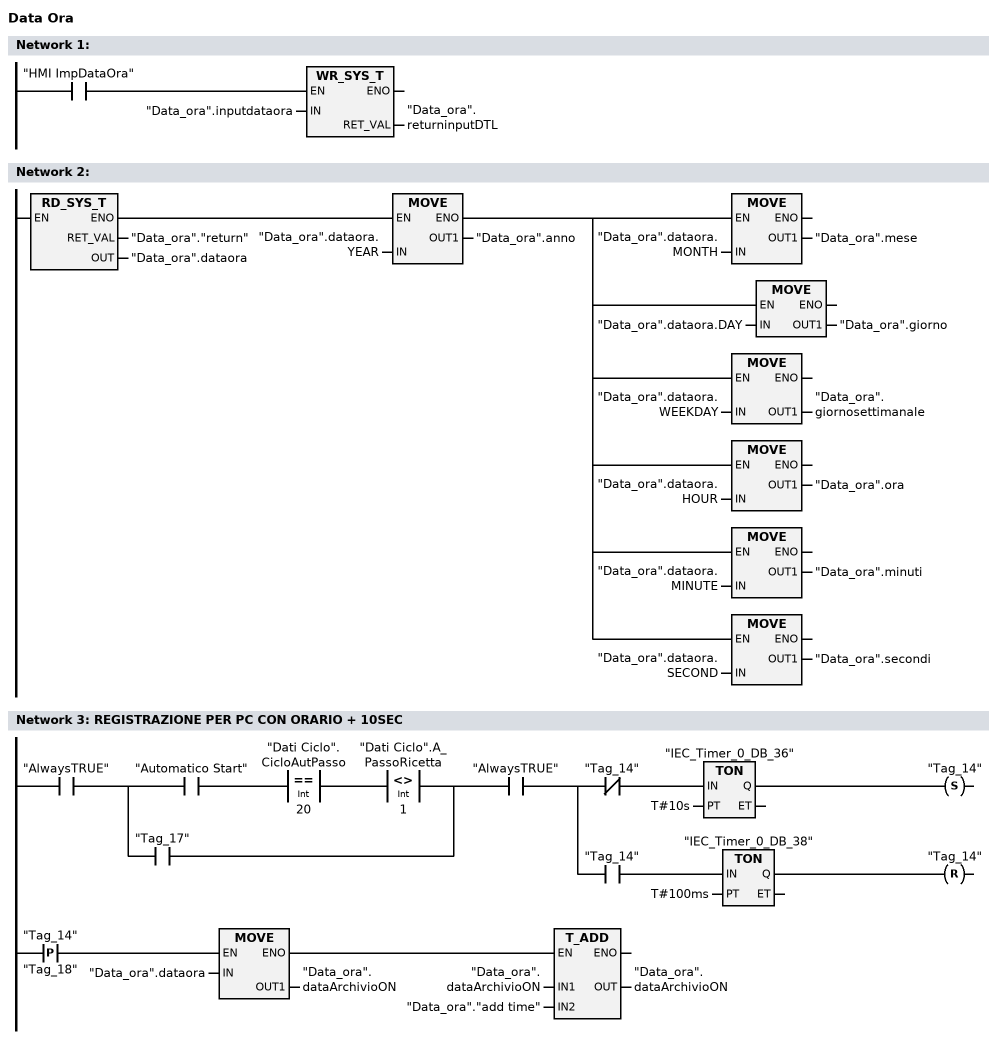
   IF "HMI ImpDataOra" THEN "Data_ora".returninputDTL := WR_SYS_T(IN := "Data_ora".inputdataora); END_IF;
END_REGION

REGION Network 2
   // ENO of a box is taken as its EN; it also drops when the box reports an error
   "Data_ora"."return" := RD_SYS_T(OUT => "Data_ora".dataora);
   "Data_ora".anno := "Data_ora".dataora.YEAR;
   "Data_ora".mese := "Data_ora".dataora.MONTH;
   "Data_ora".giorno := "Data_ora".dataora.DAY;
   "Data_ora".giornosettimanale := "Data_ora".dataora.WEEKDAY;
   "Data_ora".ora := "Data_ora".dataora.HOUR;
   "Data_ora".minuti := "Data_ora".dataora.MINUTE;
   "Data_ora".secondi := "Data_ora".dataora.SECOND;
END_REGION

REGION Network 3: REGISTRAZIONE PER PC CON ORARIO + 10SEC
   #_w1 := "AlwaysTRUE" AND (("Automatico Start" AND ("Dati Ciclo".CicloAutPasso = 20) AND ("Dati Ciclo".A_PassoRicetta <> 1)) OR "Tag_17") AND "AlwaysTRUE";
   "IEC_Timer_0_DB_36".TON(IN := #_w1 AND NOT "Tag_14", PT := T#10s);
   IF "IEC_Timer_0_DB_36".Q THEN "Tag_14" := TRUE; END_IF;
   "IEC_Timer_0_DB_38".TON(IN := #_w1 AND "Tag_14", PT := T#100ms);
   IF "IEC_Timer_0_DB_38".Q THEN "Tag_14" := FALSE; END_IF;
   #_w2 := "Tag_14" AND NOT "Tag_18";   // rising edge of "Tag_14"
   "Tag_18" := "Tag_14";
   IF #_w2 THEN
       "Data_ora".dataArchivioON := "Data_ora".dataora;
       "Data_ora".dataArchivioON := T_ADD(IN1 := "Data_ora".dataArchivioON, IN2 := "Data_ora"."add time");
   END_IF;
END_REGION
END_FUNCTION

FUNCTION "Allarmi" : Void   // FC9, LAD
{ S7_Optimized_Access := 'TRUE' }
VERSION : 0.1
   VAR_TEMP   // added for the SCL form of the ladder/FBD networks
      _w1 : Bool;
   END_VAR
BEGIN

REGION Network 1
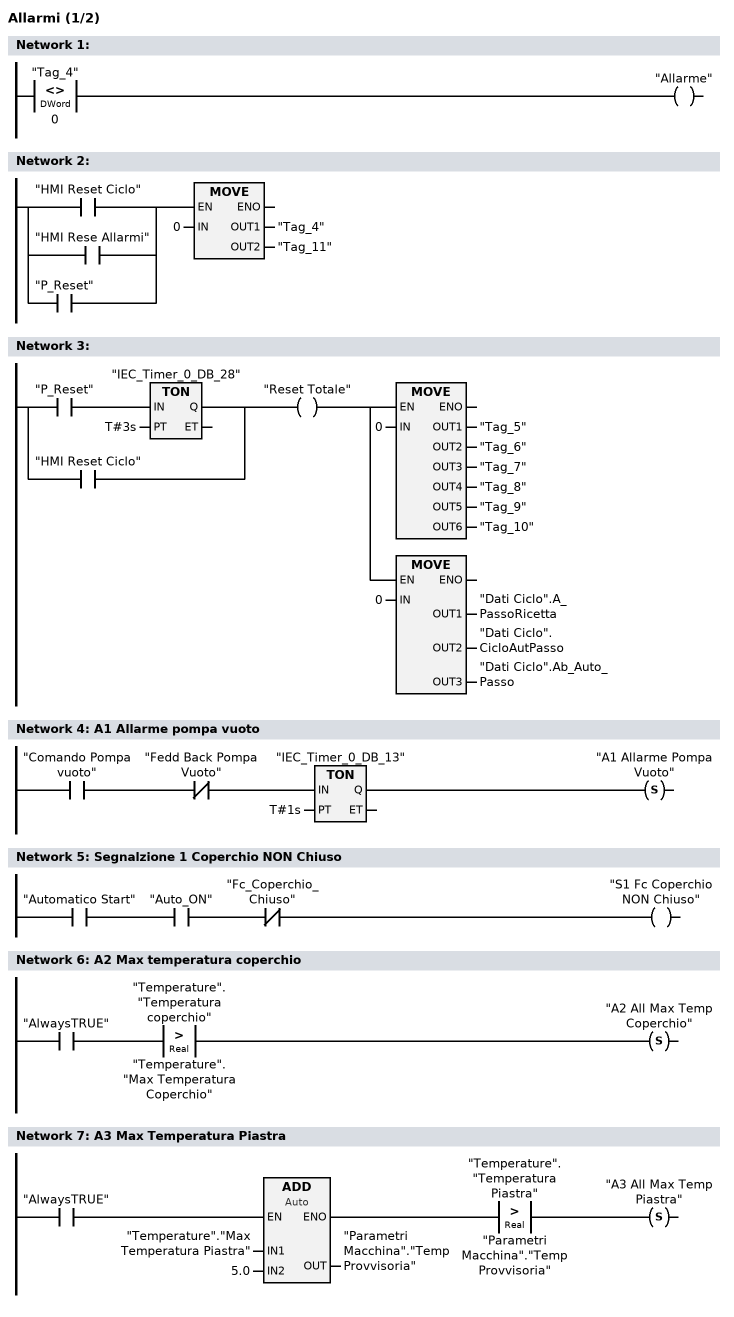
   RUNG wire#powerrail
      { S7_Templates := "SrcType := DWord" } NE_Contact(in1 := "Tag_4", in2 := 0)
      Coil( "Allarme" )
   END_RUNG
   // the same network as SCL:
   "Allarme" := "Tag_4" <> 0;
END_REGION

REGION Network 2
   RUNG wire#powerrail
      Contact( "HMI Reset Ciclo" )
      wire#w1
      Move(in := 0, out1 => "Tag_4", out2 => "Tag_11")
   END_RUNG
   RUNG wire#powerrail
      Contact( "HMI Rese Allarmi" )
   END_RUNG wire#w1
   RUNG wire#powerrail
      Contact( "P_Reset" )
   END_RUNG wire#w1
   // the same network as SCL:
   IF "HMI Reset Ciclo" OR "HMI Rese Allarmi" OR "P_Reset" THEN
       "Tag_4" := 0;
       "Tag_11" := 0;
   END_IF;
END_REGION

REGION Network 3
   "IEC_Timer_0_DB_28".TON(IN := "P_Reset", PT := T#3s);
   "Reset Totale" := "IEC_Timer_0_DB_28".Q OR "HMI Reset Ciclo";
   IF "Reset Totale" THEN
       "Tag_5" := 0;
       "Tag_6" := 0;
       "Tag_7" := 0;
       "Tag_8" := 0;
       "Tag_9" := 0;
       "Tag_10" := 0;
       "Dati Ciclo".A_PassoRicetta := 0;
       "Dati Ciclo".CicloAutPasso := 0;
       "Dati Ciclo".Ab_Auto_Passo := 0;
   END_IF;
END_REGION

REGION Network 4: A1 Allarme pompa vuoto
   "IEC_Timer_0_DB_13".TON(IN := "Comando Pompa vuoto" AND NOT "Fedd Back Pompa Vuoto", PT := T#1s);
   IF "IEC_Timer_0_DB_13".Q THEN "A1 Allarme Pompa Vuoto" := TRUE; END_IF;
END_REGION

REGION Network 5: Segnalzione 1 Coperchio NON Chiuso
   RUNG wire#powerrail
      Contact( "Automatico Start" )
      Contact( "Auto_ON" )
      I_Contact( "Fc_Coperchio_Chiuso" )
      Coil( "S1 Fc Coperchio NON Chiuso" )
   END_RUNG
   // the same network as SCL:
   "S1 Fc Coperchio NON Chiuso" := "Automatico Start" AND "Auto_ON" AND NOT "Fc_Coperchio_Chiuso";
END_REGION

REGION Network 6: A2 Max temperatura coperchio
   RUNG wire#powerrail
      Contact( "AlwaysTRUE" )
      { S7_Templates := "SrcType := Real" } GT_Contact(in1 := "Temperature"."Temperatura coperchio", in2 := "Temperature"."Max Temperatura Coperchio")
      S_Coil( "A2 All Max Temp Coperchio" )
   END_RUNG
   // the same network as SCL:
   IF "AlwaysTRUE" AND ("Temperature"."Temperatura coperchio" > "Temperature"."Max Temperatura Coperchio") THEN
       "A2 All Max Temp Coperchio" := TRUE;
   END_IF;
END_REGION

REGION Network 7: A3 Max Temperatura Piastra
   RUNG wire#powerrail
      Contact( "AlwaysTRUE" )
      Add(in1 := "Temperature"."Max Temperatura Piastra", in2 := 5.0, out => "Parametri Macchina"."Temp Provvisoria")
      { S7_Templates := "SrcType := Real" } GT_Contact(in1 := "Temperature"."Temperatura Piastra", in2 := "Parametri Macchina"."Temp Provvisoria")
      S_Coil( "A3 All Max Temp Piastra" )
   END_RUNG
   // the same network as SCL:
   IF "AlwaysTRUE" THEN
       "Parametri Macchina"."Temp Provvisoria" := "Temperature"."Max Temperatura Piastra" + 5.0;
   END_IF;
   IF "AlwaysTRUE" AND ("Temperature"."Temperatura Piastra" > "Parametri Macchina"."Temp Provvisoria") THEN
       "A3 All Max Temp Piastra" := TRUE;
   END_IF;
END_REGION

REGION Network 8: A5 Timeout movimento pin
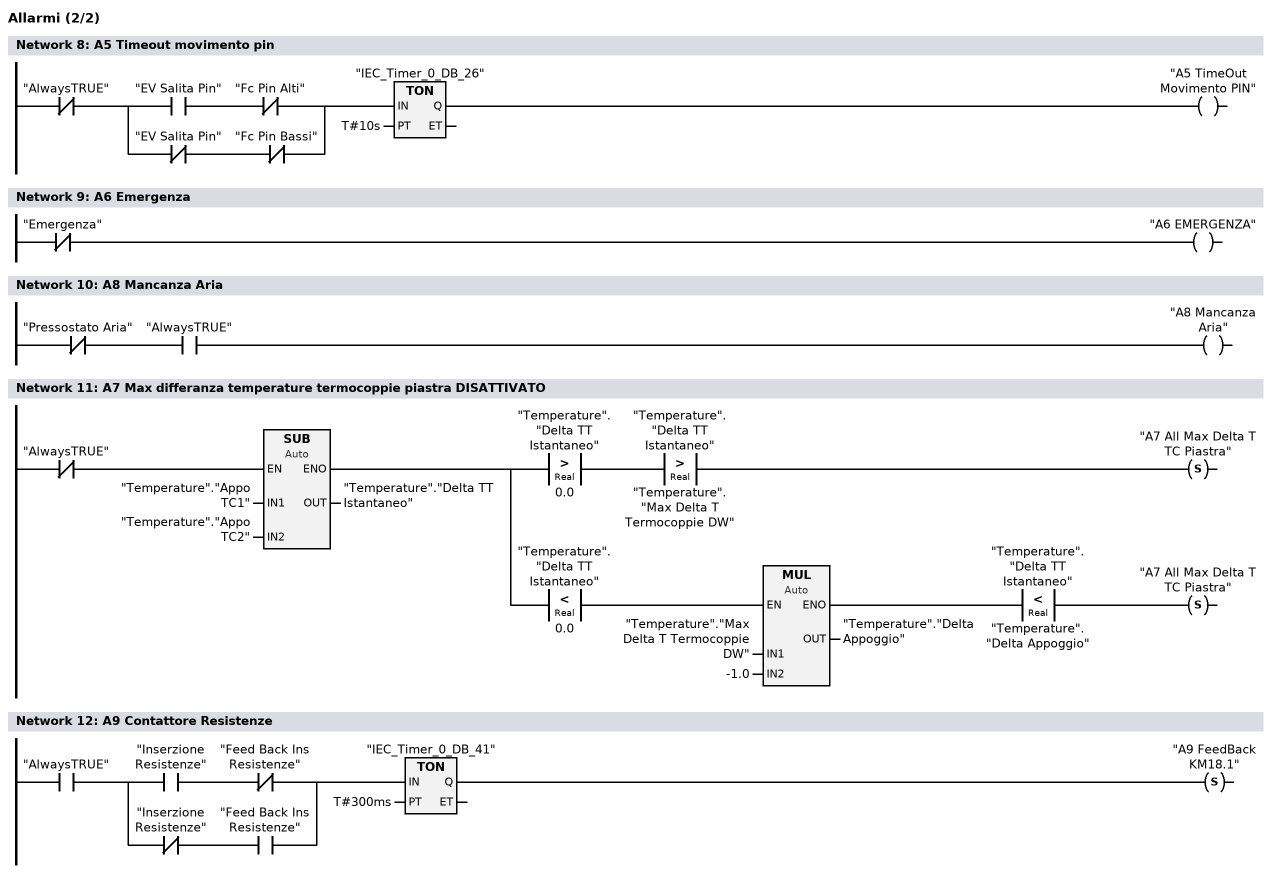
   "IEC_Timer_0_DB_26".TON(IN := NOT "AlwaysTRUE" AND (("EV Salita Pin" AND NOT "Fc Pin Alti") OR (NOT "EV Salita Pin" AND NOT "Fc Pin Bassi")),
                           PT := T#10s);
   "A5 TimeOut Movimento PIN" := "IEC_Timer_0_DB_26".Q;
END_REGION

REGION Network 9: A6 Emergenza
   RUNG wire#powerrail
      I_Contact( "Emergenza" )
      Coil( "A6 EMERGENZA" )
   END_RUNG
   // the same network as SCL:
   "A6 EMERGENZA" := NOT "Emergenza";
END_REGION

REGION Network 10: A8 Mancanza Aria
   RUNG wire#powerrail
      I_Contact( "Pressostato Aria" )
      Contact( "AlwaysTRUE" )
      Coil( "A8 Mancanza Aria" )
   END_RUNG
   // the same network as SCL:
   "A8 Mancanza Aria" := NOT "Pressostato Aria" AND "AlwaysTRUE";
END_REGION

REGION Network 11: A7 Max differanza temperature termocoppie piastra DISATTIVATO
   RUNG wire#powerrail
      I_Contact( "AlwaysTRUE" )
      Sub(in1 := "Temperature"."Appo TC1", in2 := "Temperature"."Appo TC2", out => "Temperature"."Delta TT Istantaneo")
      wire#w1
      { S7_Templates := "SrcType := Real" } GT_Contact(in1 := "Temperature"."Delta TT Istantaneo", in2 := 0.0)
      { S7_Templates := "SrcType := Real" } GT_Contact(in1 := "Temperature"."Delta TT Istantaneo", in2 := "Temperature"."Max Delta T Termocoppie DW")
      S_Coil( "A7 All Max Delta T TC Piastra" )
   END_RUNG
   RUNG wire#w1
      { S7_Templates := "SrcType := Real" } LT_Contact(in1 := "Temperature"."Delta TT Istantaneo", in2 := 0.0)
      Mul(in1 := "Temperature"."Max Delta T Termocoppie DW", in2 := -1.0, out => "Temperature"."Delta Appoggio")
      { S7_Templates := "SrcType := Real" } LT_Contact(in1 := "Temperature"."Delta TT Istantaneo", in2 := "Temperature"."Delta Appoggio")
      S_Coil( "A7 All Max Delta T TC Piastra" )
   END_RUNG
   // the same network as SCL:
   IF NOT "AlwaysTRUE" THEN
       "Temperature"."Delta TT Istantaneo" := "Temperature"."Appo TC1" - "Temperature"."Appo TC2";
   END_IF;
   IF NOT "AlwaysTRUE" AND ("Temperature"."Delta TT Istantaneo" > 0.0) AND ("Temperature"."Delta TT Istantaneo" > "Temperature"."Max Delta T Termocoppie DW") THEN
       "A7 All Max Delta T TC Piastra" := TRUE;
   END_IF;
   #_w1 := NOT "AlwaysTRUE" AND ("Temperature"."Delta TT Istantaneo" < 0.0);
   IF #_w1 THEN
       "Temperature"."Delta Appoggio" := "Temperature"."Max Delta T Termocoppie DW" * (-1.0);
   END_IF;
   IF #_w1 AND ("Temperature"."Delta TT Istantaneo" < "Temperature"."Delta Appoggio") THEN
       "A7 All Max Delta T TC Piastra" := TRUE;
   END_IF;
END_REGION

REGION Network 12: A9 Contattore Resistenze
   "IEC_Timer_0_DB_41".TON(IN := "AlwaysTRUE" AND (("Inserzione Resistenze" AND NOT "Feed Back Ins Resistenze") OR (NOT "Inserzione Resistenze" AND "Feed Back Ins Resistenze")),
                           PT := T#300ms);
   IF "IEC_Timer_0_DB_41".Q THEN "A9 FeedBack KM18.1" := TRUE; END_IF;
END_REGION
END_FUNCTION

FUNCTION "Refrigeracion" : Void   // FC10, LAD
{ S7_Optimized_Access := 'TRUE' }
VERSION : 0.1
   VAR_TEMP   // added for the SCL form of the ladder/FBD networks
      _w1 : Bool;
   END_VAR
BEGIN

